// TIA Portal V18 program export: 2 tag tables, 0 data types, 2 data blocks, 5 code blocks (in call order from the OBs), 1 instance data blocks

VAR_GLOBAL   // PLC tag table "AI_Tags"
   AI_FT3210_Bon3 AT %ID128 : Real;   // Cảm biến lưu lượng nước dosing vào Bồn 3
   AI_FT3210_Bon3_HMI AT %MD756 : Real;   // Giá trị mô phỏng/HMI song song cho Cảm biến lưu lượng nước dosing vào Bồn 3
   AI_FT3210_Bon3_Use_HMI AT %M420.7 : Bool;   // Chọn chế độ mô phỏng HMI cho Cảm biến lưu lượng nước dosing vào Bồn 3
   AI_FT3210_Bon3_Sim_Req AT %M323.0 : Bool;   // Yêu cầu mô phỏng cảm biến cho Cảm biến lưu lượng nước dosing vào Bồn 3
   AI_FT3210_Bon3_Sim_Active AT %M323.1 : Bool;   // Mô phỏng cảm biến đang hoạt động cho Cảm biến lưu lượng nước dosing vào Bồn 3
   AI_FT3210_Bon3_Eff AT %MD760 : Real;   // Giá trị thực tế/mô phỏng hiệu dụng cho Cảm biến lưu lượng nước dosing vào Bồn 3
   AI_LT3213_Bon3 AT %ID132 : Real;   // Cảm biến mức liên tục Bồn 3
   AI_LT3213_Bon3_HMI AT %MD764 : Real;   // Giá trị mô phỏng/HMI song song cho Cảm biến mức liên tục Bồn 3
   AI_LT3213_Bon3_Use_HMI AT %M421.0 : Bool;   // Chọn chế độ mô phỏng HMI cho Cảm biến mức liên tục Bồn 3
   AI_LT3213_Bon3_Sim_Req AT %M323.2 : Bool;   // Yêu cầu mô phỏng cảm biến cho Cảm biến mức liên tục Bồn 3
   AI_LT3213_Bon3_Sim_Active AT %M323.3 : Bool;   // Mô phỏng cảm biến đang hoạt động cho Cảm biến mức liên tục Bồn 3
   AI_LT3213_Bon3_Eff AT %MD768 : Real;   // Giá trị thực tế/mô phỏng hiệu dụng cho Cảm biến mức liên tục Bồn 3
   AI_TT3214_Bon3 AT %ID136 : Real;   // Cảm biến nhiệt độ Bồn 3
   AI_TT3214_Bon3_HMI AT %MD772 : Real;   // Giá trị mô phỏng/HMI song song cho Cảm biến nhiệt độ Bồn 3
   AI_TT3214_Bon3_Use_HMI AT %M421.1 : Bool;   // Chọn chế độ mô phỏng HMI cho Cảm biến nhiệt độ Bồn 3
   AI_TT3214_Bon3_Sim_Req AT %M323.4 : Bool;   // Yêu cầu mô phỏng cảm biến cho Cảm biến nhiệt độ Bồn 3
   AI_TT3214_Bon3_Sim_Active AT %M323.5 : Bool;   // Mô phỏng cảm biến đang hoạt động cho Cảm biến nhiệt độ Bồn 3
   AI_TT3214_Bon3_Eff AT %MD776 : Real;   // Giá trị thực tế/mô phỏng hiệu dụng cho Cảm biến nhiệt độ Bồn 3
   AI_FT3215_Bon4 AT %ID140 : Real;   // Cảm biến lưu lượng nước dosing vào Bồn 4
   AI_FT3215_Bon4_HMI AT %MD780 : Real;   // Giá trị mô phỏng/HMI song song cho Cảm biến lưu lượng nước dosing vào Bồn 4
   AI_FT3215_Bon4_Use_HMI AT %M421.2 : Bool;   // Chọn chế độ mô phỏng HMI cho Cảm biến lưu lượng nước dosing vào Bồn 4
   AI_FT3215_Bon4_Sim_Req AT %M323.6 : Bool;   // Yêu cầu mô phỏng cảm biến cho Cảm biến lưu lượng nước dosing vào Bồn 4
   AI_FT3215_Bon4_Sim_Active AT %M323.7 : Bool;   // Mô phỏng cảm biến đang hoạt động cho Cảm biến lưu lượng nước dosing vào Bồn 4
   AI_FT3215_Bon4_Eff AT %MD784 : Real;   // Giá trị thực tế/mô phỏng hiệu dụng cho Cảm biến lưu lượng nước dosing vào Bồn 4
   AI_FQ3215_Bon4 AT %ID144 : Real;   // Bộ đếm lưu lượng tích lũy Bồn 4
   AI_FQ3215_Bon4_HMI AT %MD788 : Real;   // Giá trị mô phỏng/HMI song song cho Bộ đếm lưu lượng tích lũy Bồn 4
   AI_FQ3215_Bon4_Use_HMI AT %M421.3 : Bool;   // Chọn chế độ mô phỏng HMI cho Bộ đếm lưu lượng tích lũy Bồn 4
   AI_FQ3215_Bon4_Sim_Req AT %M324.0 : Bool;   // Yêu cầu mô phỏng cảm biến cho Bộ đếm lưu lượng tích lũy Bồn 4
   AI_FQ3215_Bon4_Sim_Active AT %M324.1 : Bool;   // Mô phỏng cảm biến đang hoạt động cho Bộ đếm lưu lượng tích lũy Bồn 4
   AI_FQ3215_Bon4_Eff AT %MD792 : Real;   // Giá trị thực tế/mô phỏng hiệu dụng cho Bộ đếm lưu lượng tích lũy Bồn 4
   AI_LS3217_Bon4_Cao AT %I0.5 : Bool;   // Cảm biến mức cao Bồn 4
   AI_LS3217_Bon4_Cao_HMI AT %M110.5 : Bool;   // Tín hiệu mô phỏng/HMI song song cho Cảm biến mức cao Bồn 4
   AI_LS3217_Bon4_Cao_HMI_Gated AT %M324.2 : Bool;   // Tín hiệu HMI đã qua xử lý chế độ cho Cảm biến mức cao Bồn 4
   AI_LS3217_Bon4_Cao_Eff AT %M324.3 : Bool;   // Tín hiệu thực tế/mô phỏng hiệu dụng cho Cảm biến mức cao Bồn 4
   AI_LT3218_Bon4 AT %ID148 : Real;   // Cảm biến mức liên tục Bồn 4
   AI_LT3218_Bon4_HMI AT %MD796 : Real;   // Giá trị mô phỏng/HMI song song cho Cảm biến mức liên tục Bồn 4
   AI_LT3218_Bon4_Use_HMI AT %M421.4 : Bool;   // Chọn chế độ mô phỏng HMI cho Cảm biến mức liên tục Bồn 4
   AI_LT3218_Bon4_Sim_Req AT %M324.4 : Bool;   // Yêu cầu mô phỏng cảm biến cho Cảm biến mức liên tục Bồn 4
   AI_LT3218_Bon4_Sim_Active AT %M324.5 : Bool;   // Mô phỏng cảm biến đang hoạt động cho Cảm biến mức liên tục Bồn 4
   AI_LT3218_Bon4_Eff AT %MD800 : Real;   // Giá trị thực tế/mô phỏng hiệu dụng cho Cảm biến mức liên tục Bồn 4
   AI_TT3219_Bon4 AT %ID152 : Real;   // Cảm biến nhiệt độ Bồn 4
   AI_TT3219_Bon4_HMI AT %MD804 : Real;   // Giá trị mô phỏng/HMI song song cho Cảm biến nhiệt độ Bồn 4
   AI_TT3219_Bon4_Use_HMI AT %M421.5 : Bool;   // Chọn chế độ mô phỏng HMI cho Cảm biến nhiệt độ Bồn 4
   AI_TT3219_Bon4_Sim_Req AT %M324.6 : Bool;   // Yêu cầu mô phỏng cảm biến cho Cảm biến nhiệt độ Bồn 4
   AI_TT3219_Bon4_Sim_Active AT %M324.7 : Bool;   // Mô phỏng cảm biến đang hoạt động cho Cảm biến nhiệt độ Bồn 4
   AI_TT3219_Bon4_Eff AT %MD808 : Real;   // Giá trị thực tế/mô phỏng hiệu dụng cho Cảm biến nhiệt độ Bồn 4
   AI_V3240_Nuoc_Bon3 AT %Q1.4 : Bool;   // Van on/off cấp nước Bồn 3
   AI_V3240_Nuoc_Bon3_M AT %M221.4 : Bool;   // Tag gương phản hồi HMI cho Van on/off cấp nước Bồn 3
   AI_CV3211_Nuoc_Bon3 AT %QD116 : Real;   // Van tuyến tính cấp nước Bồn 3
   AI_CV3211_Nuoc_Bon3_M AT %MD936 : Real;   // Tag gương phản hồi HMI cho Van tuyến tính cấp nước Bồn 3
   AI_AGTR3262_Khuay_Bon3 AT %Q1.5 : Bool;   // Động cơ khuấy Bồn 3
   AI_AGTR3262_Khuay_Bon3_M AT %M221.5 : Bool;   // Tag gương phản hồi HMI cho Động cơ khuấy Bồn 3
   AI_AGTR3262_Toc_Do_AO AT %QD120 : Real;   // Tín hiệu tốc độ khuấy Bồn 3
   AI_AGTR3262_Toc_Do_AO_M AT %MD940 : Real;   // Tag gương phản hồi HMI cho Tín hiệu tốc độ khuấy Bồn 3
   AI_V3242_Xa_Bon3 AT %Q1.6 : Bool;   // Van xả đáy Bồn 3 số 1
   AI_V3242_Xa_Bon3_M AT %M221.6 : Bool;   // Tag gương phản hồi HMI cho Van xả đáy Bồn 3 số 1
   AI_V3243_Xa_Bon3 AT %Q1.7 : Bool;   // Van xả đáy Bồn 3 số 2
   AI_V3243_Xa_Bon3_M AT %M221.7 : Bool;   // Tag gương phản hồi HMI cho Van xả đáy Bồn 3 số 2
   AI_V3244_Xa_Bon3 AT %Q2.0 : Bool;   // Van xả đáy Bồn 3 số 3
   AI_V3244_Xa_Bon3_M AT %M222.0 : Bool;   // Tag gương phản hồi HMI cho Van xả đáy Bồn 3 số 3
   AI_V3245_Nuoc_Bon4 AT %Q2.1 : Bool;   // Van on/off cấp nước Bồn 4
   AI_V3245_Nuoc_Bon4_M AT %M222.1 : Bool;   // Tag gương phản hồi HMI cho Van on/off cấp nước Bồn 4
   AI_CV3216_Hoi_Bon4 AT %QD124 : Real;   // Van tuyến tính gia nhiệt mô phỏng Bồn 4
   AI_CV3216_Hoi_Bon4_M AT %MD944 : Real;   // Tag gương phản hồi HMI cho Van tuyến tính gia nhiệt mô phỏng Bồn 4
   AI_AGTR3263_Khuay_Bon4 AT %Q2.2 : Bool;   // Động cơ khuấy Bồn 4
   AI_AGTR3263_Khuay_Bon4_M AT %M222.2 : Bool;   // Tag gương phản hồi HMI cho Động cơ khuấy Bồn 4
   AI_AGTR3263_Dao_Chieu AT %Q2.3 : Bool;   // Lệnh đảo chiều động cơ khuấy Bồn 4
   AI_AGTR3263_Dao_Chieu_M AT %M222.3 : Bool;   // Tag gương phản hồi HMI cho Lệnh đảo chiều động cơ khuấy Bồn 4
   AI_AGTR3263_Toc_Do_AO AT %QD128 : Real;   // Tốc độ đặt động cơ khuấy Bồn 4
   AI_AGTR3263_Toc_Do_AO_M AT %MD948 : Real;   // Tag gương phản hồi HMI cho Tốc độ đặt động cơ khuấy Bồn 4
   AI_V3247_Xa_Bon4 AT %Q2.4 : Bool;   // Van xả đáy Bồn 4 số 1
   AI_V3247_Xa_Bon4_M AT %M222.4 : Bool;   // Tag gương phản hồi HMI cho Van xả đáy Bồn 4 số 1
   AI_V3248_Xa_Bon4 AT %Q2.5 : Bool;   // Van xả đáy Bồn 4 số 2
   AI_V3248_Xa_Bon4_M AT %M222.5 : Bool;   // Tag gương phản hồi HMI cho Van xả đáy Bồn 4 số 2
   AI_V3249_Xa_Bon4 AT %Q2.6 : Bool;   // Van xả đáy Bồn 4 số 3
   AI_V3249_Xa_Bon4_M AT %M222.6 : Bool;   // Tag gương phản hồi HMI cho Van xả đáy Bồn 4 số 3
   AI_Pump3265_Chuyen_Nhanh2 AT %Q2.7 : Bool;   // Bơm chuyển dung dịch Nhánh 2 xuống bồn chứa
   AI_Pump3265_Chuyen_Nhanh2_M AT %M222.7 : Bool;   // Tag gương phản hồi HMI cho Bơm chuyển dung dịch Nhánh 2 xuống bồn chứa
   AI_HMI_Operator_Login AT %M422.5 : Bool;   // Đăng nhập quyền Operator
   AI_HMI_Engineer_Login AT %M422.6 : Bool;   // Đăng nhập quyền Engineer
   AI_HMI_Admin_Login AT %M422.7 : Bool;   // Đăng nhập quyền Admin
   AI_HMI_Che_Do_Manual AT %M423.0 : Bool;   // Cho phép điều khiển tay từng thiết bị
   AI_HMI_Ack_Alarm AT %M423.1 : Bool;   // Xác nhận cảnh báo
   AI_HMI_Reset_Alarm AT %M423.2 : Bool;   // Reset alarm bằng HMI
   AI_Gia_Lap_Mat_Ket_Noi_HMI AT %M423.3 : Bool;   // Nút giả lập mất kết nối PLC
   AI_HMI_User_Level AT %MW520 : Int;   // Mức quyền hiện tại: 1 Operator, 2 Engineer, 3 Admin
   AI_HMI_Cho_Phep_Sua_Thong_So AT %M327.2 : Bool;   // Cờ cho phép sửa công thức và PID
   AI_HMI_Alarm_Status AT %MW522 : Int;   // Mã cảnh báo tổng hợp cho WinCC TextList
   AI_HMI_AnToan_Status AT %MW524 : Int;   // Mã chẩn đoán an toàn ưu tiên
   AI_PLC2_Auto_Enable AT %M328.1 : Bool;   // Cho phép chạy Auto Nhánh 2 Bồn 3-4
   AI_PLC2_EStop_Latch AT %M328.2 : Bool;   // Chốt dừng khẩn HMI/SCADA Nhánh 2 Bồn 3-4
   AI_PLC2_Loi_Tong AT %M328.3 : Bool;   // Lỗi tổng khóa Auto Nhánh 2 Bồn 3-4
   AI_PLC2_Loi_Dry_Run AT %M328.4 : Bool;   // Lỗi chạy khô bơm Nhánh 2 Bồn 3-4
   AI_PLC2_Loi_Dosing AT %M328.5 : Bool;   // Lỗi quá thời gian dosing Nhánh 2 Bồn 3-4
   AI_PLC2_Loi_Truyen_Thong AT %M328.6 : Bool;   // Lỗi truyền thông mô phỏng Nhánh 2 Bồn 3-4
   AI_PLC2_State AT %MW528 : Int;   // Mã bước chu trình Nhánh 2 Bồn 3-4
   AI_PLC2_Step_Bon3_Dosing AT %M330.4 : Bool;   // Bồn 3 đang dosing nước
   AI_PLC2_Step_Bon3_Tip AT %M330.5 : Bool;   // Bồn 3 đang mô phỏng tip cốt tương đậu đậm đặc
   AI_PLC2_Step_Bon3_Khuay AT %M330.6 : Bool;   // Bồn 3 đang khuấy ban đầu
   AI_PLC2_Step_Bon3_Xa AT %M330.7 : Bool;   // Bồn 3 đang xả sang Bồn 4
   AI_PLC2_Step_Bon4_Dosing AT %M331.0 : Bool;   // Bồn 4 đang dosing bổ sung
   AI_PLC2_Step_Bon4_Tip AT %M331.1 : Bool;   // Bồn 4 đang tip phụ gia
   AI_PLC2_Step_Bon4_Khuay_Thuan AT %M331.2 : Bool;   // Bồn 4 khuấy chiều thuận
   AI_PLC2_Step_Bon4_Khuay_Nghich AT %M331.3 : Bool;   // Bồn 4 khuấy chiều ngược
   AI_PLC2_Step_Bon4_PID_Mo_Phong AT %M331.4 : Bool;   // Bồn 4 chạy PID mô phỏng
   AI_PLC2_Step_Bon4_Thanh_Trung AT %M331.5 : Bool;   // Bồn 4 giữ thời gian thanh trùng
   AI_PLC2_Xa_Bon3_Xong AT %M331.6 : Bool;   // Bồn 3 đã xả hết
   AI_PLC2_Xa_Bon4_Xong AT %M331.7 : Bool;   // Bồn 4 đã xả hết
   AI_PLC2_Me_Nhanh2_Hoan_Thanh AT %M332.5 : Bool;   // Cờ hoàn thành Nhánh 2 gửi sang PLC1
   AI_PLC2_Me_Nhanh2_Hoan_Thanh_M AT %M224.6 : Bool;   // Tag gương phản hồi HMI cho cờ hoàn thành Nhánh 2 gửi sang PLC1
   AI_Pump3265_Chuyen_Nhanh2_Cmd_Nhan AT %M333.0 : Bool;   // Nhận lệnh chạy bơm chuyển Nhánh 2 từ PLC1
   AI_Pump3265_Chuyen_Nhanh2_Cmd_Nhan_HMI AT %M111.1 : Bool;   // Tín hiệu mô phỏng/HMI song song cho lệnh chạy bơm chuyển Nhánh 2 từ PLC1
   AI_Nut_Khoi_Dong_Nhan AT %M333.2 : Bool;   // nút khởi động nhận từ PLC1
   AI_Nut_Khoi_Dong_Nhan_HMI AT %M111.2 : Bool;   // Tín hiệu mô phỏng/HMI song song cho nút khởi động nhận từ PLC1
   AI_Nut_Khoi_Dong_Nhan_HMI_Gated AT %M333.3 : Bool;   // Tín hiệu HMI đã qua xử lý chế độ cho nút khởi động nhận từ PLC1
   AI_Nut_Khoi_Dong_Nhan_Eff AT %M333.4 : Bool;   // Tín hiệu thực tế/mô phỏng hiệu dụng cho nút khởi động nhận từ PLC1
   AI_Nut_Dung_Nhan AT %M333.5 : Bool;   // nút dừng nhận từ PLC1
   AI_Nut_Dung_Nhan_HMI AT %M111.3 : Bool;   // Tín hiệu mô phỏng/HMI song song cho nút dừng nhận từ PLC1
   AI_Nut_Dung_Nhan_HMI_Gated AT %M333.6 : Bool;   // Tín hiệu HMI đã qua xử lý chế độ cho nút dừng nhận từ PLC1
   AI_Nut_Dung_Nhan_Eff AT %M333.7 : Bool;   // Tín hiệu thực tế/mô phỏng hiệu dụng cho nút dừng nhận từ PLC1
   AI_Nut_Reset_Nhan AT %M334.0 : Bool;   // nút reset nhận từ PLC1
   AI_Nut_Reset_Nhan_HMI AT %M111.4 : Bool;   // Tín hiệu mô phỏng/HMI song song cho nút reset nhận từ PLC1
   AI_Nut_Reset_Nhan_HMI_Gated AT %M334.1 : Bool;   // Tín hiệu HMI đã qua xử lý chế độ cho nút reset nhận từ PLC1
   AI_Nut_Reset_Nhan_Eff AT %M334.2 : Bool;   // Tín hiệu thực tế/mô phỏng hiệu dụng cho nút reset nhận từ PLC1
   AI_Nut_EStop_Nhan AT %M334.3 : Bool;   // nút dừng khẩn nhận từ PLC1
   AI_Nut_EStop_Nhan_HMI AT %M111.5 : Bool;   // Tín hiệu mô phỏng/HMI song song cho nút dừng khẩn nhận từ PLC1
   AI_Nut_EStop_Nhan_HMI_Gated AT %M334.4 : Bool;   // Tín hiệu HMI đã qua xử lý chế độ cho nút dừng khẩn nhận từ PLC1
   AI_Nut_EStop_Nhan_Eff AT %M334.5 : Bool;   // Tín hiệu thực tế/mô phỏng hiệu dụng cho nút dừng khẩn nhận từ PLC1
   AI_Clock_1Hz AT %M100.5 : Bool;   // Clock 1Hz system memory bit
   AI_FirstScan AT %M101.0 : Bool;   // First Scan system memory bit
   AI_PLC2_Last_CmdSeq AT %MW80 : Int;   // Last processed command sequence
   AI_PLC2_CmdSeq_New AT %M82.0 : Bool;   // New command sequence received
   AI_MB_TCP_Server_Error AT %M82.1 : Bool;   // Modbus TCP Server Error
   AI_MB_TCP_Server_Status AT %MW84 : Word;   // Modbus TCP Server Status
   AI_MB_TCP_Server_NDR AT %M82.2 : Bool;   // Modbus TCP Server New Data Received
   AI_MB_TCP_Server_DR AT %M82.3 : Bool;   // Modbus TCP Server Data Read
   AI_PLC1_Tip_Bon1_Xong_HMI AT %M423.4 : Bool;   // Nút mô phỏng tip Bồn 1 đã hoàn tất
   AI_PLC1_Khuay_Bon1_Xong_HMI AT %M423.5 : Bool;   // Nút mô phỏng hết thời gian khuấy Bồn 1
   AI_PLC1_Tip_Bon2_Xong_HMI AT %M423.6 : Bool;   // Nút mô phỏng tip Bồn 2 đã hoàn tất
   AI_PLC1_Khuay_Thuan_Bon2_Xong_HMI AT %M423.7 : Bool;   // Nút mô phỏng hết thời gian khuấy thuận Bồn 2
   AI_PLC1_Khuay_Nghich_Bon2_Xong_HMI AT %M424.0 : Bool;   // Nút mô phỏng hết thời gian khuấy ngược Bồn 2
   AI_PLC1_Thanh_Trung_Bon2_Xong_HMI AT %M424.1 : Bool;   // Nút mô phỏng hết thời gian thanh trùng Bồn 2
   AI_PLC2_Tip_Bon3_Xong_HMI AT %M424.2 : Bool;   // Nút mô phỏng tip Bồn 3 đã hoàn tất
   AI_PLC2_Khuay_Bon3_Xong_HMI AT %M424.3 : Bool;   // Nút mô phỏng hết thời gian khuấy Bồn 3
   AI_PLC2_Tip_Bon4_Xong_HMI AT %M424.4 : Bool;   // Nút mô phỏng tip Bồn 4 đã hoàn tất
   AI_PLC2_Khuay_Thuan_Bon4_Xong_HMI AT %M424.5 : Bool;   // Nút mô phỏng hết thời gian khuấy thuận Bồn 4
   AI_PLC2_Khuay_Nghich_Bon4_Xong_HMI AT %M424.6 : Bool;   // Nút mô phỏng hết thời gian khuấy ngược Bồn 4
   AI_PLC2_Thanh_Trung_Bon4_Xong_HMI AT %M424.7 : Bool;   // Nút mô phỏng hết thời gian thanh trùng Bồn 4
   AI_BonChua_Nhan_Dich_Xong_HMI AT %M425.0 : Bool;   // Nút mô phỏng nhận dịch vào Bồn chứa 01 xong
   AI_BonChua_Chuyen_Bon2_Xong_HMI AT %M425.1 : Bool;   // Nút mô phỏng chuyển sang Bồn chứa 02 xong
   AI_HMI_SP_PLC1_Nuoc_Bon1 AT %MD880 : Real;   // Lượng nước dosing Bồn 1
   AI_HMI_SP_PLC1_Nuoc_Bon2 AT %MD884 : Real;   // Lượng nước dosing bổ sung Bồn 2
   AI_HMI_SP_PLC1_Toc_Do_Bon1 AT %MD888 : Real;   // Tốc độ khuấy Bồn 1
   AI_HMI_SP_PLC1_Toc_Do_Bon2_Main AT %MD892 : Real;   // Tốc độ khuấy chính Bồn 2
   AI_HMI_SP_PLC1_Nhiet_Do_Bon2 AT %MD896 : Real;   // Setpoint nhiệt/PID Bồn 2
   AI_HMI_SP_PLC2_Nuoc_Bon3 AT %MD900 : Real;   // Lượng nước dosing Bồn 3
   AI_HMI_SP_PLC2_Nuoc_Bon4 AT %MD904 : Real;   // Lượng nước dosing bổ sung Bồn 4
   AI_HMI_SP_PLC2_Toc_Do_Bon3 AT %MD908 : Real;   // Tốc độ khuấy Bồn 3
   AI_HMI_SP_PLC2_Toc_Do_Bon4_Main AT %MD912 : Real;   // Tốc độ khuấy chính Bồn 4
   AI_HMI_SP_PLC2_Nhiet_Do_Bon4 AT %MD916 : Real;   // Setpoint nhiệt/PID mô phỏng Bồn 4
   AI_HMI_SP_BonChua1_Nhiet_Giai_Nhiet AT %MD920 : Real;   // Nhiệt độ giải nhiệt đích Bồn chứa 01
   AI_HMI_SP_Loc_Ap_Suat_Max AT %MD924 : Real;   // Ngưỡng áp suất cao trước màng lọc
   AI_HMI_SP_Time_Khuay_Bon1 AT %MD928 : Time;   // Thời gian khuấy Bồn 1
   AI_HMI_SP_Time_Khuay_Bon3 AT %MD932 : Time;   // Thời gian khuấy Bồn 3
   AI_HMI_SP_Time_Fwd AT %MD936 : Time;   // Thời gian khuấy chiều thuận
   AI_HMI_SP_Time_Rev AT %MD940 : Time;   // Thời gian khuấy chiều ngược
   AI_HMI_SP_Time_Sterilize AT %MD944 : Time;   // Thời gian giữ nhiệt thanh trùng
   AI_PLC1_Khuay_Bon1_Xong AT %M335.3 : Bool;   // Trạng thái tự động xong khuấy Bồn 1
   AI_PLC1_Khuay_Thuan_Bon2_Xong AT %M335.4 : Bool;   // Trạng thái tự động xong khuấy thuận Bồn 2
   AI_PLC1_Khuay_Nghich_Bon2_Xong AT %M335.5 : Bool;   // Trạng thái tự động xong khuấy ngược Bồn 2
   AI_PLC1_Thanh_Trung_Bon2_Xong AT %M335.6 : Bool;   // Trạng thái tự động xong thanh trùng Bồn 2
   AI_PLC2_Khuay_Bon3_Xong AT %M335.7 : Bool;   // Trạng thái tự động xong khuấy Bồn 3
   AI_PLC2_Khuay_Thuan_Bon4_Xong AT %M336.0 : Bool;   // Trạng thái tự động xong khuấy thuận Bồn 4
   AI_PLC2_Khuay_Nghich_Bon4_Xong AT %M336.1 : Bool;   // Trạng thái tự động xong khuấy ngược Bồn 4
   AI_PLC2_Thanh_Trung_Bon4_Xong AT %M336.2 : Bool;   // Trạng thái tự động xong thanh trùng Bồn 4
   AI_PID_Bon2_Enable AT %M336.3 : Bool;   // Cho phép PID Bồn 2
   AI_PID_Bon2_ManualEnable AT %M336.4 : Bool;   // Chế độ manual PID Bồn 2
   AI_PID_Bon2_Error AT %M336.5 : Bool;   // Lỗi khối PID Bồn 2
   AI_PID_Bon4_Enable AT %M336.6 : Bool;   // Cho phép PID mô phỏng Bồn 4
   AI_PID_Bon4_ManualEnable AT %M336.7 : Bool;   // Chế độ manual PID Bồn 4
   AI_PID_Bon4_Error AT %M337.0 : Bool;   // Lỗi khối PID Bồn 4
   AI_PID_Bon2_ErrorBits AT %MD948 : DWord;   // Mã lỗi DWORD PID Bồn 2
   AI_PID_Bon4_ErrorBits AT %MD952 : DWord;   // Mã lỗi DWORD PID Bồn 4
   AI_PID_Bon2_SP AT %MD956 : Real;   // Setpoint đưa vào PID Bồn 2
   AI_PID_Bon2_Err AT %MD960 : Real;   // Sai lệch PID Bồn 2 = SP - PV
   AI_PID_Bon2_CV AT %MD964 : Real;   // Giá trị điều khiển PID Bồn 2
   AI_PID_Bon2_ManualValue AT %MD968 : Real;   // Giá trị manual PID Bồn 2
   AI_PID_Bon4_SP AT %MD972 : Real;   // Setpoint đưa vào PID mô phỏng Bồn 4
   AI_PID_Bon4_Err AT %MD976 : Real;   // Sai lệch PID mô phỏng Bồn 4 = SP - PV
   AI_PID_Bon4_CV AT %MD980 : Real;   // Giá trị điều khiển PID mô phỏng Bồn 4
   AI_PID_Bon4_ManualValue AT %MD984 : Real;   // Giá trị manual PID Bồn 4
   AI_TT3219_Bon4_Sim AT %MD988 : Real;   // Nhiệt độ mô phỏng nội bộ cho PID Bồn 4
   AI_PID_Bon4_Tang_Nhiet_Buoc AT %MD992 : Real;   // Mức tăng nhiệt mô phỏng mỗi chu kỳ OB31
   AI_TT3219_Bon4_Target AT %MD996 : Real;   // Nhiệt độ đích mô phỏng bồn 4
   AI_TT3219_Bon4_Sim_Pure AT %MD1000 : Real;   // Nhiệt độ mô phỏng chưa có nhiễu bồn 4
   AI_PID_Bon4_Temp_Val_1 AT %MD1004 : Real;   // Biến tạm mô phỏng nhiệt độ 1
   AI_PID_Bon4_Temp_Val_2 AT %MD1008 : Real;   // Biến tạm mô phỏng nhiệt độ 2
   AI_PID_Bon4_Sim_Counter AT %MD1012 : Real;   // Đồng hồ chu kỳ mô phỏng
   AI_PID_Bon4_Sim_Angle AT %MD1016 : Real;   // Góc lượng giác nhiễu
   AI_PID_Bon4_Sim_Sin AT %MD1020 : Real;   // Giá trị hình sin nhiễu
   AI_PID_Bon4_Sim_Noise AT %MD1024 : Real;   // Giá trị nhiễu nhiệt độ
   AI_PID_Bon4_State AT %MW536 : Int;   // Trạng thái khối PID Bồn 4
   AI_PLC2_Stop_Active AT %M337.2 : Bool;   // Tín hiệu dừng active PLC2
   AI_AGTR3263_Khuay_Active AT %M337.5 : Bool;   // Trạng thái khuấy Bồn 4 active
   AI_AGTR3263_Should_Run AT %M337.6 : Bool;   // Yêu cầu chạy động cơ Bồn 4
   AI_HMI_Use_Sim_Input_PLC2 AT %M338.0 : Bool;   // Cho phép sử dụng đầu vào mô phỏng PLC2
   AI_Pump3265_Chuyen_Nhanh2_Cmd_Nhan_Eff AT %M338.3 : Bool;   // Lệnh chạy bơm chuyển Nhánh 2 nhận được hiệu dụng
   AI_Pump3265_Chuyen_Nhanh2_Cmd_Nhan_HMI_Gated AT %M338.5 : Bool;   // Lệnh chạy bơm chuyển Nhánh 2 HMI gated
   AI_PLC2_SP_Valid AT %M338.7 : Bool;   // Setpoint PLC2 hợp lệ
   AI_PLC2_Loi_Setpoint AT %M339.2 : Bool;   // Lỗi Setpoint PLC2
   AI_Init_Defaults_Done_PLC2 AT %M339.5 : Bool;   // Khởi tạo Setpoint mặc định PLC2 hoàn tất
   AI_Init_Trigger_PLC2 AT %M340.0 : Bool;   // Cờ kích hoạt nạp recipe mặc định PLC2
   AI_HMI_Load_Default_Recipe AT %M340.2 : Bool;   // Yêu cầu nạp lại Recipe mặc định từ HMI
   AI_PLC2_Load_Default_Cmd_Nhan AT %M340.4 : Bool;   // Nhận lệnh nạp recipe mặc định từ PLC1
   AI_PLC2_Load_Default_Cmd_Nhan_HMI AT %M111.6 : Bool;   // Tín hiệu mô phỏng/HMI cho nhận lệnh nạp recipe
   AI_PLC2_Load_Default_Cmd_Nhan_HMI_Gated AT %M340.5 : Bool;   // Tín hiệu nhận lệnh nạp recipe HMI gated
   AI_PLC2_Load_Default_Cmd_Nhan_Eff AT %M340.6 : Bool;   // Tín hiệu nhận lệnh nạp recipe hiệu dụng
   AI_PLC2_Load_Default_Done AT %M340.7 : Bool;   // Báo nạp recipe mặc định xong gửi sang PLC1
   AI_PLC2_Load_Default_Done_M AT %M225.1 : Bool;   // Tag gương phản hồi HMI cho báo nạp recipe xong PLC2
   AI_HMI_Sim_Mode AT %M341.3 : Bool;   // Cho phép toàn bộ tín hiệu mô phỏng HMI tác động vào input hiệu dụng
   AI_HMI_Run_Enable AT %M341.4 : Bool;   // Cho phép vận hành từ HMI ở chế độ thật
   AI_System_Mode_Real AT %M341.5 : Bool;   // Hệ thống đang hoạt động ở chế độ thực tế
   AI_System_Mode_Sim AT %M341.6 : Bool;   // Hệ thống đang hoạt động ở chế độ mô phỏng
   AI_HMI_Sim_Active_Warning AT %M341.7 : Bool;   // Cảnh báo chế độ mô phỏng HMI đang hoạt động
   AI_PID_Bon4_Kp_HMI AT %MD1036 : Real;   // HMI parameter for Kp PID Bồn 4
   AI_PID_Bon4_Ti_HMI AT %MD1040 : Real;   // HMI parameter for Ti PID Bồn 4
END_VAR

VAR_GLOBAL   // PLC tag table "Default tag table"
   System_Byte AT %MB101 : Byte;
   FirstScan AT %M101.0 : Bool;
   DiagStatusUpdate AT %M101.1 : Bool;
   AlwaysTRUE AT %M101.2 : Bool;
   AlwaysFALSE AT %M101.3 : Bool;
   Clock_Byte AT %MB100 : Byte;
   Clock_10Hz AT %M100.0 : Bool;
   Clock_5Hz AT %M100.1 : Bool;
   "Clock_2.5Hz" AT %M100.2 : Bool;
   Clock_2Hz AT %M100.3 : Bool;
   "Clock_1.25Hz" AT %M100.4 : Bool;
   Clock_1Hz AT %M100.5 : Bool;
   "Clock_0.625Hz" AT %M100.6 : Bool;
   "Clock_0.5Hz" AT %M100.7 : Bool;
END_VAR

DATA_BLOCK "AI_Timers_PLC2"   // DB1
TITLE = AI_Timers_PLC2
{ S7_Optimized_Access := 'TRUE' }
VERSION : 0.1
// Global DB containing all timers and PID instances
// stored: AutoNumber true, DBAccessibleFromOPCUA true, IsOnlyStoredInLoadMemory false, IsRetainMemResEnabled false, IsWriteProtectedInAS false, MemoryReserve 100
   VAR
      AI_Timer_Dosing_Bon3 : IEC_TIMER;
      AI_Timer_Dosing_Bon4 : IEC_TIMER;
      AI_Timer_Khuay_Bon3 : IEC_TIMER;
      AI_Timer_Khuay_Thuan_Bon4 : IEC_TIMER;
      AI_Timer_Khuay_Nghich_Bon4 : IEC_TIMER;
      AI_Timer_Thanh_Trung_Bon4 : IEC_TIMER;
   END_VAR
BEGIN
END_DATA_BLOCK

DATA_BLOCK "DB_Modbus_Holding_Register_DB"   // DB20
TITLE = DB_Modbus_Holding_Register_DB
{ S7_Optimized_Access := 'FALSE' }
VERSION : 0.1
// DB communication via Modbus TCP
// stored: AutoNumber false, DBAccessibleFromOPCUA true, IsOnlyStoredInLoadMemory false, IsWriteProtectedInAS false
   VAR
      CmdSeq : Int;
      Cmd_Start : Bool;
      Cmd_Stop : Bool;
      Cmd_Reset : Bool;
      Cmd_EStop : Bool;
      Cmd_Pump_Branch2_To_SubTanks : Bool;
      Cmd_Load_Recipe : Bool;
      Heartbeat_Client : Int;
      AckSeq : Int;
      Done_Branch2 : Bool;
      Done_Recipe : Bool;
      Alarm : Bool;
      State : Int;
      PID_Bon4_SP : Real;
      PID_Bon4_PV : Real;
      PID_Bon4_CV : Real;
      Heartbeat_Server : Int;
   END_VAR
BEGIN
END_DATA_BLOCK

ORGANIZATION_BLOCK "Main"   // OB1, LAD, ProgramCycle
TITLE = "Main Program Sweep (Cycle)"
{ S7_Optimized_Access := 'TRUE' }
VERSION : 0.1
// stored: AutoNumber true, IsIECCheckEnabled false, SetENOAutomatically false
   VAR_INPUT
      Initial_Call : Bool;   // Initial call of this OB
      Remanence : Bool;   // =True, if remanent data are available
   END_VAR
BEGIN

REGION Network 1: Modbus TCP Server - Call MB_SERVER
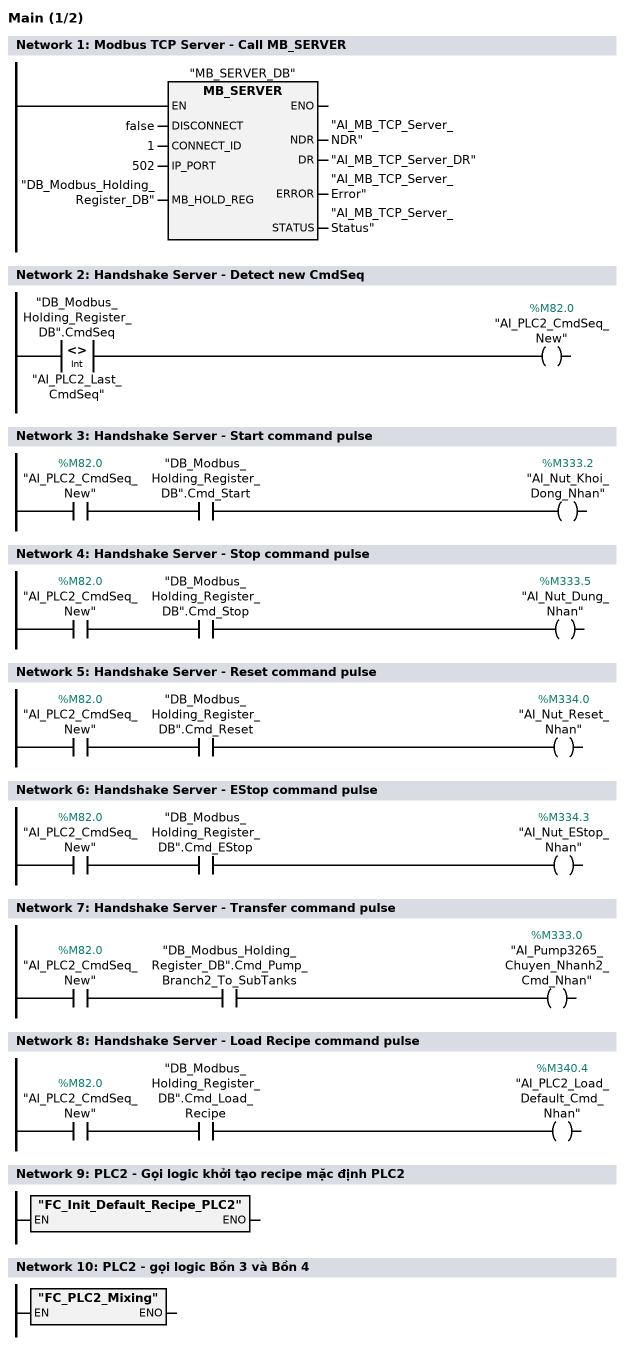
   RUNG wire#powerrail
      { S7_Templates := "[card1200 := 1, card1500 := 0]" } "MB_SERVER_DB".MB_SERVER(DISCONNECT := false, CONNECT_ID := 1, IP_PORT := 502, MB_HOLD_REG := "DB_Modbus_Holding_Register_DB", NDR => "AI_MB_TCP_Server_NDR", DR => "AI_MB_TCP_Server_DR", ERROR => "AI_MB_TCP_Server_Error", STATUS => "AI_MB_TCP_Server_Status")
   END_RUNG
   // the same network as SCL:
   "MB_SERVER_DB"(DISCONNECT := false,   // MB_SERVER
                  CONNECT_ID := 1,
                  IP_PORT := 502,
                  MB_HOLD_REG := "DB_Modbus_Holding_Register_DB",
                  NDR => "AI_MB_TCP_Server_NDR",
                  DR => "AI_MB_TCP_Server_DR",
                  ERROR => "AI_MB_TCP_Server_Error",
                  STATUS => "AI_MB_TCP_Server_Status");
END_REGION

REGION Network 2: Handshake Server - Detect new CmdSeq
   RUNG wire#powerrail
      { S7_Templates := "SrcType := Int" } NE_Contact(in1 := "DB_Modbus_Holding_Register_DB".CmdSeq, in2 := "AI_PLC2_Last_CmdSeq")
      Coil( "AI_PLC2_CmdSeq_New" )
   END_RUNG
   // the same network as SCL:
   "AI_PLC2_CmdSeq_New" := "DB_Modbus_Holding_Register_DB".CmdSeq <> "AI_PLC2_Last_CmdSeq";
END_REGION

REGION Network 3: Handshake Server - Start command pulse
   RUNG wire#powerrail
      Contact( "AI_PLC2_CmdSeq_New" )
      Contact( "DB_Modbus_Holding_Register_DB".Cmd_Start )
      Coil( "AI_Nut_Khoi_Dong_Nhan" )
   END_RUNG
   // the same network as SCL:
   "AI_Nut_Khoi_Dong_Nhan" := "AI_PLC2_CmdSeq_New" AND "DB_Modbus_Holding_Register_DB".Cmd_Start;
END_REGION

REGION Network 4: Handshake Server - Stop command pulse
   RUNG wire#powerrail
      Contact( "AI_PLC2_CmdSeq_New" )
      Contact( "DB_Modbus_Holding_Register_DB".Cmd_Stop )
      Coil( "AI_Nut_Dung_Nhan" )
   END_RUNG
   // the same network as SCL:
   "AI_Nut_Dung_Nhan" := "AI_PLC2_CmdSeq_New" AND "DB_Modbus_Holding_Register_DB".Cmd_Stop;
END_REGION

REGION Network 5: Handshake Server - Reset command pulse
   RUNG wire#powerrail
      Contact( "AI_PLC2_CmdSeq_New" )
      Contact( "DB_Modbus_Holding_Register_DB".Cmd_Reset )
      Coil( "AI_Nut_Reset_Nhan" )
   END_RUNG
   // the same network as SCL:
   "AI_Nut_Reset_Nhan" := "AI_PLC2_CmdSeq_New" AND "DB_Modbus_Holding_Register_DB".Cmd_Reset;
END_REGION

REGION Network 6: Handshake Server - EStop command pulse
   RUNG wire#powerrail
      Contact( "AI_PLC2_CmdSeq_New" )
      Contact( "DB_Modbus_Holding_Register_DB".Cmd_EStop )
      Coil( "AI_Nut_EStop_Nhan" )
   END_RUNG
   // the same network as SCL:
   "AI_Nut_EStop_Nhan" := "AI_PLC2_CmdSeq_New" AND "DB_Modbus_Holding_Register_DB".Cmd_EStop;
END_REGION

REGION Network 7: Handshake Server - Transfer command pulse
   RUNG wire#powerrail
      Contact( "AI_PLC2_CmdSeq_New" )
      Contact( "DB_Modbus_Holding_Register_DB".Cmd_Pump_Branch2_To_SubTanks )
      Coil( "AI_Pump3265_Chuyen_Nhanh2_Cmd_Nhan" )
   END_RUNG
   // the same network as SCL:
   "AI_Pump3265_Chuyen_Nhanh2_Cmd_Nhan" := "AI_PLC2_CmdSeq_New" AND "DB_Modbus_Holding_Register_DB".Cmd_Pump_Branch2_To_SubTanks;
END_REGION

REGION Network 8: Handshake Server - Load Recipe command pulse
   RUNG wire#powerrail
      Contact( "AI_PLC2_CmdSeq_New" )
      Contact( "DB_Modbus_Holding_Register_DB".Cmd_Load_Recipe )
      Coil( "AI_PLC2_Load_Default_Cmd_Nhan" )
   END_RUNG
   // the same network as SCL:
   "AI_PLC2_Load_Default_Cmd_Nhan" := "AI_PLC2_CmdSeq_New" AND "DB_Modbus_Holding_Register_DB".Cmd_Load_Recipe;
END_REGION

REGION Network 9: PLC2 - Gọi logic khởi tạo recipe mặc định PLC2
   RUNG wire#powerrail
      "FC_Init_Default_Recipe_PLC2"()
   END_RUNG
   // the same network as SCL:
   "FC_Init_Default_Recipe_PLC2"();
END_REGION

REGION Network 10: PLC2 - gọi logic Bồn 3 và Bồn 4
   RUNG wire#powerrail
      "FC_PLC2_Mixing"()
   END_RUNG
   // the same network as SCL:
   "FC_PLC2_Mixing"();
END_REGION

REGION Network 11: PLC2 - cập nhật mirror HMI
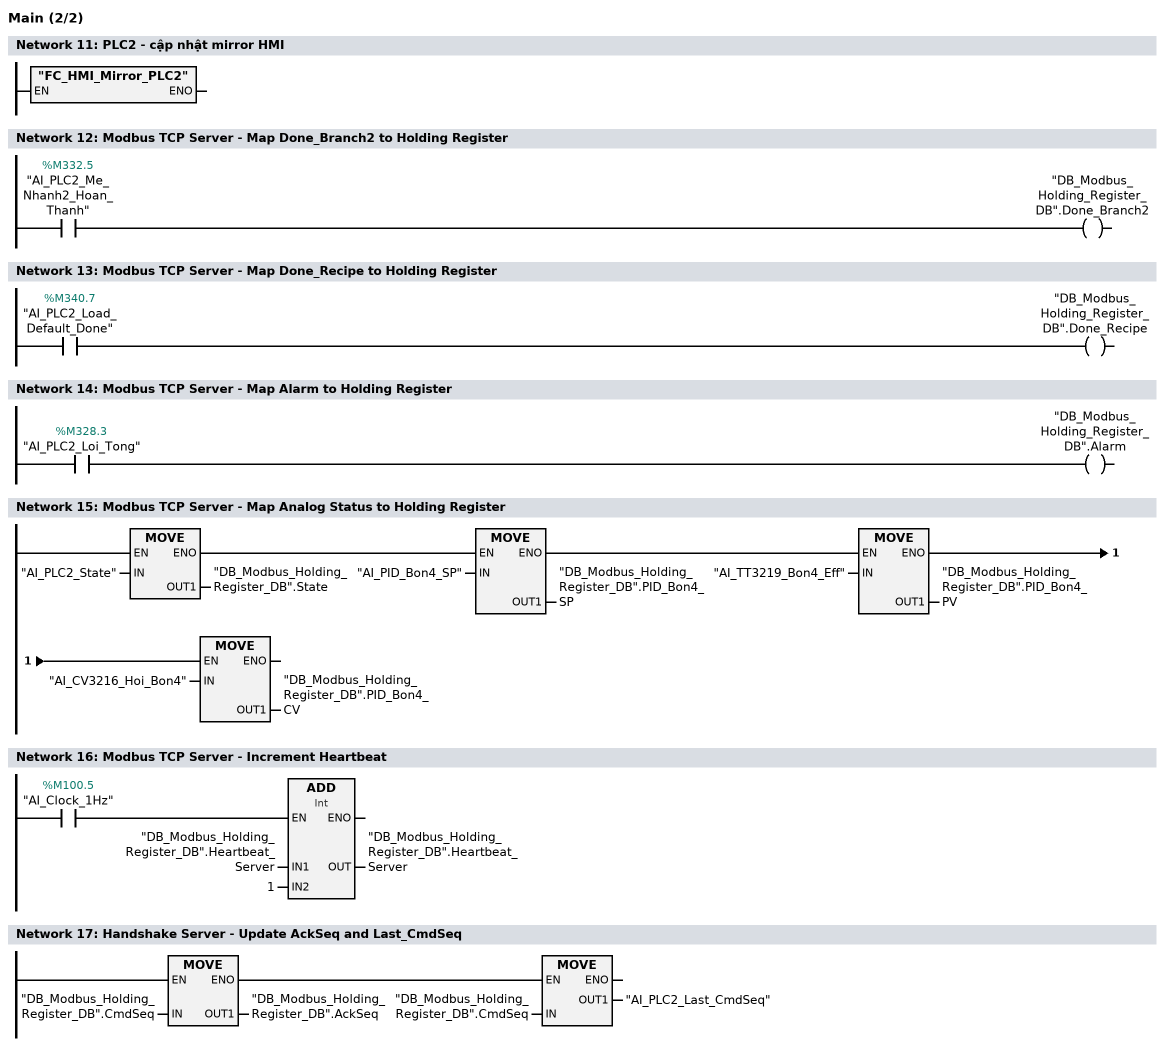
   RUNG wire#powerrail
      "FC_HMI_Mirror_PLC2"()
   END_RUNG
   // the same network as SCL:
   "FC_HMI_Mirror_PLC2"();
END_REGION

REGION Network 12: Modbus TCP Server - Map Done_Branch2 to Holding Register
   RUNG wire#powerrail
      Contact( "AI_PLC2_Me_Nhanh2_Hoan_Thanh" )
      Coil( "DB_Modbus_Holding_Register_DB".Done_Branch2 )
   END_RUNG
   // the same network as SCL:
   "DB_Modbus_Holding_Register_DB".Done_Branch2 := "AI_PLC2_Me_Nhanh2_Hoan_Thanh";
END_REGION

REGION Network 13: Modbus TCP Server - Map Done_Recipe to Holding Register
   RUNG wire#powerrail
      Contact( "AI_PLC2_Load_Default_Done" )
      Coil( "DB_Modbus_Holding_Register_DB".Done_Recipe )
   END_RUNG
   // the same network as SCL:
   "DB_Modbus_Holding_Register_DB".Done_Recipe := "AI_PLC2_Load_Default_Done";
END_REGION

REGION Network 14: Modbus TCP Server - Map Alarm to Holding Register
   RUNG wire#powerrail
      Contact( "AI_PLC2_Loi_Tong" )
      Coil( "DB_Modbus_Holding_Register_DB".Alarm )
   END_RUNG
   // the same network as SCL:
   "DB_Modbus_Holding_Register_DB".Alarm := "AI_PLC2_Loi_Tong";
END_REGION

REGION Network 15: Modbus TCP Server - Map Analog Status to Holding Register
   RUNG wire#powerrail
      { S7_GenerateENO := "TRUE" } Move(in := "AI_PLC2_State", out1 => "DB_Modbus_Holding_Register_DB".State)
      { S7_GenerateENO := "TRUE" } Move(in := "AI_PID_Bon4_SP", out1 => "DB_Modbus_Holding_Register_DB".PID_Bon4_SP)
      { S7_GenerateENO := "TRUE" } Move(in := "AI_TT3219_Bon4_Eff", out1 => "DB_Modbus_Holding_Register_DB".PID_Bon4_PV)
      { S7_GenerateENO := "TRUE" } Move(in := "AI_CV3216_Hoi_Bon4", out1 => "DB_Modbus_Holding_Register_DB".PID_Bon4_CV)
   END_RUNG
   // the same network as SCL:
   // ENO of a box is taken as its EN; it also drops when the box reports an error
   "DB_Modbus_Holding_Register_DB".State := "AI_PLC2_State";
   "DB_Modbus_Holding_Register_DB".PID_Bon4_SP := "AI_PID_Bon4_SP";
   "DB_Modbus_Holding_Register_DB".PID_Bon4_PV := "AI_TT3219_Bon4_Eff";
   "DB_Modbus_Holding_Register_DB".PID_Bon4_CV := "AI_CV3216_Hoi_Bon4";
END_REGION

REGION Network 16: Modbus TCP Server - Increment Heartbeat
   RUNG wire#powerrail
      Contact( "AI_Clock_1Hz" )
      { S7_Templates := "SrcType := Int"; S7_GenerateENO := "TRUE" } Add(in1 := "DB_Modbus_Holding_Register_DB".Heartbeat_Server, in2 := 1, out => "DB_Modbus_Holding_Register_DB".Heartbeat_Server)
   END_RUNG
   // the same network as SCL:
   IF "AI_Clock_1Hz" THEN
       "DB_Modbus_Holding_Register_DB".Heartbeat_Server := "DB_Modbus_Holding_Register_DB".Heartbeat_Server + 1;
   END_IF;
END_REGION

REGION Network 17: Handshake Server - Update AckSeq and Last_CmdSeq
   RUNG wire#powerrail
      { S7_GenerateENO := "TRUE" } Move(in := "DB_Modbus_Holding_Register_DB".CmdSeq, out1 => "DB_Modbus_Holding_Register_DB".AckSeq)
      { S7_GenerateENO := "TRUE" } Move(in := "DB_Modbus_Holding_Register_DB".CmdSeq, out1 => "AI_PLC2_Last_CmdSeq")
   END_RUNG
   // the same network as SCL:
   // ENO of a box is taken as its EN; it also drops when the box reports an error
   "DB_Modbus_Holding_Register_DB".AckSeq := "DB_Modbus_Holding_Register_DB".CmdSeq;
   "AI_PLC2_Last_CmdSeq" := "DB_Modbus_Holding_Register_DB".CmdSeq;
END_REGION
END_ORGANIZATION_BLOCK

FUNCTION "FC_Init_Default_Recipe_PLC2" : Void   // FC51, LAD
{ S7_Optimized_Access := 'TRUE' }
VERSION : 0.1
// stored: AutoNumber true, IsIECCheckEnabled false, SetENOAutomatically false, UDAEnableTagReadback false
BEGIN

REGION Network 1: Kích hoạt nạp recipe mặc định lần đầu scan PLC2
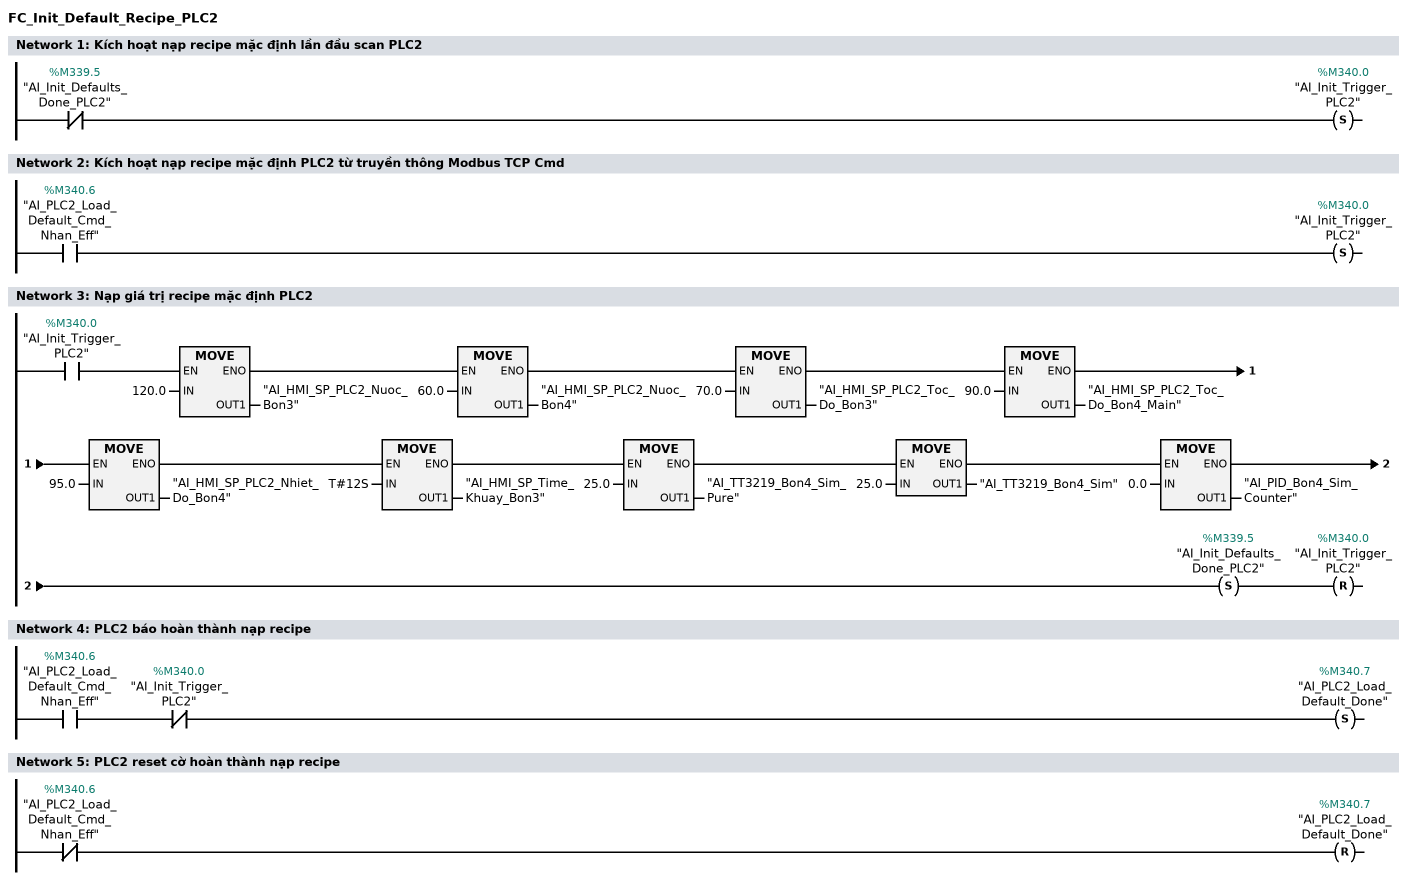
   RUNG wire#powerrail
      I_Contact( "AI_Init_Defaults_Done_PLC2" )
      S_Coil( "AI_Init_Trigger_PLC2" )
   END_RUNG
   // the same network as SCL:
   IF NOT "AI_Init_Defaults_Done_PLC2" THEN "AI_Init_Trigger_PLC2" := TRUE; END_IF;
END_REGION

REGION Network 2: Kích hoạt nạp recipe mặc định PLC2 từ truyền thông Modbus TCP Cmd
   RUNG wire#powerrail
      Contact( "AI_PLC2_Load_Default_Cmd_Nhan_Eff" )
      S_Coil( "AI_Init_Trigger_PLC2" )
   END_RUNG
   // the same network as SCL:
   IF "AI_PLC2_Load_Default_Cmd_Nhan_Eff" THEN "AI_Init_Trigger_PLC2" := TRUE; END_IF;
END_REGION

REGION Network 3: Nạp giá trị recipe mặc định PLC2
   RUNG wire#powerrail
      Contact( "AI_Init_Trigger_PLC2" )
      { S7_GenerateENO := "TRUE" } Move(in := 120.0, out1 => "AI_HMI_SP_PLC2_Nuoc_Bon3")
      { S7_GenerateENO := "TRUE" } Move(in := 60.0, out1 => "AI_HMI_SP_PLC2_Nuoc_Bon4")
      { S7_GenerateENO := "TRUE" } Move(in := 70.0, out1 => "AI_HMI_SP_PLC2_Toc_Do_Bon3")
      { S7_GenerateENO := "TRUE" } Move(in := 90.0, out1 => "AI_HMI_SP_PLC2_Toc_Do_Bon4_Main")
      { S7_GenerateENO := "TRUE" } Move(in := 95.0, out1 => "AI_HMI_SP_PLC2_Nhiet_Do_Bon4")
      { S7_GenerateENO := "TRUE" } Move(in := T#12S, out1 => "AI_HMI_SP_Time_Khuay_Bon3")
      { S7_GenerateENO := "TRUE" } Move(in := 25.0, out1 => "AI_TT3219_Bon4_Sim_Pure")
      { S7_GenerateENO := "TRUE" } Move(in := 25.0, out1 => "AI_TT3219_Bon4_Sim")
      { S7_GenerateENO := "TRUE" } Move(in := 0.0, out1 => "AI_PID_Bon4_Sim_Counter")
      S_Coil( "AI_Init_Defaults_Done_PLC2" )
      R_Coil( "AI_Init_Trigger_PLC2" )
   END_RUNG
   // the same network as SCL:
   // ENO of a box is taken as its EN; it also drops when the box reports an error
   IF "AI_Init_Trigger_PLC2" THEN
       "AI_HMI_SP_PLC2_Nuoc_Bon3" := 120.0;
       "AI_HMI_SP_PLC2_Nuoc_Bon4" := 60.0;
       "AI_HMI_SP_PLC2_Toc_Do_Bon3" := 70.0;
       "AI_HMI_SP_PLC2_Toc_Do_Bon4_Main" := 90.0;
       "AI_HMI_SP_PLC2_Nhiet_Do_Bon4" := 95.0;
       "AI_HMI_SP_Time_Khuay_Bon3" := T#12S;
       "AI_TT3219_Bon4_Sim_Pure" := 25.0;
       "AI_TT3219_Bon4_Sim" := 25.0;
       "AI_PID_Bon4_Sim_Counter" := 0.0;
       "AI_Init_Defaults_Done_PLC2" := TRUE;
       "AI_Init_Trigger_PLC2" := FALSE;
   END_IF;
END_REGION

REGION Network 4: PLC2 báo hoàn thành nạp recipe
   RUNG wire#powerrail
      Contact( "AI_PLC2_Load_Default_Cmd_Nhan_Eff" )
      I_Contact( "AI_Init_Trigger_PLC2" )
      S_Coil( "AI_PLC2_Load_Default_Done" )
   END_RUNG
   // the same network as SCL:
   IF "AI_PLC2_Load_Default_Cmd_Nhan_Eff" AND NOT "AI_Init_Trigger_PLC2" THEN
       "AI_PLC2_Load_Default_Done" := TRUE;
   END_IF;
END_REGION

REGION Network 5: PLC2 reset cờ hoàn thành nạp recipe
   RUNG wire#powerrail
      I_Contact( "AI_PLC2_Load_Default_Cmd_Nhan_Eff" )
      R_Coil( "AI_PLC2_Load_Default_Done" )
   END_RUNG
   // the same network as SCL:
   IF NOT "AI_PLC2_Load_Default_Cmd_Nhan_Eff" THEN "AI_PLC2_Load_Default_Done" := FALSE; END_IF;
END_REGION
END_FUNCTION

FUNCTION "FC_PLC2_Mixing" : Void   // FC20, LAD
{ S7_Optimized_Access := 'TRUE' }
VERSION : 0.1
// stored: AutoNumber true, IsIECCheckEnabled false, SetENOAutomatically false, UDAEnableTagReadback false
BEGIN

REGION Network 1: Khóa nút nhấn Start HMI qua Run Enable PLC2
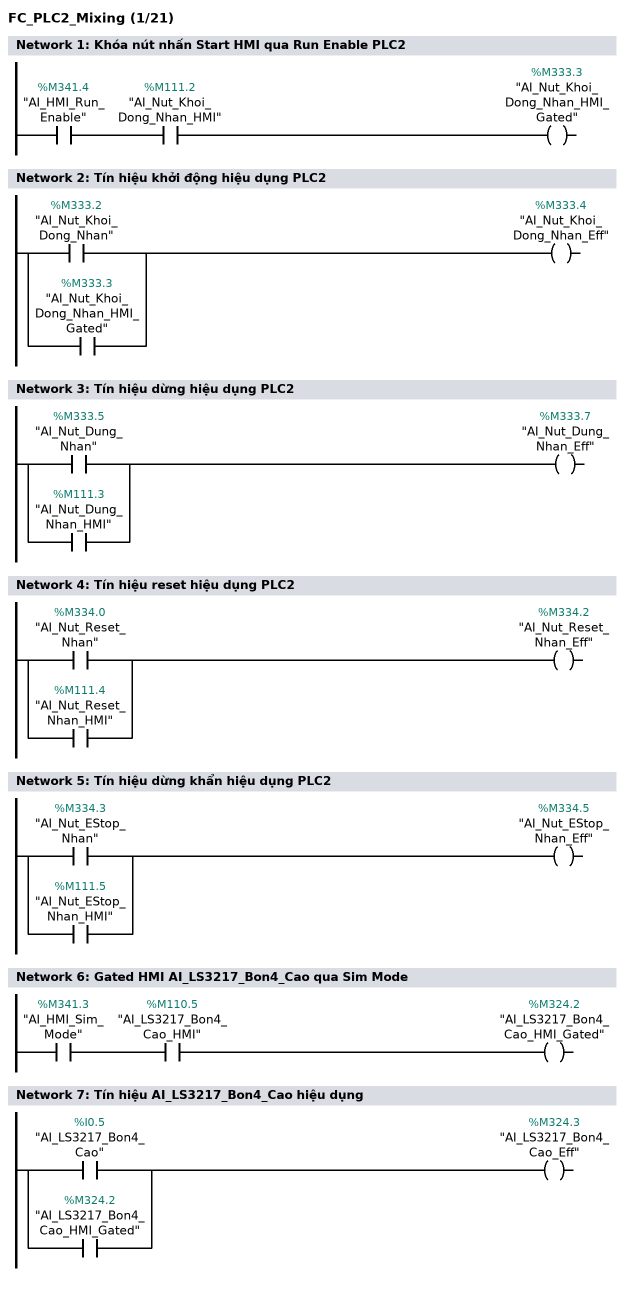
   RUNG wire#powerrail
      Contact( "AI_HMI_Run_Enable" )
      Contact( "AI_Nut_Khoi_Dong_Nhan_HMI" )
      Coil( "AI_Nut_Khoi_Dong_Nhan_HMI_Gated" )
   END_RUNG
   // the same network as SCL:
   "AI_Nut_Khoi_Dong_Nhan_HMI_Gated" := "AI_HMI_Run_Enable" AND "AI_Nut_Khoi_Dong_Nhan_HMI";
END_REGION

REGION Network 2: Tín hiệu khởi động hiệu dụng PLC2
   RUNG wire#powerrail
      Contact( "AI_Nut_Khoi_Dong_Nhan" )
      wire#w1
      Coil( "AI_Nut_Khoi_Dong_Nhan_Eff" )
   END_RUNG
   RUNG wire#powerrail
      Contact( "AI_Nut_Khoi_Dong_Nhan_HMI_Gated" )
   END_RUNG wire#w1
   // the same network as SCL:
   "AI_Nut_Khoi_Dong_Nhan_Eff" := "AI_Nut_Khoi_Dong_Nhan" OR "AI_Nut_Khoi_Dong_Nhan_HMI_Gated";
END_REGION

REGION Network 3: Tín hiệu dừng hiệu dụng PLC2
   RUNG wire#powerrail
      Contact( "AI_Nut_Dung_Nhan" )
      wire#w1
      Coil( "AI_Nut_Dung_Nhan_Eff" )
   END_RUNG
   RUNG wire#powerrail
      Contact( "AI_Nut_Dung_Nhan_HMI" )
   END_RUNG wire#w1
   // the same network as SCL:
   "AI_Nut_Dung_Nhan_Eff" := "AI_Nut_Dung_Nhan" OR "AI_Nut_Dung_Nhan_HMI";
END_REGION

REGION Network 4: Tín hiệu reset hiệu dụng PLC2
   RUNG wire#powerrail
      Contact( "AI_Nut_Reset_Nhan" )
      wire#w1
      Coil( "AI_Nut_Reset_Nhan_Eff" )
   END_RUNG
   RUNG wire#powerrail
      Contact( "AI_Nut_Reset_Nhan_HMI" )
   END_RUNG wire#w1
   // the same network as SCL:
   "AI_Nut_Reset_Nhan_Eff" := "AI_Nut_Reset_Nhan" OR "AI_Nut_Reset_Nhan_HMI";
END_REGION

REGION Network 5: Tín hiệu dừng khẩn hiệu dụng PLC2
   RUNG wire#powerrail
      Contact( "AI_Nut_EStop_Nhan" )
      wire#w1
      Coil( "AI_Nut_EStop_Nhan_Eff" )
   END_RUNG
   RUNG wire#powerrail
      Contact( "AI_Nut_EStop_Nhan_HMI" )
   END_RUNG wire#w1
   // the same network as SCL:
   "AI_Nut_EStop_Nhan_Eff" := "AI_Nut_EStop_Nhan" OR "AI_Nut_EStop_Nhan_HMI";
END_REGION

REGION Network 6: Gated HMI AI_LS3217_Bon4_Cao qua Sim Mode
   RUNG wire#powerrail
      Contact( "AI_HMI_Sim_Mode" )
      Contact( "AI_LS3217_Bon4_Cao_HMI" )
      Coil( "AI_LS3217_Bon4_Cao_HMI_Gated" )
   END_RUNG
   // the same network as SCL:
   "AI_LS3217_Bon4_Cao_HMI_Gated" := "AI_HMI_Sim_Mode" AND "AI_LS3217_Bon4_Cao_HMI";
END_REGION

REGION Network 7: Tín hiệu AI_LS3217_Bon4_Cao hiệu dụng
   RUNG wire#powerrail
      Contact( "AI_LS3217_Bon4_Cao" )
      wire#w1
      Coil( "AI_LS3217_Bon4_Cao_Eff" )
   END_RUNG
   RUNG wire#powerrail
      Contact( "AI_LS3217_Bon4_Cao_HMI_Gated" )
   END_RUNG wire#w1
   // the same network as SCL:
   "AI_LS3217_Bon4_Cao_Eff" := "AI_LS3217_Bon4_Cao" OR "AI_LS3217_Bon4_Cao_HMI_Gated";
END_REGION

REGION Network 8: Gated HMI AI_Pump3265_Chuyen_Nhanh2_Cmd_Nhan qua Sim Mode
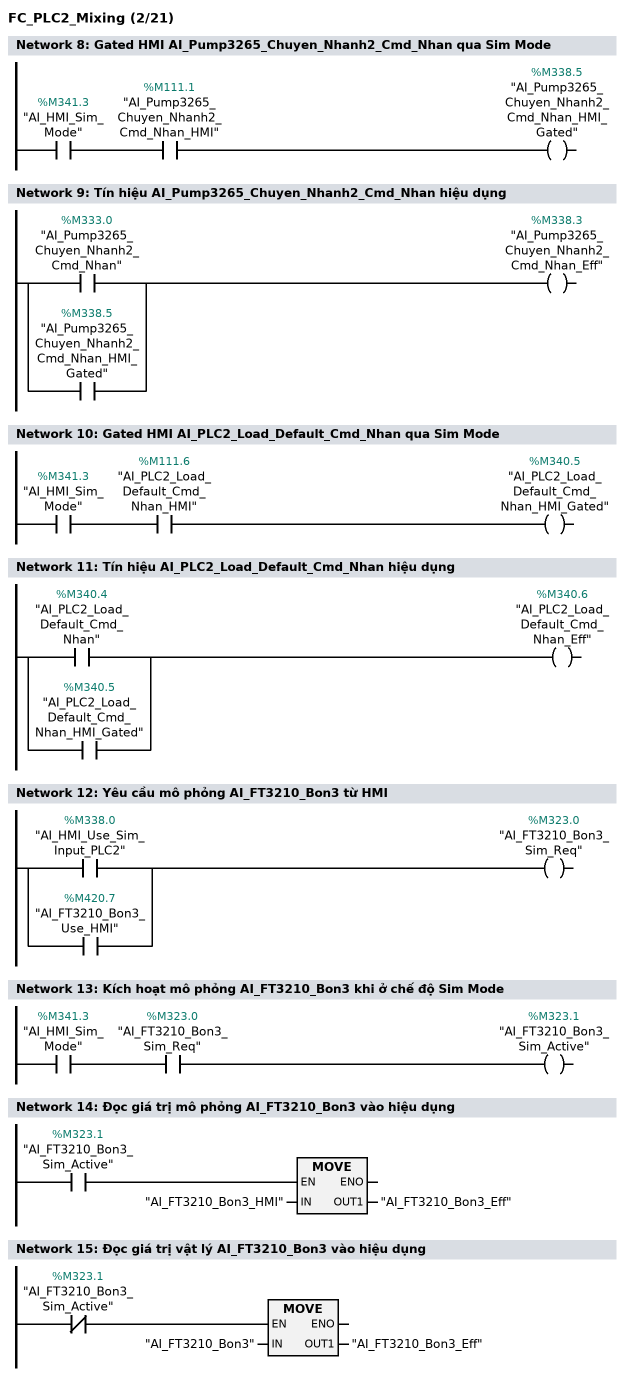
   RUNG wire#powerrail
      Contact( "AI_HMI_Sim_Mode" )
      Contact( "AI_Pump3265_Chuyen_Nhanh2_Cmd_Nhan_HMI" )
      Coil( "AI_Pump3265_Chuyen_Nhanh2_Cmd_Nhan_HMI_Gated" )
   END_RUNG
   // the same network as SCL:
   "AI_Pump3265_Chuyen_Nhanh2_Cmd_Nhan_HMI_Gated" := "AI_HMI_Sim_Mode" AND "AI_Pump3265_Chuyen_Nhanh2_Cmd_Nhan_HMI";
END_REGION

REGION Network 9: Tín hiệu AI_Pump3265_Chuyen_Nhanh2_Cmd_Nhan hiệu dụng
   RUNG wire#powerrail
      Contact( "AI_Pump3265_Chuyen_Nhanh2_Cmd_Nhan" )
      wire#w1
      Coil( "AI_Pump3265_Chuyen_Nhanh2_Cmd_Nhan_Eff" )
   END_RUNG
   RUNG wire#powerrail
      Contact( "AI_Pump3265_Chuyen_Nhanh2_Cmd_Nhan_HMI_Gated" )
   END_RUNG wire#w1
   // the same network as SCL:
   "AI_Pump3265_Chuyen_Nhanh2_Cmd_Nhan_Eff" := "AI_Pump3265_Chuyen_Nhanh2_Cmd_Nhan" OR "AI_Pump3265_Chuyen_Nhanh2_Cmd_Nhan_HMI_Gated";
END_REGION

REGION Network 10: Gated HMI AI_PLC2_Load_Default_Cmd_Nhan qua Sim Mode
   RUNG wire#powerrail
      Contact( "AI_HMI_Sim_Mode" )
      Contact( "AI_PLC2_Load_Default_Cmd_Nhan_HMI" )
      Coil( "AI_PLC2_Load_Default_Cmd_Nhan_HMI_Gated" )
   END_RUNG
   // the same network as SCL:
   "AI_PLC2_Load_Default_Cmd_Nhan_HMI_Gated" := "AI_HMI_Sim_Mode" AND "AI_PLC2_Load_Default_Cmd_Nhan_HMI";
END_REGION

REGION Network 11: Tín hiệu AI_PLC2_Load_Default_Cmd_Nhan hiệu dụng
   RUNG wire#powerrail
      Contact( "AI_PLC2_Load_Default_Cmd_Nhan" )
      wire#w1
      Coil( "AI_PLC2_Load_Default_Cmd_Nhan_Eff" )
   END_RUNG
   RUNG wire#powerrail
      Contact( "AI_PLC2_Load_Default_Cmd_Nhan_HMI_Gated" )
   END_RUNG wire#w1
   // the same network as SCL:
   "AI_PLC2_Load_Default_Cmd_Nhan_Eff" := "AI_PLC2_Load_Default_Cmd_Nhan" OR "AI_PLC2_Load_Default_Cmd_Nhan_HMI_Gated";
END_REGION

REGION Network 12: Yêu cầu mô phỏng AI_FT3210_Bon3 từ HMI
   RUNG wire#powerrail
      Contact( "AI_HMI_Use_Sim_Input_PLC2" )
      wire#w1
      Coil( "AI_FT3210_Bon3_Sim_Req" )
   END_RUNG
   RUNG wire#powerrail
      Contact( "AI_FT3210_Bon3_Use_HMI" )
   END_RUNG wire#w1
   // the same network as SCL:
   "AI_FT3210_Bon3_Sim_Req" := "AI_HMI_Use_Sim_Input_PLC2" OR "AI_FT3210_Bon3_Use_HMI";
END_REGION

REGION Network 13: Kích hoạt mô phỏng AI_FT3210_Bon3 khi ở chế độ Sim Mode
   RUNG wire#powerrail
      Contact( "AI_HMI_Sim_Mode" )
      Contact( "AI_FT3210_Bon3_Sim_Req" )
      Coil( "AI_FT3210_Bon3_Sim_Active" )
   END_RUNG
   // the same network as SCL:
   "AI_FT3210_Bon3_Sim_Active" := "AI_HMI_Sim_Mode" AND "AI_FT3210_Bon3_Sim_Req";
END_REGION

REGION Network 14: Đọc giá trị mô phỏng AI_FT3210_Bon3 vào hiệu dụng
   RUNG wire#powerrail
      Contact( "AI_FT3210_Bon3_Sim_Active" )
      { S7_GenerateENO := "TRUE" } Move(in := "AI_FT3210_Bon3_HMI", out1 => "AI_FT3210_Bon3_Eff")
   END_RUNG
   // the same network as SCL:
   IF "AI_FT3210_Bon3_Sim_Active" THEN "AI_FT3210_Bon3_Eff" := "AI_FT3210_Bon3_HMI"; END_IF;
END_REGION

REGION Network 15: Đọc giá trị vật lý AI_FT3210_Bon3 vào hiệu dụng
   RUNG wire#powerrail
      I_Contact( "AI_FT3210_Bon3_Sim_Active" )
      { S7_GenerateENO := "TRUE" } Move(in := "AI_FT3210_Bon3", out1 => "AI_FT3210_Bon3_Eff")
   END_RUNG
   // the same network as SCL:
   IF NOT "AI_FT3210_Bon3_Sim_Active" THEN "AI_FT3210_Bon3_Eff" := "AI_FT3210_Bon3"; END_IF;
END_REGION

REGION Network 16: Yêu cầu mô phỏng AI_LT3213_Bon3 từ HMI
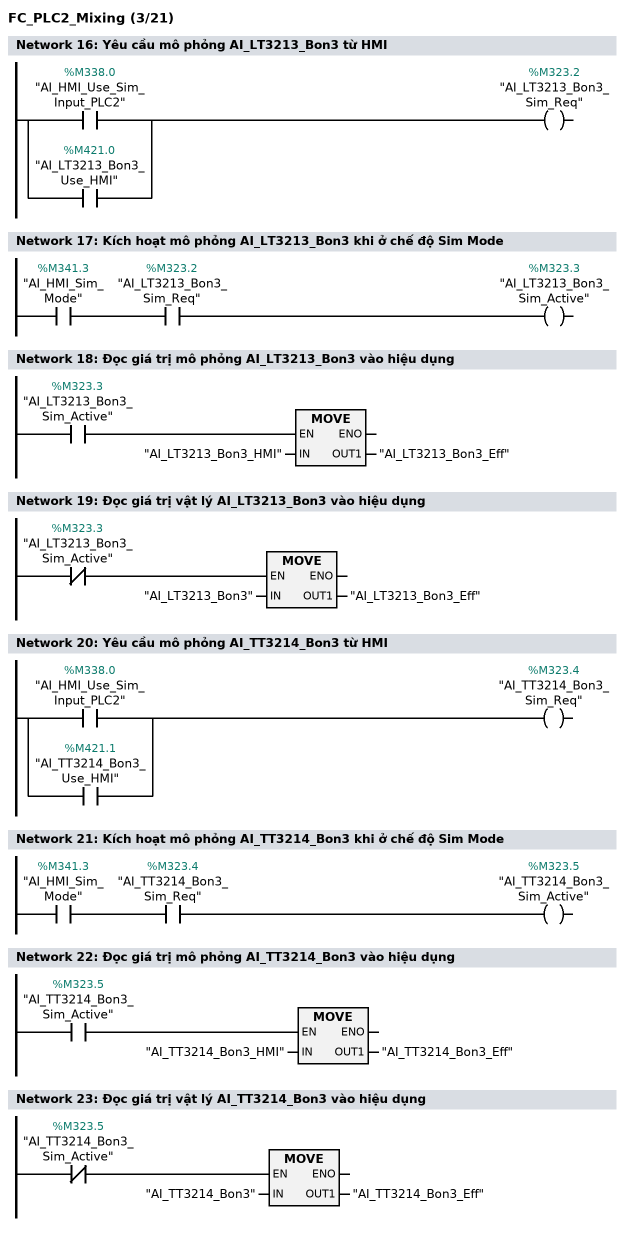
   RUNG wire#powerrail
      Contact( "AI_HMI_Use_Sim_Input_PLC2" )
      wire#w1
      Coil( "AI_LT3213_Bon3_Sim_Req" )
   END_RUNG
   RUNG wire#powerrail
      Contact( "AI_LT3213_Bon3_Use_HMI" )
   END_RUNG wire#w1
   // the same network as SCL:
   "AI_LT3213_Bon3_Sim_Req" := "AI_HMI_Use_Sim_Input_PLC2" OR "AI_LT3213_Bon3_Use_HMI";
END_REGION

REGION Network 17: Kích hoạt mô phỏng AI_LT3213_Bon3 khi ở chế độ Sim Mode
   RUNG wire#powerrail
      Contact( "AI_HMI_Sim_Mode" )
      Contact( "AI_LT3213_Bon3_Sim_Req" )
      Coil( "AI_LT3213_Bon3_Sim_Active" )
   END_RUNG
   // the same network as SCL:
   "AI_LT3213_Bon3_Sim_Active" := "AI_HMI_Sim_Mode" AND "AI_LT3213_Bon3_Sim_Req";
END_REGION

REGION Network 18: Đọc giá trị mô phỏng AI_LT3213_Bon3 vào hiệu dụng
   RUNG wire#powerrail
      Contact( "AI_LT3213_Bon3_Sim_Active" )
      { S7_GenerateENO := "TRUE" } Move(in := "AI_LT3213_Bon3_HMI", out1 => "AI_LT3213_Bon3_Eff")
   END_RUNG
   // the same network as SCL:
   IF "AI_LT3213_Bon3_Sim_Active" THEN "AI_LT3213_Bon3_Eff" := "AI_LT3213_Bon3_HMI"; END_IF;
END_REGION

REGION Network 19: Đọc giá trị vật lý AI_LT3213_Bon3 vào hiệu dụng
   RUNG wire#powerrail
      I_Contact( "AI_LT3213_Bon3_Sim_Active" )
      { S7_GenerateENO := "TRUE" } Move(in := "AI_LT3213_Bon3", out1 => "AI_LT3213_Bon3_Eff")
   END_RUNG
   // the same network as SCL:
   IF NOT "AI_LT3213_Bon3_Sim_Active" THEN "AI_LT3213_Bon3_Eff" := "AI_LT3213_Bon3"; END_IF;
END_REGION

REGION Network 20: Yêu cầu mô phỏng AI_TT3214_Bon3 từ HMI
   RUNG wire#powerrail
      Contact( "AI_HMI_Use_Sim_Input_PLC2" )
      wire#w1
      Coil( "AI_TT3214_Bon3_Sim_Req" )
   END_RUNG
   RUNG wire#powerrail
      Contact( "AI_TT3214_Bon3_Use_HMI" )
   END_RUNG wire#w1
   // the same network as SCL:
   "AI_TT3214_Bon3_Sim_Req" := "AI_HMI_Use_Sim_Input_PLC2" OR "AI_TT3214_Bon3_Use_HMI";
END_REGION

REGION Network 21: Kích hoạt mô phỏng AI_TT3214_Bon3 khi ở chế độ Sim Mode
   RUNG wire#powerrail
      Contact( "AI_HMI_Sim_Mode" )
      Contact( "AI_TT3214_Bon3_Sim_Req" )
      Coil( "AI_TT3214_Bon3_Sim_Active" )
   END_RUNG
   // the same network as SCL:
   "AI_TT3214_Bon3_Sim_Active" := "AI_HMI_Sim_Mode" AND "AI_TT3214_Bon3_Sim_Req";
END_REGION

REGION Network 22: Đọc giá trị mô phỏng AI_TT3214_Bon3 vào hiệu dụng
   RUNG wire#powerrail
      Contact( "AI_TT3214_Bon3_Sim_Active" )
      { S7_GenerateENO := "TRUE" } Move(in := "AI_TT3214_Bon3_HMI", out1 => "AI_TT3214_Bon3_Eff")
   END_RUNG
   // the same network as SCL:
   IF "AI_TT3214_Bon3_Sim_Active" THEN "AI_TT3214_Bon3_Eff" := "AI_TT3214_Bon3_HMI"; END_IF;
END_REGION

REGION Network 23: Đọc giá trị vật lý AI_TT3214_Bon3 vào hiệu dụng
   RUNG wire#powerrail
      I_Contact( "AI_TT3214_Bon3_Sim_Active" )
      { S7_GenerateENO := "TRUE" } Move(in := "AI_TT3214_Bon3", out1 => "AI_TT3214_Bon3_Eff")
   END_RUNG
   // the same network as SCL:
   IF NOT "AI_TT3214_Bon3_Sim_Active" THEN "AI_TT3214_Bon3_Eff" := "AI_TT3214_Bon3"; END_IF;
END_REGION

REGION Network 24: Yêu cầu mô phỏng AI_FT3215_Bon4 từ HMI
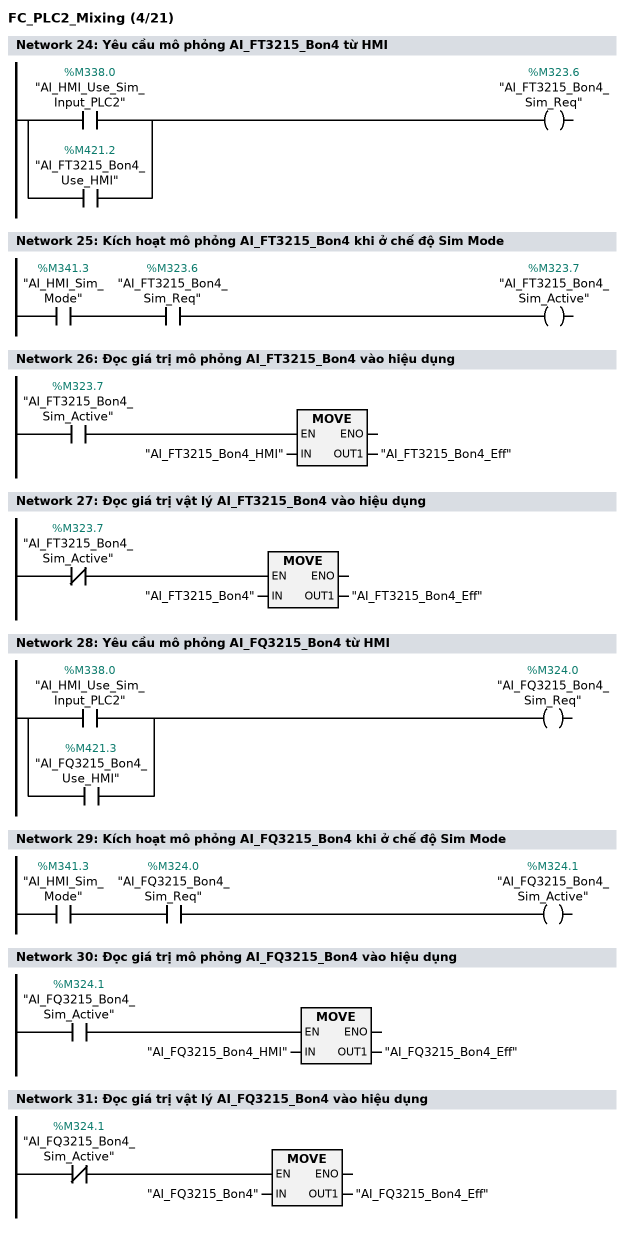
   RUNG wire#powerrail
      Contact( "AI_HMI_Use_Sim_Input_PLC2" )
      wire#w1
      Coil( "AI_FT3215_Bon4_Sim_Req" )
   END_RUNG
   RUNG wire#powerrail
      Contact( "AI_FT3215_Bon4_Use_HMI" )
   END_RUNG wire#w1
   // the same network as SCL:
   "AI_FT3215_Bon4_Sim_Req" := "AI_HMI_Use_Sim_Input_PLC2" OR "AI_FT3215_Bon4_Use_HMI";
END_REGION

REGION Network 25: Kích hoạt mô phỏng AI_FT3215_Bon4 khi ở chế độ Sim Mode
   RUNG wire#powerrail
      Contact( "AI_HMI_Sim_Mode" )
      Contact( "AI_FT3215_Bon4_Sim_Req" )
      Coil( "AI_FT3215_Bon4_Sim_Active" )
   END_RUNG
   // the same network as SCL:
   "AI_FT3215_Bon4_Sim_Active" := "AI_HMI_Sim_Mode" AND "AI_FT3215_Bon4_Sim_Req";
END_REGION

REGION Network 26: Đọc giá trị mô phỏng AI_FT3215_Bon4 vào hiệu dụng
   RUNG wire#powerrail
      Contact( "AI_FT3215_Bon4_Sim_Active" )
      { S7_GenerateENO := "TRUE" } Move(in := "AI_FT3215_Bon4_HMI", out1 => "AI_FT3215_Bon4_Eff")
   END_RUNG
   // the same network as SCL:
   IF "AI_FT3215_Bon4_Sim_Active" THEN "AI_FT3215_Bon4_Eff" := "AI_FT3215_Bon4_HMI"; END_IF;
END_REGION

REGION Network 27: Đọc giá trị vật lý AI_FT3215_Bon4 vào hiệu dụng
   RUNG wire#powerrail
      I_Contact( "AI_FT3215_Bon4_Sim_Active" )
      { S7_GenerateENO := "TRUE" } Move(in := "AI_FT3215_Bon4", out1 => "AI_FT3215_Bon4_Eff")
   END_RUNG
   // the same network as SCL:
   IF NOT "AI_FT3215_Bon4_Sim_Active" THEN "AI_FT3215_Bon4_Eff" := "AI_FT3215_Bon4"; END_IF;
END_REGION

REGION Network 28: Yêu cầu mô phỏng AI_FQ3215_Bon4 từ HMI
   RUNG wire#powerrail
      Contact( "AI_HMI_Use_Sim_Input_PLC2" )
      wire#w1
      Coil( "AI_FQ3215_Bon4_Sim_Req" )
   END_RUNG
   RUNG wire#powerrail
      Contact( "AI_FQ3215_Bon4_Use_HMI" )
   END_RUNG wire#w1
   // the same network as SCL:
   "AI_FQ3215_Bon4_Sim_Req" := "AI_HMI_Use_Sim_Input_PLC2" OR "AI_FQ3215_Bon4_Use_HMI";
END_REGION

REGION Network 29: Kích hoạt mô phỏng AI_FQ3215_Bon4 khi ở chế độ Sim Mode
   RUNG wire#powerrail
      Contact( "AI_HMI_Sim_Mode" )
      Contact( "AI_FQ3215_Bon4_Sim_Req" )
      Coil( "AI_FQ3215_Bon4_Sim_Active" )
   END_RUNG
   // the same network as SCL:
   "AI_FQ3215_Bon4_Sim_Active" := "AI_HMI_Sim_Mode" AND "AI_FQ3215_Bon4_Sim_Req";
END_REGION

REGION Network 30: Đọc giá trị mô phỏng AI_FQ3215_Bon4 vào hiệu dụng
   RUNG wire#powerrail
      Contact( "AI_FQ3215_Bon4_Sim_Active" )
      { S7_GenerateENO := "TRUE" } Move(in := "AI_FQ3215_Bon4_HMI", out1 => "AI_FQ3215_Bon4_Eff")
   END_RUNG
   // the same network as SCL:
   IF "AI_FQ3215_Bon4_Sim_Active" THEN "AI_FQ3215_Bon4_Eff" := "AI_FQ3215_Bon4_HMI"; END_IF;
END_REGION

REGION Network 31: Đọc giá trị vật lý AI_FQ3215_Bon4 vào hiệu dụng
   RUNG wire#powerrail
      I_Contact( "AI_FQ3215_Bon4_Sim_Active" )
      { S7_GenerateENO := "TRUE" } Move(in := "AI_FQ3215_Bon4", out1 => "AI_FQ3215_Bon4_Eff")
   END_RUNG
   // the same network as SCL:
   IF NOT "AI_FQ3215_Bon4_Sim_Active" THEN "AI_FQ3215_Bon4_Eff" := "AI_FQ3215_Bon4"; END_IF;
END_REGION

REGION Network 32: Yêu cầu mô phỏng AI_LT3218_Bon4 từ HMI
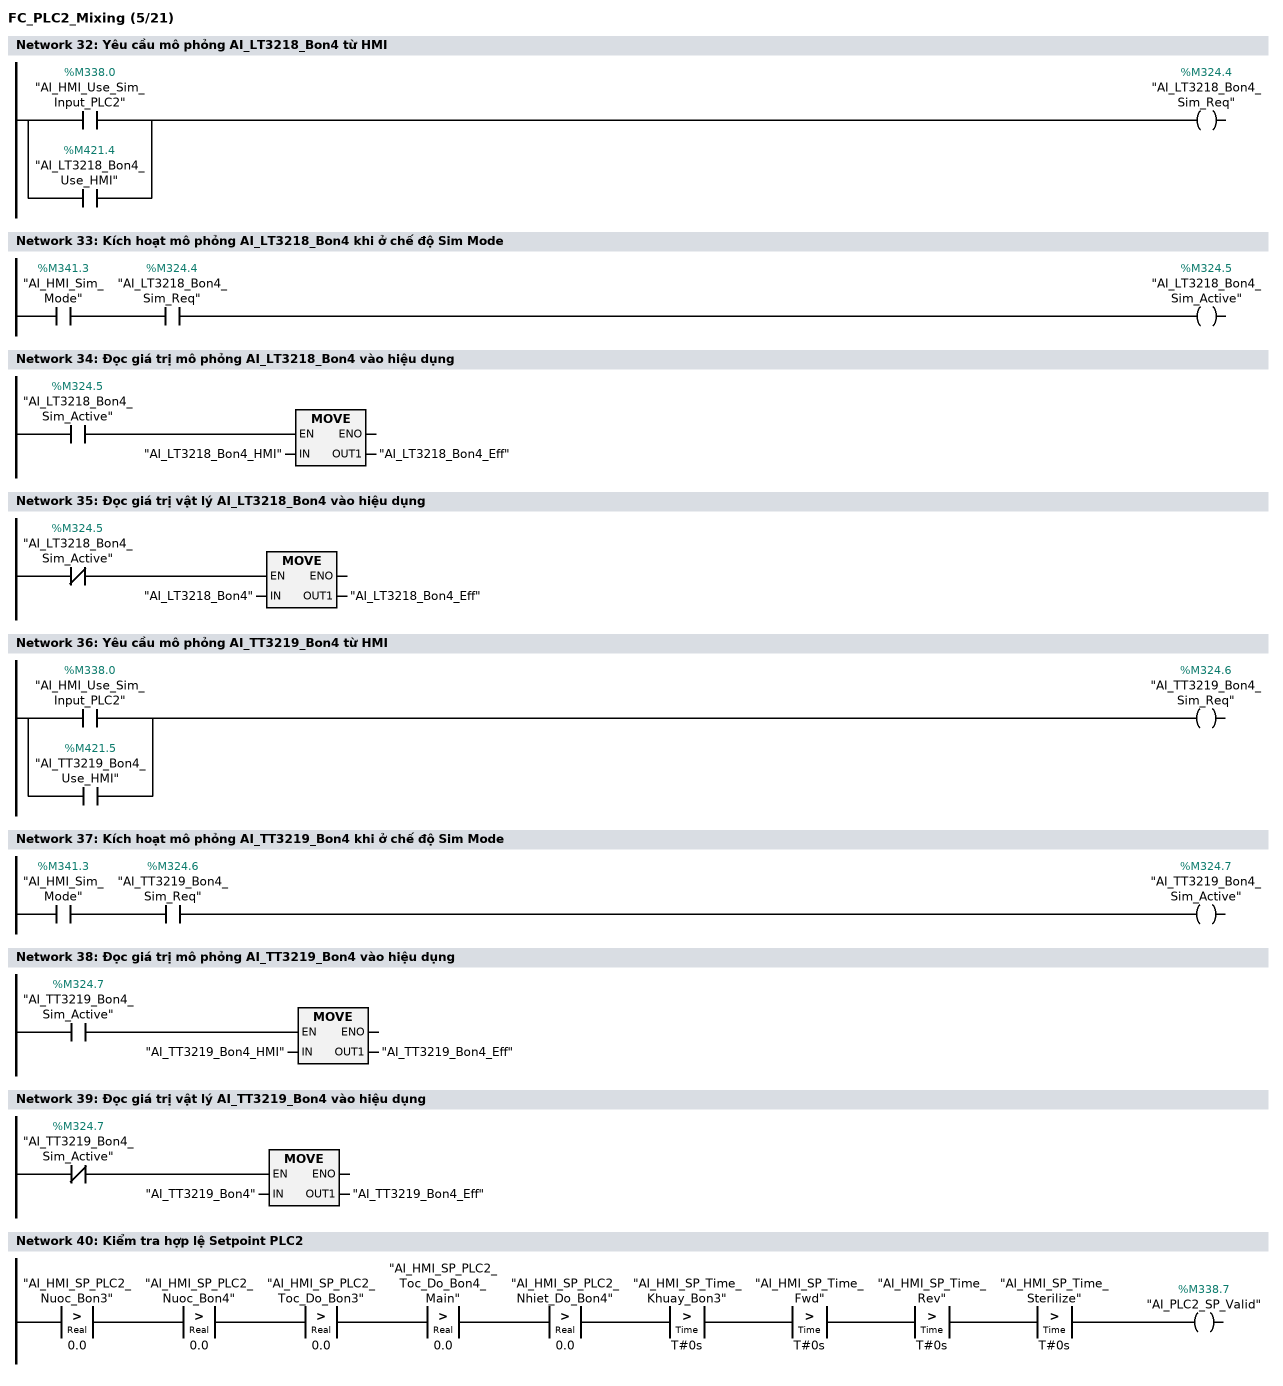
   RUNG wire#powerrail
      Contact( "AI_HMI_Use_Sim_Input_PLC2" )
      wire#w1
      Coil( "AI_LT3218_Bon4_Sim_Req" )
   END_RUNG
   RUNG wire#powerrail
      Contact( "AI_LT3218_Bon4_Use_HMI" )
   END_RUNG wire#w1
   // the same network as SCL:
   "AI_LT3218_Bon4_Sim_Req" := "AI_HMI_Use_Sim_Input_PLC2" OR "AI_LT3218_Bon4_Use_HMI";
END_REGION

REGION Network 33: Kích hoạt mô phỏng AI_LT3218_Bon4 khi ở chế độ Sim Mode
   RUNG wire#powerrail
      Contact( "AI_HMI_Sim_Mode" )
      Contact( "AI_LT3218_Bon4_Sim_Req" )
      Coil( "AI_LT3218_Bon4_Sim_Active" )
   END_RUNG
   // the same network as SCL:
   "AI_LT3218_Bon4_Sim_Active" := "AI_HMI_Sim_Mode" AND "AI_LT3218_Bon4_Sim_Req";
END_REGION

REGION Network 34: Đọc giá trị mô phỏng AI_LT3218_Bon4 vào hiệu dụng
   RUNG wire#powerrail
      Contact( "AI_LT3218_Bon4_Sim_Active" )
      { S7_GenerateENO := "TRUE" } Move(in := "AI_LT3218_Bon4_HMI", out1 => "AI_LT3218_Bon4_Eff")
   END_RUNG
   // the same network as SCL:
   IF "AI_LT3218_Bon4_Sim_Active" THEN "AI_LT3218_Bon4_Eff" := "AI_LT3218_Bon4_HMI"; END_IF;
END_REGION

REGION Network 35: Đọc giá trị vật lý AI_LT3218_Bon4 vào hiệu dụng
   RUNG wire#powerrail
      I_Contact( "AI_LT3218_Bon4_Sim_Active" )
      { S7_GenerateENO := "TRUE" } Move(in := "AI_LT3218_Bon4", out1 => "AI_LT3218_Bon4_Eff")
   END_RUNG
   // the same network as SCL:
   IF NOT "AI_LT3218_Bon4_Sim_Active" THEN "AI_LT3218_Bon4_Eff" := "AI_LT3218_Bon4"; END_IF;
END_REGION

REGION Network 36: Yêu cầu mô phỏng AI_TT3219_Bon4 từ HMI
   RUNG wire#powerrail
      Contact( "AI_HMI_Use_Sim_Input_PLC2" )
      wire#w1
      Coil( "AI_TT3219_Bon4_Sim_Req" )
   END_RUNG
   RUNG wire#powerrail
      Contact( "AI_TT3219_Bon4_Use_HMI" )
   END_RUNG wire#w1
   // the same network as SCL:
   "AI_TT3219_Bon4_Sim_Req" := "AI_HMI_Use_Sim_Input_PLC2" OR "AI_TT3219_Bon4_Use_HMI";
END_REGION

REGION Network 37: Kích hoạt mô phỏng AI_TT3219_Bon4 khi ở chế độ Sim Mode
   RUNG wire#powerrail
      Contact( "AI_HMI_Sim_Mode" )
      Contact( "AI_TT3219_Bon4_Sim_Req" )
      Coil( "AI_TT3219_Bon4_Sim_Active" )
   END_RUNG
   // the same network as SCL:
   "AI_TT3219_Bon4_Sim_Active" := "AI_HMI_Sim_Mode" AND "AI_TT3219_Bon4_Sim_Req";
END_REGION

REGION Network 38: Đọc giá trị mô phỏng AI_TT3219_Bon4 vào hiệu dụng
   RUNG wire#powerrail
      Contact( "AI_TT3219_Bon4_Sim_Active" )
      { S7_GenerateENO := "TRUE" } Move(in := "AI_TT3219_Bon4_HMI", out1 => "AI_TT3219_Bon4_Eff")
   END_RUNG
   // the same network as SCL:
   IF "AI_TT3219_Bon4_Sim_Active" THEN "AI_TT3219_Bon4_Eff" := "AI_TT3219_Bon4_HMI"; END_IF;
END_REGION

REGION Network 39: Đọc giá trị vật lý AI_TT3219_Bon4 vào hiệu dụng
   RUNG wire#powerrail
      I_Contact( "AI_TT3219_Bon4_Sim_Active" )
      { S7_GenerateENO := "TRUE" } Move(in := "AI_TT3219_Bon4", out1 => "AI_TT3219_Bon4_Eff")
   END_RUNG
   // the same network as SCL:
   IF NOT "AI_TT3219_Bon4_Sim_Active" THEN "AI_TT3219_Bon4_Eff" := "AI_TT3219_Bon4"; END_IF;
END_REGION

REGION Network 40: Kiểm tra hợp lệ Setpoint PLC2
   RUNG wire#powerrail
      { S7_Templates := "SrcType := Real" } GT_Contact(in1 := "AI_HMI_SP_PLC2_Nuoc_Bon3", in2 := 0.0)
      { S7_Templates := "SrcType := Real" } GT_Contact(in1 := "AI_HMI_SP_PLC2_Nuoc_Bon4", in2 := 0.0)
      { S7_Templates := "SrcType := Real" } GT_Contact(in1 := "AI_HMI_SP_PLC2_Toc_Do_Bon3", in2 := 0.0)
      { S7_Templates := "SrcType := Real" } GT_Contact(in1 := "AI_HMI_SP_PLC2_Toc_Do_Bon4_Main", in2 := 0.0)
      { S7_Templates := "SrcType := Real" } GT_Contact(in1 := "AI_HMI_SP_PLC2_Nhiet_Do_Bon4", in2 := 0.0)
      { S7_Templates := "SrcType := Time" } GT_Contact(in1 := "AI_HMI_SP_Time_Khuay_Bon3", in2 := T#0s)
      { S7_Templates := "SrcType := Time" } GT_Contact(in1 := "AI_HMI_SP_Time_Fwd", in2 := T#0s)
      { S7_Templates := "SrcType := Time" } GT_Contact(in1 := "AI_HMI_SP_Time_Rev", in2 := T#0s)
      { S7_Templates := "SrcType := Time" } GT_Contact(in1 := "AI_HMI_SP_Time_Sterilize", in2 := T#0s)
      Coil( "AI_PLC2_SP_Valid" )
   END_RUNG
   // the same network as SCL:
   "AI_PLC2_SP_Valid" := ("AI_HMI_SP_PLC2_Nuoc_Bon3" > 0.0) AND ("AI_HMI_SP_PLC2_Nuoc_Bon4" > 0.0) AND ("AI_HMI_SP_PLC2_Toc_Do_Bon3" > 0.0) AND ("AI_HMI_SP_PLC2_Toc_Do_Bon4_Main" > 0.0) AND ("AI_HMI_SP_PLC2_Nhiet_Do_Bon4" > 0.0) AND ("AI_HMI_SP_Time_Khuay_Bon3" > T#0s) AND ("AI_HMI_SP_Time_Fwd" > T#0s) AND ("AI_HMI_SP_Time_Rev" > T#0s) AND ("AI_HMI_SP_Time_Sterilize" > T#0s);
END_REGION

REGION Network 41: Start PLC2 thành công từ HMI dùng chung
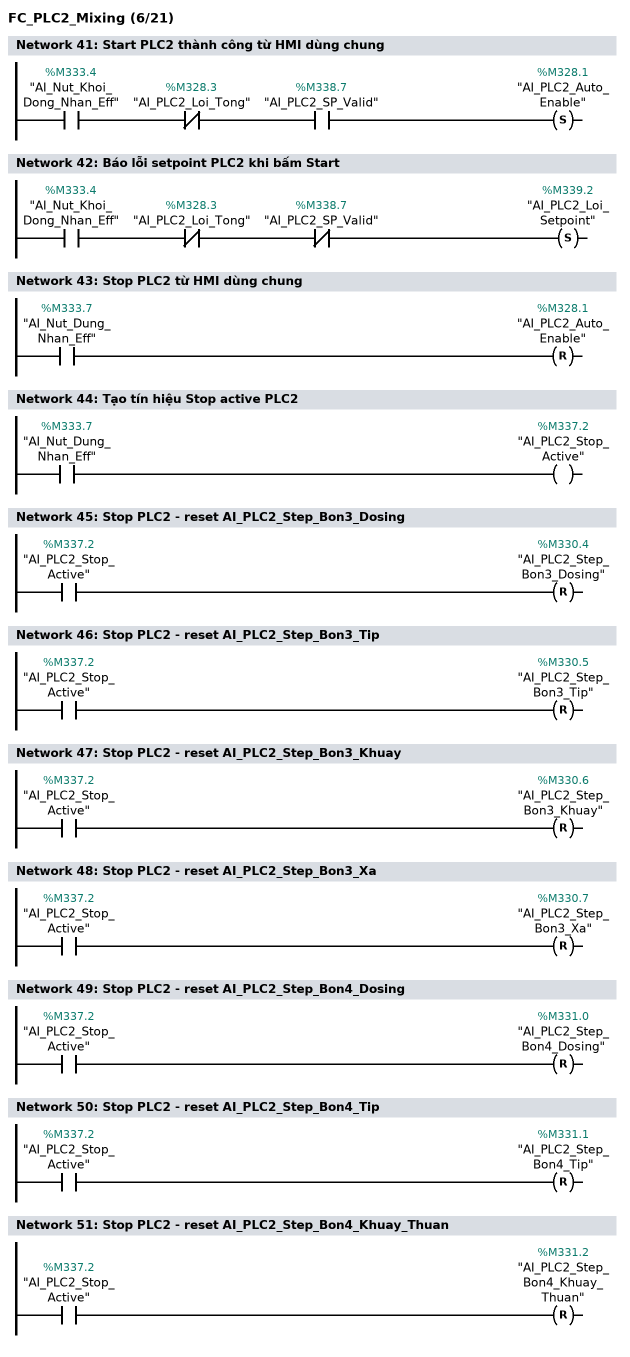
   RUNG wire#powerrail
      Contact( "AI_Nut_Khoi_Dong_Nhan_Eff" )
      I_Contact( "AI_PLC2_Loi_Tong" )
      Contact( "AI_PLC2_SP_Valid" )
      S_Coil( "AI_PLC2_Auto_Enable" )
   END_RUNG
   // the same network as SCL:
   IF "AI_Nut_Khoi_Dong_Nhan_Eff" AND NOT "AI_PLC2_Loi_Tong" AND "AI_PLC2_SP_Valid" THEN
       "AI_PLC2_Auto_Enable" := TRUE;
   END_IF;
END_REGION

REGION Network 42: Báo lỗi setpoint PLC2 khi bấm Start
   RUNG wire#powerrail
      Contact( "AI_Nut_Khoi_Dong_Nhan_Eff" )
      I_Contact( "AI_PLC2_Loi_Tong" )
      I_Contact( "AI_PLC2_SP_Valid" )
      S_Coil( "AI_PLC2_Loi_Setpoint" )
   END_RUNG
   // the same network as SCL:
   IF "AI_Nut_Khoi_Dong_Nhan_Eff" AND NOT "AI_PLC2_Loi_Tong" AND NOT "AI_PLC2_SP_Valid" THEN
       "AI_PLC2_Loi_Setpoint" := TRUE;
   END_IF;
END_REGION

REGION Network 43: Stop PLC2 từ HMI dùng chung
   RUNG wire#powerrail
      Contact( "AI_Nut_Dung_Nhan_Eff" )
      R_Coil( "AI_PLC2_Auto_Enable" )
   END_RUNG
   // the same network as SCL:
   IF "AI_Nut_Dung_Nhan_Eff" THEN "AI_PLC2_Auto_Enable" := FALSE; END_IF;
END_REGION

REGION Network 44: Tạo tín hiệu Stop active PLC2
   RUNG wire#powerrail
      Contact( "AI_Nut_Dung_Nhan_Eff" )
      Coil( "AI_PLC2_Stop_Active" )
   END_RUNG
   // the same network as SCL:
   "AI_PLC2_Stop_Active" := "AI_Nut_Dung_Nhan_Eff";
END_REGION

REGION Network 45: Stop PLC2 - reset AI_PLC2_Step_Bon3_Dosing
   RUNG wire#powerrail
      Contact( "AI_PLC2_Stop_Active" )
      R_Coil( "AI_PLC2_Step_Bon3_Dosing" )
   END_RUNG
   // the same network as SCL:
   IF "AI_PLC2_Stop_Active" THEN "AI_PLC2_Step_Bon3_Dosing" := FALSE; END_IF;
END_REGION

REGION Network 46: Stop PLC2 - reset AI_PLC2_Step_Bon3_Tip
   RUNG wire#powerrail
      Contact( "AI_PLC2_Stop_Active" )
      R_Coil( "AI_PLC2_Step_Bon3_Tip" )
   END_RUNG
   // the same network as SCL:
   IF "AI_PLC2_Stop_Active" THEN "AI_PLC2_Step_Bon3_Tip" := FALSE; END_IF;
END_REGION

REGION Network 47: Stop PLC2 - reset AI_PLC2_Step_Bon3_Khuay
   RUNG wire#powerrail
      Contact( "AI_PLC2_Stop_Active" )
      R_Coil( "AI_PLC2_Step_Bon3_Khuay" )
   END_RUNG
   // the same network as SCL:
   IF "AI_PLC2_Stop_Active" THEN "AI_PLC2_Step_Bon3_Khuay" := FALSE; END_IF;
END_REGION

REGION Network 48: Stop PLC2 - reset AI_PLC2_Step_Bon3_Xa
   RUNG wire#powerrail
      Contact( "AI_PLC2_Stop_Active" )
      R_Coil( "AI_PLC2_Step_Bon3_Xa" )
   END_RUNG
   // the same network as SCL:
   IF "AI_PLC2_Stop_Active" THEN "AI_PLC2_Step_Bon3_Xa" := FALSE; END_IF;
END_REGION

REGION Network 49: Stop PLC2 - reset AI_PLC2_Step_Bon4_Dosing
   RUNG wire#powerrail
      Contact( "AI_PLC2_Stop_Active" )
      R_Coil( "AI_PLC2_Step_Bon4_Dosing" )
   END_RUNG
   // the same network as SCL:
   IF "AI_PLC2_Stop_Active" THEN "AI_PLC2_Step_Bon4_Dosing" := FALSE; END_IF;
END_REGION

REGION Network 50: Stop PLC2 - reset AI_PLC2_Step_Bon4_Tip
   RUNG wire#powerrail
      Contact( "AI_PLC2_Stop_Active" )
      R_Coil( "AI_PLC2_Step_Bon4_Tip" )
   END_RUNG
   // the same network as SCL:
   IF "AI_PLC2_Stop_Active" THEN "AI_PLC2_Step_Bon4_Tip" := FALSE; END_IF;
END_REGION

REGION Network 51: Stop PLC2 - reset AI_PLC2_Step_Bon4_Khuay_Thuan
   RUNG wire#powerrail
      Contact( "AI_PLC2_Stop_Active" )
      R_Coil( "AI_PLC2_Step_Bon4_Khuay_Thuan" )
   END_RUNG
   // the same network as SCL:
   IF "AI_PLC2_Stop_Active" THEN "AI_PLC2_Step_Bon4_Khuay_Thuan" := FALSE; END_IF;
END_REGION

REGION Network 52: Stop PLC2 - reset AI_PLC2_Step_Bon4_Khuay_Nghich
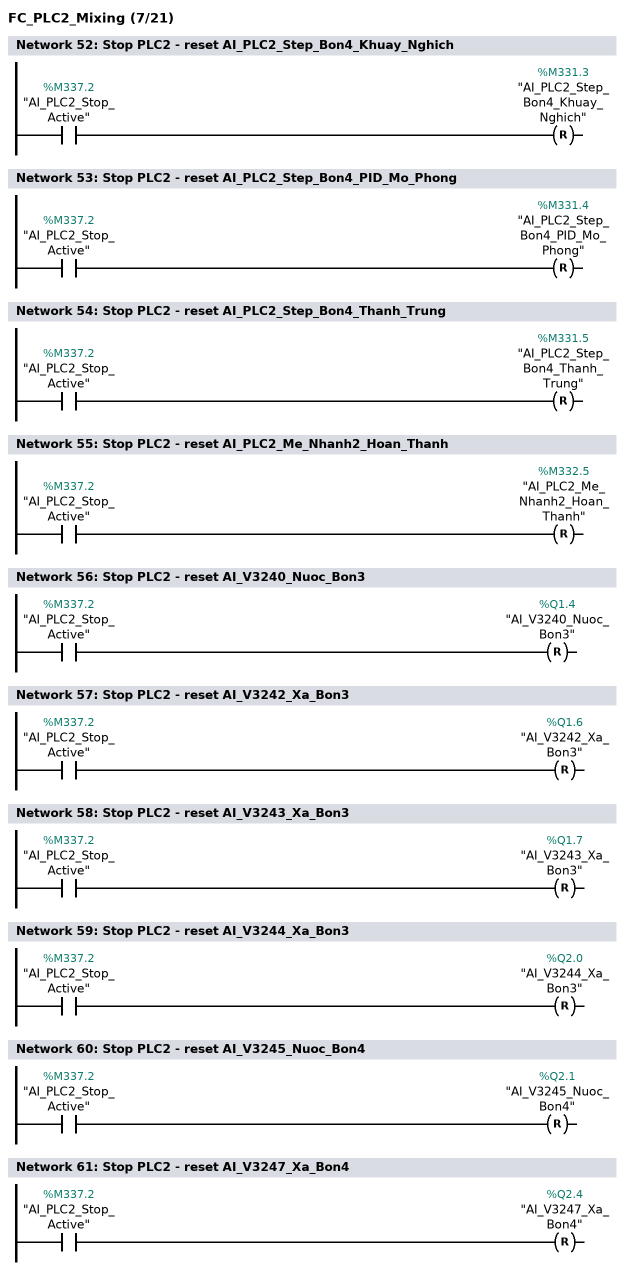
   RUNG wire#powerrail
      Contact( "AI_PLC2_Stop_Active" )
      R_Coil( "AI_PLC2_Step_Bon4_Khuay_Nghich" )
   END_RUNG
   // the same network as SCL:
   IF "AI_PLC2_Stop_Active" THEN "AI_PLC2_Step_Bon4_Khuay_Nghich" := FALSE; END_IF;
END_REGION

REGION Network 53: Stop PLC2 - reset AI_PLC2_Step_Bon4_PID_Mo_Phong
   RUNG wire#powerrail
      Contact( "AI_PLC2_Stop_Active" )
      R_Coil( "AI_PLC2_Step_Bon4_PID_Mo_Phong" )
   END_RUNG
   // the same network as SCL:
   IF "AI_PLC2_Stop_Active" THEN "AI_PLC2_Step_Bon4_PID_Mo_Phong" := FALSE; END_IF;
END_REGION

REGION Network 54: Stop PLC2 - reset AI_PLC2_Step_Bon4_Thanh_Trung
   RUNG wire#powerrail
      Contact( "AI_PLC2_Stop_Active" )
      R_Coil( "AI_PLC2_Step_Bon4_Thanh_Trung" )
   END_RUNG
   // the same network as SCL:
   IF "AI_PLC2_Stop_Active" THEN "AI_PLC2_Step_Bon4_Thanh_Trung" := FALSE; END_IF;
END_REGION

REGION Network 55: Stop PLC2 - reset AI_PLC2_Me_Nhanh2_Hoan_Thanh
   RUNG wire#powerrail
      Contact( "AI_PLC2_Stop_Active" )
      R_Coil( "AI_PLC2_Me_Nhanh2_Hoan_Thanh" )
   END_RUNG
   // the same network as SCL:
   IF "AI_PLC2_Stop_Active" THEN "AI_PLC2_Me_Nhanh2_Hoan_Thanh" := FALSE; END_IF;
END_REGION

REGION Network 56: Stop PLC2 - reset AI_V3240_Nuoc_Bon3
   RUNG wire#powerrail
      Contact( "AI_PLC2_Stop_Active" )
      R_Coil( "AI_V3240_Nuoc_Bon3" )
   END_RUNG
   // the same network as SCL:
   IF "AI_PLC2_Stop_Active" THEN "AI_V3240_Nuoc_Bon3" := FALSE; END_IF;
END_REGION

REGION Network 57: Stop PLC2 - reset AI_V3242_Xa_Bon3
   RUNG wire#powerrail
      Contact( "AI_PLC2_Stop_Active" )
      R_Coil( "AI_V3242_Xa_Bon3" )
   END_RUNG
   // the same network as SCL:
   IF "AI_PLC2_Stop_Active" THEN "AI_V3242_Xa_Bon3" := FALSE; END_IF;
END_REGION

REGION Network 58: Stop PLC2 - reset AI_V3243_Xa_Bon3
   RUNG wire#powerrail
      Contact( "AI_PLC2_Stop_Active" )
      R_Coil( "AI_V3243_Xa_Bon3" )
   END_RUNG
   // the same network as SCL:
   IF "AI_PLC2_Stop_Active" THEN "AI_V3243_Xa_Bon3" := FALSE; END_IF;
END_REGION

REGION Network 59: Stop PLC2 - reset AI_V3244_Xa_Bon3
   RUNG wire#powerrail
      Contact( "AI_PLC2_Stop_Active" )
      R_Coil( "AI_V3244_Xa_Bon3" )
   END_RUNG
   // the same network as SCL:
   IF "AI_PLC2_Stop_Active" THEN "AI_V3244_Xa_Bon3" := FALSE; END_IF;
END_REGION

REGION Network 60: Stop PLC2 - reset AI_V3245_Nuoc_Bon4
   RUNG wire#powerrail
      Contact( "AI_PLC2_Stop_Active" )
      R_Coil( "AI_V3245_Nuoc_Bon4" )
   END_RUNG
   // the same network as SCL:
   IF "AI_PLC2_Stop_Active" THEN "AI_V3245_Nuoc_Bon4" := FALSE; END_IF;
END_REGION

REGION Network 61: Stop PLC2 - reset AI_V3247_Xa_Bon4
   RUNG wire#powerrail
      Contact( "AI_PLC2_Stop_Active" )
      R_Coil( "AI_V3247_Xa_Bon4" )
   END_RUNG
   // the same network as SCL:
   IF "AI_PLC2_Stop_Active" THEN "AI_V3247_Xa_Bon4" := FALSE; END_IF;
END_REGION

REGION Network 62: Stop PLC2 - reset AI_V3248_Xa_Bon4
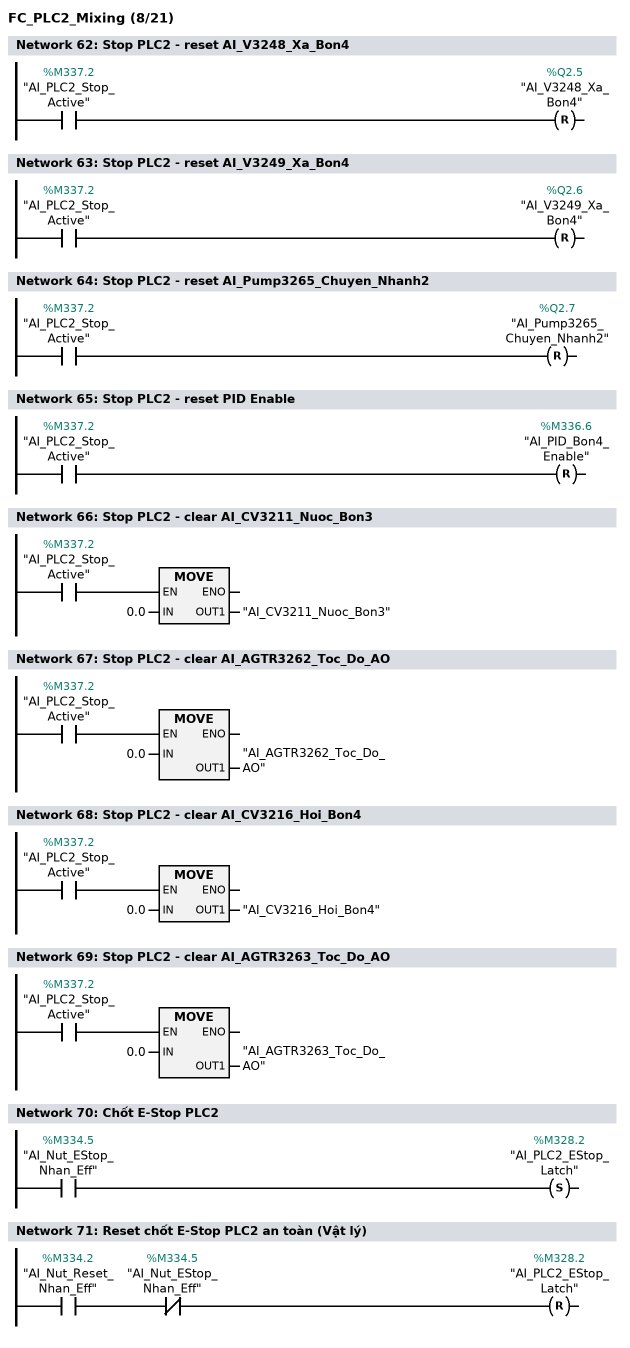
   RUNG wire#powerrail
      Contact( "AI_PLC2_Stop_Active" )
      R_Coil( "AI_V3248_Xa_Bon4" )
   END_RUNG
   // the same network as SCL:
   IF "AI_PLC2_Stop_Active" THEN "AI_V3248_Xa_Bon4" := FALSE; END_IF;
END_REGION

REGION Network 63: Stop PLC2 - reset AI_V3249_Xa_Bon4
   RUNG wire#powerrail
      Contact( "AI_PLC2_Stop_Active" )
      R_Coil( "AI_V3249_Xa_Bon4" )
   END_RUNG
   // the same network as SCL:
   IF "AI_PLC2_Stop_Active" THEN "AI_V3249_Xa_Bon4" := FALSE; END_IF;
END_REGION

REGION Network 64: Stop PLC2 - reset AI_Pump3265_Chuyen_Nhanh2
   RUNG wire#powerrail
      Contact( "AI_PLC2_Stop_Active" )
      R_Coil( "AI_Pump3265_Chuyen_Nhanh2" )
   END_RUNG
   // the same network as SCL:
   IF "AI_PLC2_Stop_Active" THEN "AI_Pump3265_Chuyen_Nhanh2" := FALSE; END_IF;
END_REGION

REGION Network 65: Stop PLC2 - reset PID Enable
   RUNG wire#powerrail
      Contact( "AI_PLC2_Stop_Active" )
      R_Coil( "AI_PID_Bon4_Enable" )
   END_RUNG
   // the same network as SCL:
   IF "AI_PLC2_Stop_Active" THEN "AI_PID_Bon4_Enable" := FALSE; END_IF;
END_REGION

REGION Network 66: Stop PLC2 - clear AI_CV3211_Nuoc_Bon3
   RUNG wire#powerrail
      Contact( "AI_PLC2_Stop_Active" )
      { S7_GenerateENO := "TRUE" } Move(in := 0.0, out1 => "AI_CV3211_Nuoc_Bon3")
   END_RUNG
   // the same network as SCL:
   IF "AI_PLC2_Stop_Active" THEN "AI_CV3211_Nuoc_Bon3" := 0.0; END_IF;
END_REGION

REGION Network 67: Stop PLC2 - clear AI_AGTR3262_Toc_Do_AO
   RUNG wire#powerrail
      Contact( "AI_PLC2_Stop_Active" )
      { S7_GenerateENO := "TRUE" } Move(in := 0.0, out1 => "AI_AGTR3262_Toc_Do_AO")
   END_RUNG
   // the same network as SCL:
   IF "AI_PLC2_Stop_Active" THEN "AI_AGTR3262_Toc_Do_AO" := 0.0; END_IF;
END_REGION

REGION Network 68: Stop PLC2 - clear AI_CV3216_Hoi_Bon4
   RUNG wire#powerrail
      Contact( "AI_PLC2_Stop_Active" )
      { S7_GenerateENO := "TRUE" } Move(in := 0.0, out1 => "AI_CV3216_Hoi_Bon4")
   END_RUNG
   // the same network as SCL:
   IF "AI_PLC2_Stop_Active" THEN "AI_CV3216_Hoi_Bon4" := 0.0; END_IF;
END_REGION

REGION Network 69: Stop PLC2 - clear AI_AGTR3263_Toc_Do_AO
   RUNG wire#powerrail
      Contact( "AI_PLC2_Stop_Active" )
      { S7_GenerateENO := "TRUE" } Move(in := 0.0, out1 => "AI_AGTR3263_Toc_Do_AO")
   END_RUNG
   // the same network as SCL:
   IF "AI_PLC2_Stop_Active" THEN "AI_AGTR3263_Toc_Do_AO" := 0.0; END_IF;
END_REGION

REGION Network 70: Chốt E-Stop PLC2
   RUNG wire#powerrail
      Contact( "AI_Nut_EStop_Nhan_Eff" )
      S_Coil( "AI_PLC2_EStop_Latch" )
   END_RUNG
   // the same network as SCL:
   IF "AI_Nut_EStop_Nhan_Eff" THEN "AI_PLC2_EStop_Latch" := TRUE; END_IF;
END_REGION

REGION Network 71: Reset chốt E-Stop PLC2 an toàn (Vật lý)
   RUNG wire#powerrail
      Contact( "AI_Nut_Reset_Nhan_Eff" )
      I_Contact( "AI_Nut_EStop_Nhan_Eff" )
      R_Coil( "AI_PLC2_EStop_Latch" )
   END_RUNG
   // the same network as SCL:
   IF "AI_Nut_Reset_Nhan_Eff" AND NOT "AI_Nut_EStop_Nhan_Eff" THEN "AI_PLC2_EStop_Latch" := FALSE; END_IF;
END_REGION

REGION Network 72: Reset chốt E-Stop PLC2 an toàn (HMI)
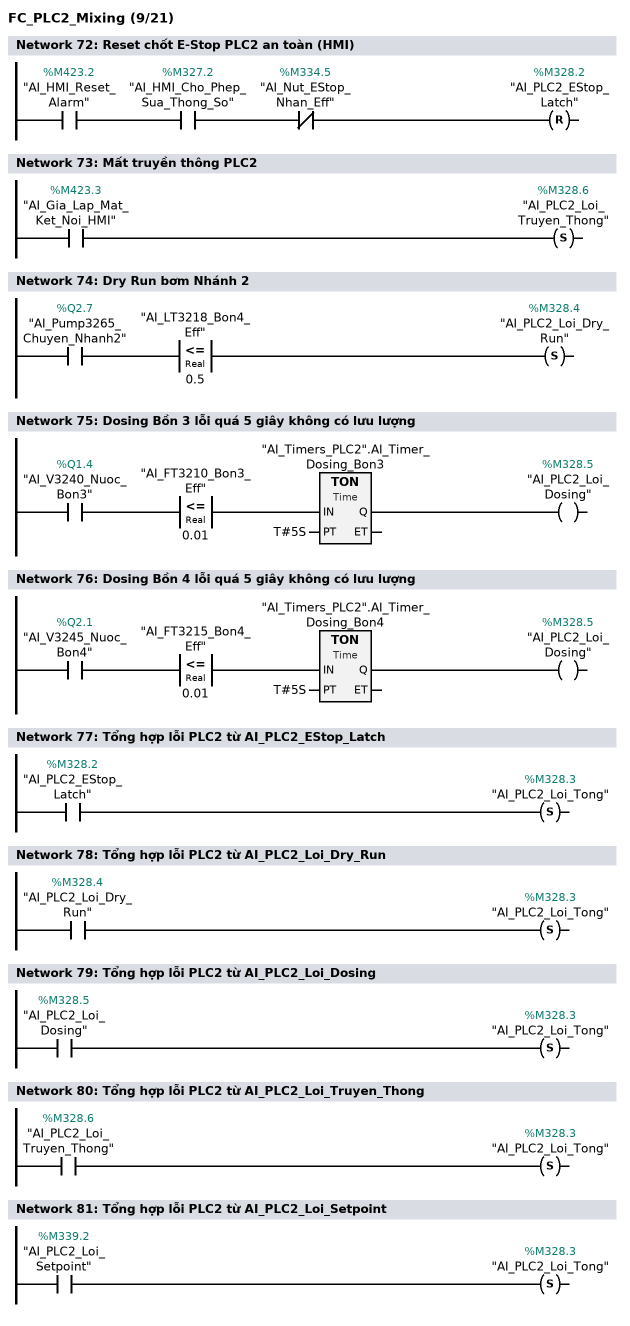
   RUNG wire#powerrail
      Contact( "AI_HMI_Reset_Alarm" )
      Contact( "AI_HMI_Cho_Phep_Sua_Thong_So" )
      I_Contact( "AI_Nut_EStop_Nhan_Eff" )
      R_Coil( "AI_PLC2_EStop_Latch" )
   END_RUNG
   // the same network as SCL:
   IF "AI_HMI_Reset_Alarm" AND "AI_HMI_Cho_Phep_Sua_Thong_So" AND NOT "AI_Nut_EStop_Nhan_Eff" THEN
       "AI_PLC2_EStop_Latch" := FALSE;
   END_IF;
END_REGION

REGION Network 73: Mất truyền thông PLC2
   RUNG wire#powerrail
      Contact( "AI_Gia_Lap_Mat_Ket_Noi_HMI" )
      S_Coil( "AI_PLC2_Loi_Truyen_Thong" )
   END_RUNG
   // the same network as SCL:
   IF "AI_Gia_Lap_Mat_Ket_Noi_HMI" THEN "AI_PLC2_Loi_Truyen_Thong" := TRUE; END_IF;
END_REGION

REGION Network 74: Dry Run bơm Nhánh 2
   RUNG wire#powerrail
      Contact( "AI_Pump3265_Chuyen_Nhanh2" )
      { S7_Templates := "SrcType := Real" } LE_Contact(in1 := "AI_LT3218_Bon4_Eff", in2 := 0.5)
      S_Coil( "AI_PLC2_Loi_Dry_Run" )
   END_RUNG
   // the same network as SCL:
   IF "AI_Pump3265_Chuyen_Nhanh2" AND ("AI_LT3218_Bon4_Eff" <= 0.5) THEN
       "AI_PLC2_Loi_Dry_Run" := TRUE;
   END_IF;
END_REGION

REGION Network 75: Dosing Bồn 3 lỗi quá 5 giây không có lưu lượng
   RUNG wire#powerrail
      Contact( "AI_V3240_Nuoc_Bon3" )
      { S7_Templates := "SrcType := Real" } LE_Contact(in1 := "AI_FT3210_Bon3_Eff", in2 := 0.01)
      { S7_Templates := "time_type := Time" } "AI_Timers_PLC2".AI_Timer_Dosing_Bon3.TON(pt := T#5S, et =>)
      Coil( "AI_PLC2_Loi_Dosing" )
   END_RUNG
   // the same network as SCL:
   "AI_Timers_PLC2".AI_Timer_Dosing_Bon3.TON(IN := "AI_V3240_Nuoc_Bon3" AND ("AI_FT3210_Bon3_Eff" <= 0.01),
                           PT := T#5S);
   "AI_PLC2_Loi_Dosing" := "AI_Timers_PLC2".AI_Timer_Dosing_Bon3.Q;
END_REGION

REGION Network 76: Dosing Bồn 4 lỗi quá 5 giây không có lưu lượng
   RUNG wire#powerrail
      Contact( "AI_V3245_Nuoc_Bon4" )
      { S7_Templates := "SrcType := Real" } LE_Contact(in1 := "AI_FT3215_Bon4_Eff", in2 := 0.01)
      { S7_Templates := "time_type := Time" } "AI_Timers_PLC2".AI_Timer_Dosing_Bon4.TON(pt := T#5S, et =>)
      Coil( "AI_PLC2_Loi_Dosing" )
   END_RUNG
   // the same network as SCL:
   "AI_Timers_PLC2".AI_Timer_Dosing_Bon4.TON(IN := "AI_V3245_Nuoc_Bon4" AND ("AI_FT3215_Bon4_Eff" <= 0.01),
                           PT := T#5S);
   "AI_PLC2_Loi_Dosing" := "AI_Timers_PLC2".AI_Timer_Dosing_Bon4.Q;
END_REGION

REGION Network 77: Tổng hợp lỗi PLC2 từ AI_PLC2_EStop_Latch
   RUNG wire#powerrail
      Contact( "AI_PLC2_EStop_Latch" )
      S_Coil( "AI_PLC2_Loi_Tong" )
   END_RUNG
   // the same network as SCL:
   IF "AI_PLC2_EStop_Latch" THEN "AI_PLC2_Loi_Tong" := TRUE; END_IF;
END_REGION

REGION Network 78: Tổng hợp lỗi PLC2 từ AI_PLC2_Loi_Dry_Run
   RUNG wire#powerrail
      Contact( "AI_PLC2_Loi_Dry_Run" )
      S_Coil( "AI_PLC2_Loi_Tong" )
   END_RUNG
   // the same network as SCL:
   IF "AI_PLC2_Loi_Dry_Run" THEN "AI_PLC2_Loi_Tong" := TRUE; END_IF;
END_REGION

REGION Network 79: Tổng hợp lỗi PLC2 từ AI_PLC2_Loi_Dosing
   RUNG wire#powerrail
      Contact( "AI_PLC2_Loi_Dosing" )
      S_Coil( "AI_PLC2_Loi_Tong" )
   END_RUNG
   // the same network as SCL:
   IF "AI_PLC2_Loi_Dosing" THEN "AI_PLC2_Loi_Tong" := TRUE; END_IF;
END_REGION

REGION Network 80: Tổng hợp lỗi PLC2 từ AI_PLC2_Loi_Truyen_Thong
   RUNG wire#powerrail
      Contact( "AI_PLC2_Loi_Truyen_Thong" )
      S_Coil( "AI_PLC2_Loi_Tong" )
   END_RUNG
   // the same network as SCL:
   IF "AI_PLC2_Loi_Truyen_Thong" THEN "AI_PLC2_Loi_Tong" := TRUE; END_IF;
END_REGION

REGION Network 81: Tổng hợp lỗi PLC2 từ AI_PLC2_Loi_Setpoint
   RUNG wire#powerrail
      Contact( "AI_PLC2_Loi_Setpoint" )
      S_Coil( "AI_PLC2_Loi_Tong" )
   END_RUNG
   // the same network as SCL:
   IF "AI_PLC2_Loi_Setpoint" THEN "AI_PLC2_Loi_Tong" := TRUE; END_IF;
END_REGION

REGION Network 82: Reset AI_PLC2_Loi_Tong từ nút vật lý
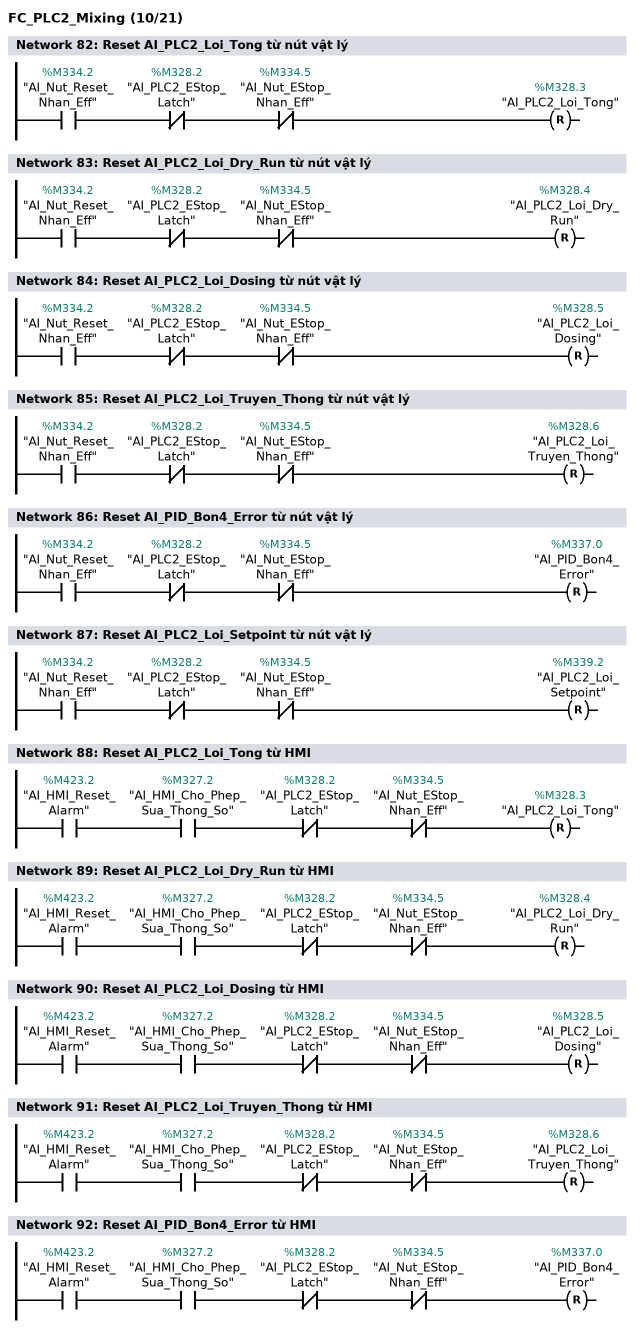
   RUNG wire#powerrail
      Contact( "AI_Nut_Reset_Nhan_Eff" )
      I_Contact( "AI_PLC2_EStop_Latch" )
      I_Contact( "AI_Nut_EStop_Nhan_Eff" )
      R_Coil( "AI_PLC2_Loi_Tong" )
   END_RUNG
   // the same network as SCL:
   IF "AI_Nut_Reset_Nhan_Eff" AND NOT "AI_PLC2_EStop_Latch" AND NOT "AI_Nut_EStop_Nhan_Eff" THEN
       "AI_PLC2_Loi_Tong" := FALSE;
   END_IF;
END_REGION

REGION Network 83: Reset AI_PLC2_Loi_Dry_Run từ nút vật lý
   RUNG wire#powerrail
      Contact( "AI_Nut_Reset_Nhan_Eff" )
      I_Contact( "AI_PLC2_EStop_Latch" )
      I_Contact( "AI_Nut_EStop_Nhan_Eff" )
      R_Coil( "AI_PLC2_Loi_Dry_Run" )
   END_RUNG
   // the same network as SCL:
   IF "AI_Nut_Reset_Nhan_Eff" AND NOT "AI_PLC2_EStop_Latch" AND NOT "AI_Nut_EStop_Nhan_Eff" THEN
       "AI_PLC2_Loi_Dry_Run" := FALSE;
   END_IF;
END_REGION

REGION Network 84: Reset AI_PLC2_Loi_Dosing từ nút vật lý
   RUNG wire#powerrail
      Contact( "AI_Nut_Reset_Nhan_Eff" )
      I_Contact( "AI_PLC2_EStop_Latch" )
      I_Contact( "AI_Nut_EStop_Nhan_Eff" )
      R_Coil( "AI_PLC2_Loi_Dosing" )
   END_RUNG
   // the same network as SCL:
   IF "AI_Nut_Reset_Nhan_Eff" AND NOT "AI_PLC2_EStop_Latch" AND NOT "AI_Nut_EStop_Nhan_Eff" THEN
       "AI_PLC2_Loi_Dosing" := FALSE;
   END_IF;
END_REGION

REGION Network 85: Reset AI_PLC2_Loi_Truyen_Thong từ nút vật lý
   RUNG wire#powerrail
      Contact( "AI_Nut_Reset_Nhan_Eff" )
      I_Contact( "AI_PLC2_EStop_Latch" )
      I_Contact( "AI_Nut_EStop_Nhan_Eff" )
      R_Coil( "AI_PLC2_Loi_Truyen_Thong" )
   END_RUNG
   // the same network as SCL:
   IF "AI_Nut_Reset_Nhan_Eff" AND NOT "AI_PLC2_EStop_Latch" AND NOT "AI_Nut_EStop_Nhan_Eff" THEN
       "AI_PLC2_Loi_Truyen_Thong" := FALSE;
   END_IF;
END_REGION

REGION Network 86: Reset AI_PID_Bon4_Error từ nút vật lý
   RUNG wire#powerrail
      Contact( "AI_Nut_Reset_Nhan_Eff" )
      I_Contact( "AI_PLC2_EStop_Latch" )
      I_Contact( "AI_Nut_EStop_Nhan_Eff" )
      R_Coil( "AI_PID_Bon4_Error" )
   END_RUNG
   // the same network as SCL:
   IF "AI_Nut_Reset_Nhan_Eff" AND NOT "AI_PLC2_EStop_Latch" AND NOT "AI_Nut_EStop_Nhan_Eff" THEN
       "AI_PID_Bon4_Error" := FALSE;
   END_IF;
END_REGION

REGION Network 87: Reset AI_PLC2_Loi_Setpoint từ nút vật lý
   RUNG wire#powerrail
      Contact( "AI_Nut_Reset_Nhan_Eff" )
      I_Contact( "AI_PLC2_EStop_Latch" )
      I_Contact( "AI_Nut_EStop_Nhan_Eff" )
      R_Coil( "AI_PLC2_Loi_Setpoint" )
   END_RUNG
   // the same network as SCL:
   IF "AI_Nut_Reset_Nhan_Eff" AND NOT "AI_PLC2_EStop_Latch" AND NOT "AI_Nut_EStop_Nhan_Eff" THEN
       "AI_PLC2_Loi_Setpoint" := FALSE;
   END_IF;
END_REGION

REGION Network 88: Reset AI_PLC2_Loi_Tong từ HMI
   RUNG wire#powerrail
      Contact( "AI_HMI_Reset_Alarm" )
      Contact( "AI_HMI_Cho_Phep_Sua_Thong_So" )
      I_Contact( "AI_PLC2_EStop_Latch" )
      I_Contact( "AI_Nut_EStop_Nhan_Eff" )
      R_Coil( "AI_PLC2_Loi_Tong" )
   END_RUNG
   // the same network as SCL:
   IF "AI_HMI_Reset_Alarm" AND "AI_HMI_Cho_Phep_Sua_Thong_So" AND NOT "AI_PLC2_EStop_Latch" AND NOT "AI_Nut_EStop_Nhan_Eff" THEN
       "AI_PLC2_Loi_Tong" := FALSE;
   END_IF;
END_REGION

REGION Network 89: Reset AI_PLC2_Loi_Dry_Run từ HMI
   RUNG wire#powerrail
      Contact( "AI_HMI_Reset_Alarm" )
      Contact( "AI_HMI_Cho_Phep_Sua_Thong_So" )
      I_Contact( "AI_PLC2_EStop_Latch" )
      I_Contact( "AI_Nut_EStop_Nhan_Eff" )
      R_Coil( "AI_PLC2_Loi_Dry_Run" )
   END_RUNG
   // the same network as SCL:
   IF "AI_HMI_Reset_Alarm" AND "AI_HMI_Cho_Phep_Sua_Thong_So" AND NOT "AI_PLC2_EStop_Latch" AND NOT "AI_Nut_EStop_Nhan_Eff" THEN
       "AI_PLC2_Loi_Dry_Run" := FALSE;
   END_IF;
END_REGION

REGION Network 90: Reset AI_PLC2_Loi_Dosing từ HMI
   RUNG wire#powerrail
      Contact( "AI_HMI_Reset_Alarm" )
      Contact( "AI_HMI_Cho_Phep_Sua_Thong_So" )
      I_Contact( "AI_PLC2_EStop_Latch" )
      I_Contact( "AI_Nut_EStop_Nhan_Eff" )
      R_Coil( "AI_PLC2_Loi_Dosing" )
   END_RUNG
   // the same network as SCL:
   IF "AI_HMI_Reset_Alarm" AND "AI_HMI_Cho_Phep_Sua_Thong_So" AND NOT "AI_PLC2_EStop_Latch" AND NOT "AI_Nut_EStop_Nhan_Eff" THEN
       "AI_PLC2_Loi_Dosing" := FALSE;
   END_IF;
END_REGION

REGION Network 91: Reset AI_PLC2_Loi_Truyen_Thong từ HMI
   RUNG wire#powerrail
      Contact( "AI_HMI_Reset_Alarm" )
      Contact( "AI_HMI_Cho_Phep_Sua_Thong_So" )
      I_Contact( "AI_PLC2_EStop_Latch" )
      I_Contact( "AI_Nut_EStop_Nhan_Eff" )
      R_Coil( "AI_PLC2_Loi_Truyen_Thong" )
   END_RUNG
   // the same network as SCL:
   IF "AI_HMI_Reset_Alarm" AND "AI_HMI_Cho_Phep_Sua_Thong_So" AND NOT "AI_PLC2_EStop_Latch" AND NOT "AI_Nut_EStop_Nhan_Eff" THEN
       "AI_PLC2_Loi_Truyen_Thong" := FALSE;
   END_IF;
END_REGION

REGION Network 92: Reset AI_PID_Bon4_Error từ HMI
   RUNG wire#powerrail
      Contact( "AI_HMI_Reset_Alarm" )
      Contact( "AI_HMI_Cho_Phep_Sua_Thong_So" )
      I_Contact( "AI_PLC2_EStop_Latch" )
      I_Contact( "AI_Nut_EStop_Nhan_Eff" )
      R_Coil( "AI_PID_Bon4_Error" )
   END_RUNG
   // the same network as SCL:
   IF "AI_HMI_Reset_Alarm" AND "AI_HMI_Cho_Phep_Sua_Thong_So" AND NOT "AI_PLC2_EStop_Latch" AND NOT "AI_Nut_EStop_Nhan_Eff" THEN
       "AI_PID_Bon4_Error" := FALSE;
   END_IF;
END_REGION

REGION Network 93: Reset AI_PLC2_Loi_Setpoint từ HMI
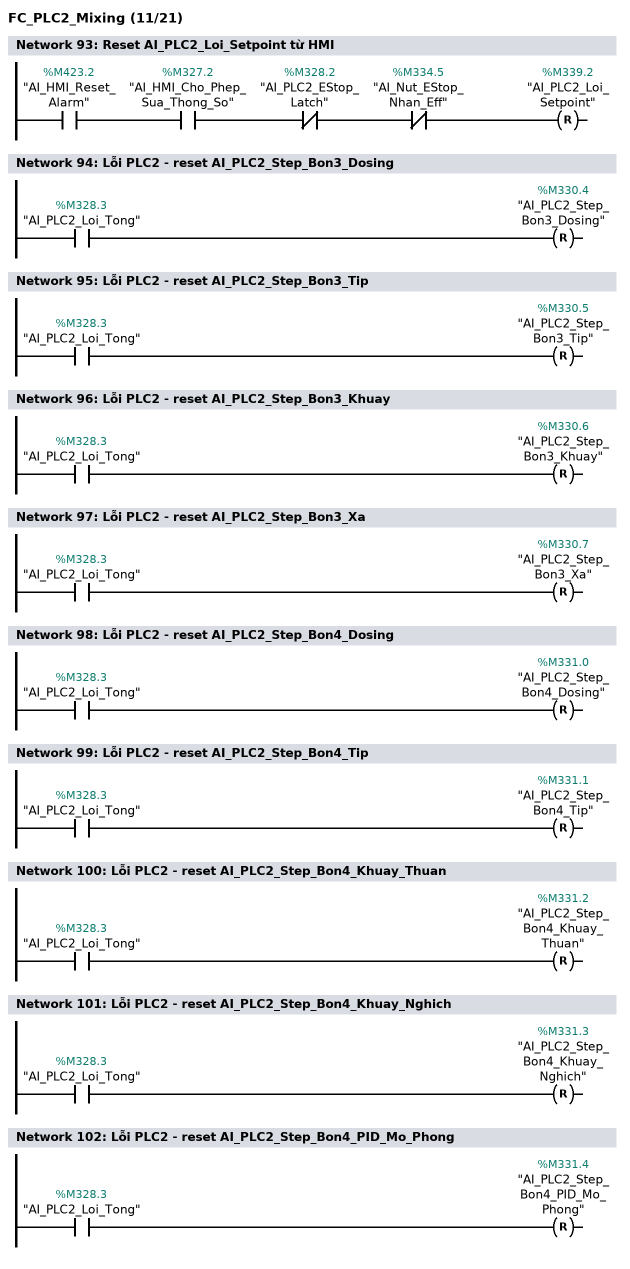
   RUNG wire#powerrail
      Contact( "AI_HMI_Reset_Alarm" )
      Contact( "AI_HMI_Cho_Phep_Sua_Thong_So" )
      I_Contact( "AI_PLC2_EStop_Latch" )
      I_Contact( "AI_Nut_EStop_Nhan_Eff" )
      R_Coil( "AI_PLC2_Loi_Setpoint" )
   END_RUNG
   // the same network as SCL:
   IF "AI_HMI_Reset_Alarm" AND "AI_HMI_Cho_Phep_Sua_Thong_So" AND NOT "AI_PLC2_EStop_Latch" AND NOT "AI_Nut_EStop_Nhan_Eff" THEN
       "AI_PLC2_Loi_Setpoint" := FALSE;
   END_IF;
END_REGION

REGION Network 94: Lỗi PLC2 - reset AI_PLC2_Step_Bon3_Dosing
   RUNG wire#powerrail
      Contact( "AI_PLC2_Loi_Tong" )
      R_Coil( "AI_PLC2_Step_Bon3_Dosing" )
   END_RUNG
   // the same network as SCL:
   IF "AI_PLC2_Loi_Tong" THEN "AI_PLC2_Step_Bon3_Dosing" := FALSE; END_IF;
END_REGION

REGION Network 95: Lỗi PLC2 - reset AI_PLC2_Step_Bon3_Tip
   RUNG wire#powerrail
      Contact( "AI_PLC2_Loi_Tong" )
      R_Coil( "AI_PLC2_Step_Bon3_Tip" )
   END_RUNG
   // the same network as SCL:
   IF "AI_PLC2_Loi_Tong" THEN "AI_PLC2_Step_Bon3_Tip" := FALSE; END_IF;
END_REGION

REGION Network 96: Lỗi PLC2 - reset AI_PLC2_Step_Bon3_Khuay
   RUNG wire#powerrail
      Contact( "AI_PLC2_Loi_Tong" )
      R_Coil( "AI_PLC2_Step_Bon3_Khuay" )
   END_RUNG
   // the same network as SCL:
   IF "AI_PLC2_Loi_Tong" THEN "AI_PLC2_Step_Bon3_Khuay" := FALSE; END_IF;
END_REGION

REGION Network 97: Lỗi PLC2 - reset AI_PLC2_Step_Bon3_Xa
   RUNG wire#powerrail
      Contact( "AI_PLC2_Loi_Tong" )
      R_Coil( "AI_PLC2_Step_Bon3_Xa" )
   END_RUNG
   // the same network as SCL:
   IF "AI_PLC2_Loi_Tong" THEN "AI_PLC2_Step_Bon3_Xa" := FALSE; END_IF;
END_REGION

REGION Network 98: Lỗi PLC2 - reset AI_PLC2_Step_Bon4_Dosing
   RUNG wire#powerrail
      Contact( "AI_PLC2_Loi_Tong" )
      R_Coil( "AI_PLC2_Step_Bon4_Dosing" )
   END_RUNG
   // the same network as SCL:
   IF "AI_PLC2_Loi_Tong" THEN "AI_PLC2_Step_Bon4_Dosing" := FALSE; END_IF;
END_REGION

REGION Network 99: Lỗi PLC2 - reset AI_PLC2_Step_Bon4_Tip
   RUNG wire#powerrail
      Contact( "AI_PLC2_Loi_Tong" )
      R_Coil( "AI_PLC2_Step_Bon4_Tip" )
   END_RUNG
   // the same network as SCL:
   IF "AI_PLC2_Loi_Tong" THEN "AI_PLC2_Step_Bon4_Tip" := FALSE; END_IF;
END_REGION

REGION Network 100: Lỗi PLC2 - reset AI_PLC2_Step_Bon4_Khuay_Thuan
   RUNG wire#powerrail
      Contact( "AI_PLC2_Loi_Tong" )
      R_Coil( "AI_PLC2_Step_Bon4_Khuay_Thuan" )
   END_RUNG
   // the same network as SCL:
   IF "AI_PLC2_Loi_Tong" THEN "AI_PLC2_Step_Bon4_Khuay_Thuan" := FALSE; END_IF;
END_REGION

REGION Network 101: Lỗi PLC2 - reset AI_PLC2_Step_Bon4_Khuay_Nghich
   RUNG wire#powerrail
      Contact( "AI_PLC2_Loi_Tong" )
      R_Coil( "AI_PLC2_Step_Bon4_Khuay_Nghich" )
   END_RUNG
   // the same network as SCL:
   IF "AI_PLC2_Loi_Tong" THEN "AI_PLC2_Step_Bon4_Khuay_Nghich" := FALSE; END_IF;
END_REGION

REGION Network 102: Lỗi PLC2 - reset AI_PLC2_Step_Bon4_PID_Mo_Phong
   RUNG wire#powerrail
      Contact( "AI_PLC2_Loi_Tong" )
      R_Coil( "AI_PLC2_Step_Bon4_PID_Mo_Phong" )
   END_RUNG
   // the same network as SCL:
   IF "AI_PLC2_Loi_Tong" THEN "AI_PLC2_Step_Bon4_PID_Mo_Phong" := FALSE; END_IF;
END_REGION

REGION Network 103: Lỗi PLC2 - reset AI_PLC2_Step_Bon4_Thanh_Trung
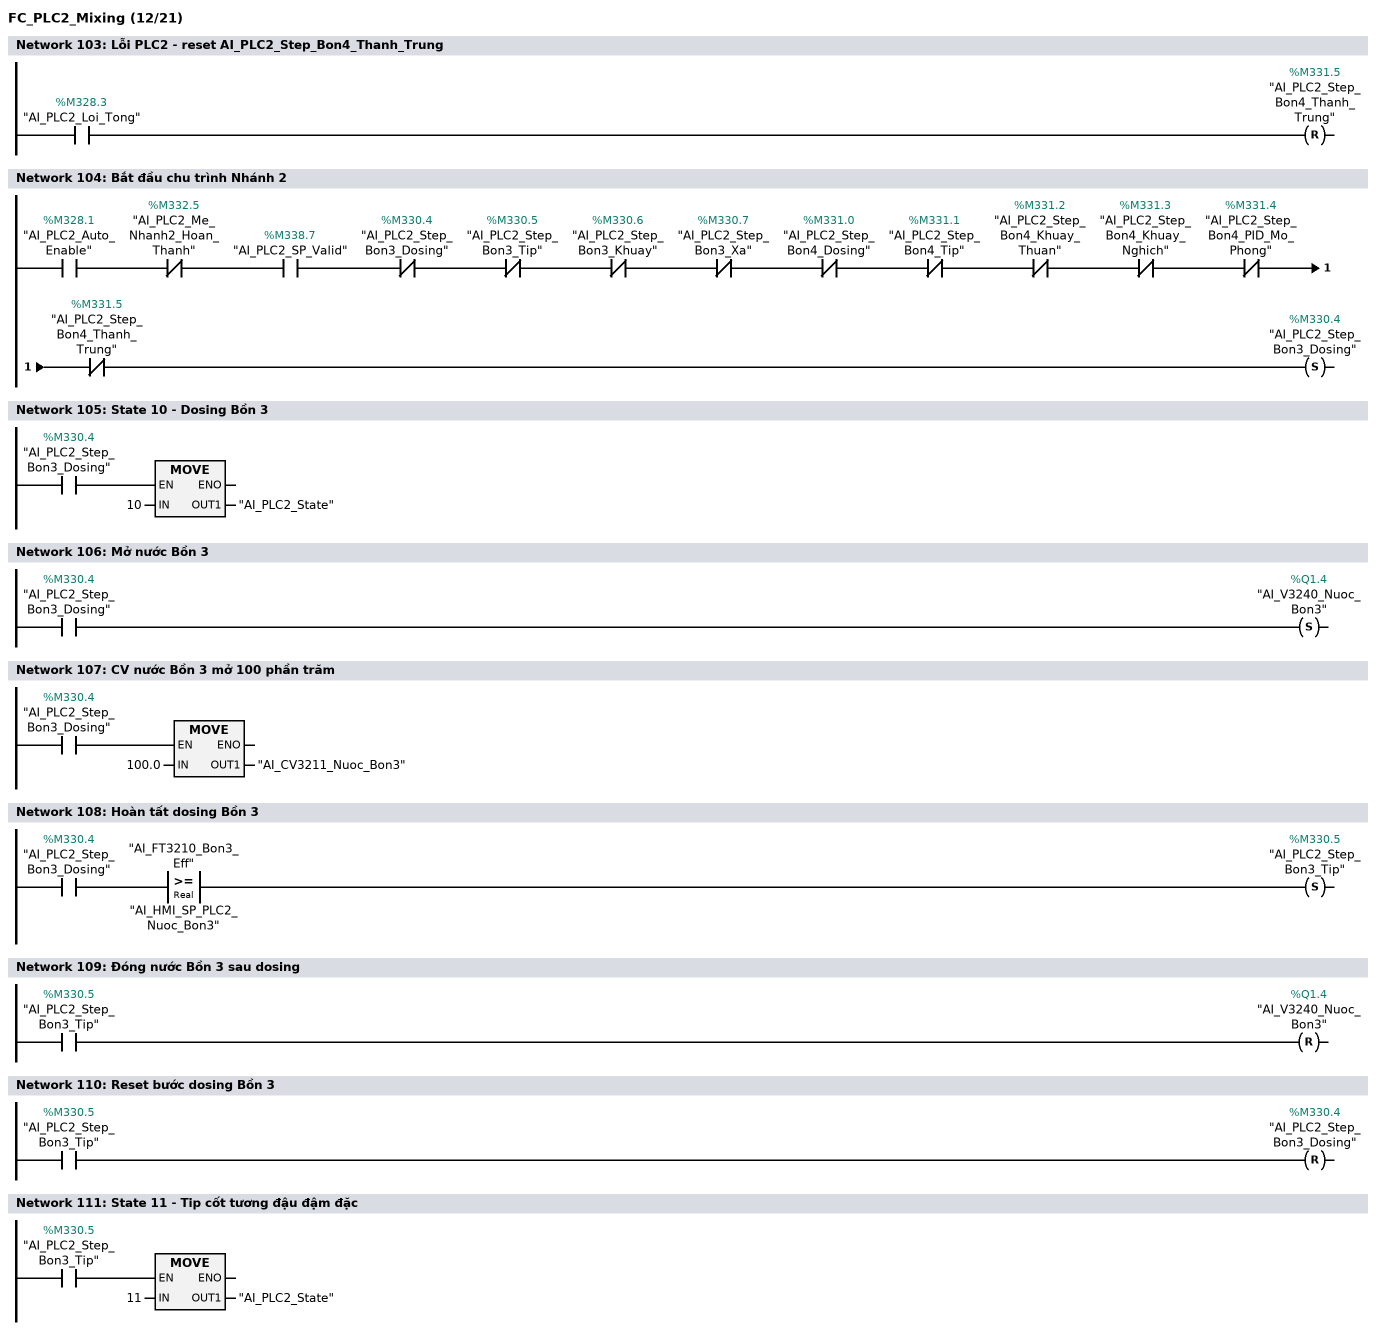
   RUNG wire#powerrail
      Contact( "AI_PLC2_Loi_Tong" )
      R_Coil( "AI_PLC2_Step_Bon4_Thanh_Trung" )
   END_RUNG
   // the same network as SCL:
   IF "AI_PLC2_Loi_Tong" THEN "AI_PLC2_Step_Bon4_Thanh_Trung" := FALSE; END_IF;
END_REGION

REGION Network 104: Bắt đầu chu trình Nhánh 2
   RUNG wire#powerrail
      Contact( "AI_PLC2_Auto_Enable" )
      I_Contact( "AI_PLC2_Me_Nhanh2_Hoan_Thanh" )
      Contact( "AI_PLC2_SP_Valid" )
      I_Contact( "AI_PLC2_Step_Bon3_Dosing" )
      I_Contact( "AI_PLC2_Step_Bon3_Tip" )
      I_Contact( "AI_PLC2_Step_Bon3_Khuay" )
      I_Contact( "AI_PLC2_Step_Bon3_Xa" )
      I_Contact( "AI_PLC2_Step_Bon4_Dosing" )
      I_Contact( "AI_PLC2_Step_Bon4_Tip" )
      I_Contact( "AI_PLC2_Step_Bon4_Khuay_Thuan" )
      I_Contact( "AI_PLC2_Step_Bon4_Khuay_Nghich" )
      I_Contact( "AI_PLC2_Step_Bon4_PID_Mo_Phong" )
      I_Contact( "AI_PLC2_Step_Bon4_Thanh_Trung" )
      S_Coil( "AI_PLC2_Step_Bon3_Dosing" )
   END_RUNG
   // the same network as SCL:
   IF "AI_PLC2_Auto_Enable" AND NOT "AI_PLC2_Me_Nhanh2_Hoan_Thanh" AND "AI_PLC2_SP_Valid" AND NOT "AI_PLC2_Step_Bon3_Dosing" AND NOT "AI_PLC2_Step_Bon3_Tip" AND NOT "AI_PLC2_Step_Bon3_Khuay" AND NOT "AI_PLC2_Step_Bon3_Xa" AND NOT "AI_PLC2_Step_Bon4_Dosing" AND NOT "AI_PLC2_Step_Bon4_Tip" AND NOT "AI_PLC2_Step_Bon4_Khuay_Thuan" AND NOT "AI_PLC2_Step_Bon4_Khuay_Nghich" AND NOT "AI_PLC2_Step_Bon4_PID_Mo_Phong" AND NOT "AI_PLC2_Step_Bon4_Thanh_Trung" THEN
       "AI_PLC2_Step_Bon3_Dosing" := TRUE;
   END_IF;
END_REGION

REGION Network 105: State 10 - Dosing Bồn 3
   RUNG wire#powerrail
      Contact( "AI_PLC2_Step_Bon3_Dosing" )
      { S7_GenerateENO := "TRUE" } Move(in := 10, out1 => "AI_PLC2_State")
   END_RUNG
   // the same network as SCL:
   IF "AI_PLC2_Step_Bon3_Dosing" THEN "AI_PLC2_State" := 10; END_IF;
END_REGION

REGION Network 106: Mở nước Bồn 3
   RUNG wire#powerrail
      Contact( "AI_PLC2_Step_Bon3_Dosing" )
      S_Coil( "AI_V3240_Nuoc_Bon3" )
   END_RUNG
   // the same network as SCL:
   IF "AI_PLC2_Step_Bon3_Dosing" THEN "AI_V3240_Nuoc_Bon3" := TRUE; END_IF;
END_REGION

REGION Network 107: CV nước Bồn 3 mở 100 phần trăm
   RUNG wire#powerrail
      Contact( "AI_PLC2_Step_Bon3_Dosing" )
      { S7_GenerateENO := "TRUE" } Move(in := 100.0, out1 => "AI_CV3211_Nuoc_Bon3")
   END_RUNG
   // the same network as SCL:
   IF "AI_PLC2_Step_Bon3_Dosing" THEN "AI_CV3211_Nuoc_Bon3" := 100.0; END_IF;
END_REGION

REGION Network 108: Hoàn tất dosing Bồn 3
   RUNG wire#powerrail
      Contact( "AI_PLC2_Step_Bon3_Dosing" )
      { S7_Templates := "SrcType := Real" } GE_Contact(in1 := "AI_FT3210_Bon3_Eff", in2 := "AI_HMI_SP_PLC2_Nuoc_Bon3")
      S_Coil( "AI_PLC2_Step_Bon3_Tip" )
   END_RUNG
   // the same network as SCL:
   IF "AI_PLC2_Step_Bon3_Dosing" AND ("AI_FT3210_Bon3_Eff" >= "AI_HMI_SP_PLC2_Nuoc_Bon3") THEN
       "AI_PLC2_Step_Bon3_Tip" := TRUE;
   END_IF;
END_REGION

REGION Network 109: Đóng nước Bồn 3 sau dosing
   RUNG wire#powerrail
      Contact( "AI_PLC2_Step_Bon3_Tip" )
      R_Coil( "AI_V3240_Nuoc_Bon3" )
   END_RUNG
   // the same network as SCL:
   IF "AI_PLC2_Step_Bon3_Tip" THEN "AI_V3240_Nuoc_Bon3" := FALSE; END_IF;
END_REGION

REGION Network 110: Reset bước dosing Bồn 3
   RUNG wire#powerrail
      Contact( "AI_PLC2_Step_Bon3_Tip" )
      R_Coil( "AI_PLC2_Step_Bon3_Dosing" )
   END_RUNG
   // the same network as SCL:
   IF "AI_PLC2_Step_Bon3_Tip" THEN "AI_PLC2_Step_Bon3_Dosing" := FALSE; END_IF;
END_REGION

REGION Network 111: State 11 - Tip cốt tương đậu đậm đặc
   RUNG wire#powerrail
      Contact( "AI_PLC2_Step_Bon3_Tip" )
      { S7_GenerateENO := "TRUE" } Move(in := 11, out1 => "AI_PLC2_State")
   END_RUNG
   // the same network as SCL:
   IF "AI_PLC2_Step_Bon3_Tip" THEN "AI_PLC2_State" := 11; END_IF;
END_REGION

REGION Network 112: Tip Bồn 3 xong chuyển sang khuấy
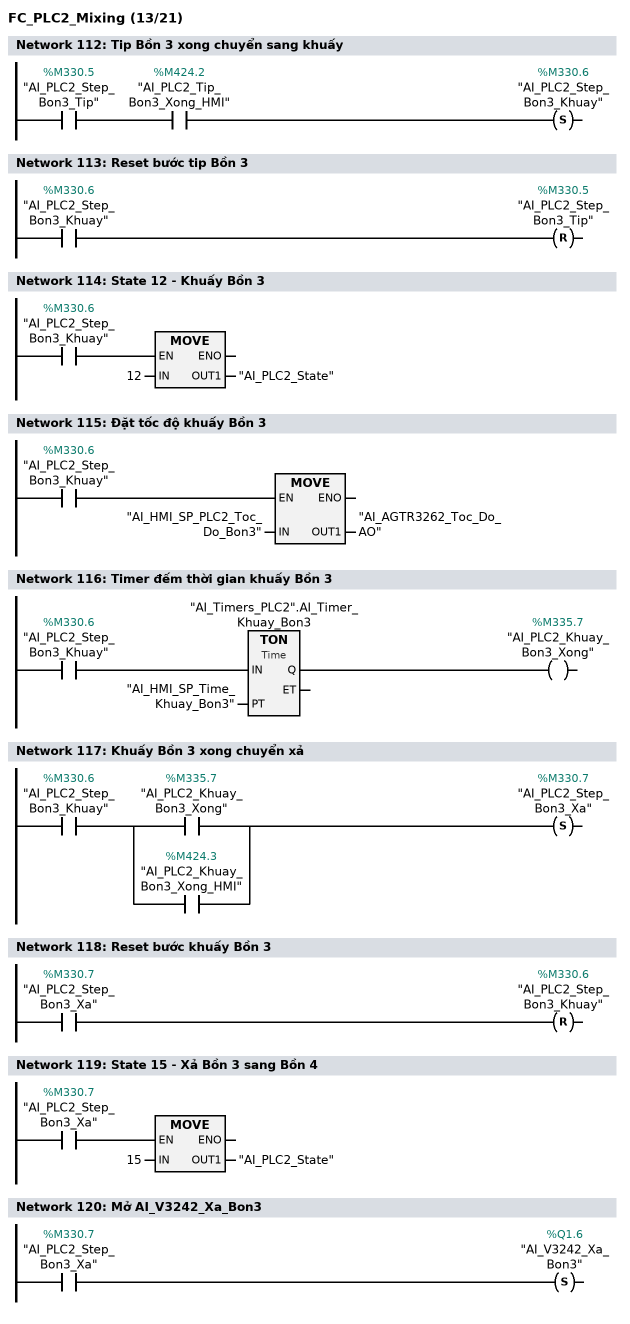
   RUNG wire#powerrail
      Contact( "AI_PLC2_Step_Bon3_Tip" )
      Contact( "AI_PLC2_Tip_Bon3_Xong_HMI" )
      S_Coil( "AI_PLC2_Step_Bon3_Khuay" )
   END_RUNG
   // the same network as SCL:
   IF "AI_PLC2_Step_Bon3_Tip" AND "AI_PLC2_Tip_Bon3_Xong_HMI" THEN "AI_PLC2_Step_Bon3_Khuay" := TRUE; END_IF;
END_REGION

REGION Network 113: Reset bước tip Bồn 3
   RUNG wire#powerrail
      Contact( "AI_PLC2_Step_Bon3_Khuay" )
      R_Coil( "AI_PLC2_Step_Bon3_Tip" )
   END_RUNG
   // the same network as SCL:
   IF "AI_PLC2_Step_Bon3_Khuay" THEN "AI_PLC2_Step_Bon3_Tip" := FALSE; END_IF;
END_REGION

REGION Network 114: State 12 - Khuấy Bồn 3
   RUNG wire#powerrail
      Contact( "AI_PLC2_Step_Bon3_Khuay" )
      { S7_GenerateENO := "TRUE" } Move(in := 12, out1 => "AI_PLC2_State")
   END_RUNG
   // the same network as SCL:
   IF "AI_PLC2_Step_Bon3_Khuay" THEN "AI_PLC2_State" := 12; END_IF;
END_REGION

REGION Network 115: Đặt tốc độ khuấy Bồn 3
   RUNG wire#powerrail
      Contact( "AI_PLC2_Step_Bon3_Khuay" )
      { S7_GenerateENO := "TRUE" } Move(in := "AI_HMI_SP_PLC2_Toc_Do_Bon3", out1 => "AI_AGTR3262_Toc_Do_AO")
   END_RUNG
   // the same network as SCL:
   IF "AI_PLC2_Step_Bon3_Khuay" THEN "AI_AGTR3262_Toc_Do_AO" := "AI_HMI_SP_PLC2_Toc_Do_Bon3"; END_IF;
END_REGION

REGION Network 116: Timer đếm thời gian khuấy Bồn 3
   RUNG wire#powerrail
      Contact( "AI_PLC2_Step_Bon3_Khuay" )
      { S7_Templates := "time_type := Time" } "AI_Timers_PLC2".AI_Timer_Khuay_Bon3.TON(pt := "AI_HMI_SP_Time_Khuay_Bon3", et =>)
      Coil( "AI_PLC2_Khuay_Bon3_Xong" )
   END_RUNG
   // the same network as SCL:
   "AI_Timers_PLC2".AI_Timer_Khuay_Bon3.TON(IN := "AI_PLC2_Step_Bon3_Khuay", PT := "AI_HMI_SP_Time_Khuay_Bon3");
   "AI_PLC2_Khuay_Bon3_Xong" := "AI_Timers_PLC2".AI_Timer_Khuay_Bon3.Q;
END_REGION

REGION Network 117: Khuấy Bồn 3 xong chuyển xả
   RUNG wire#powerrail
      Contact( "AI_PLC2_Step_Bon3_Khuay" )
      wire#w1
      Contact( "AI_PLC2_Khuay_Bon3_Xong" )
      wire#w2
      S_Coil( "AI_PLC2_Step_Bon3_Xa" )
   END_RUNG
   RUNG wire#w1
      Contact( "AI_PLC2_Khuay_Bon3_Xong_HMI" )
   END_RUNG wire#w2
   // the same network as SCL:
   IF "AI_PLC2_Step_Bon3_Khuay" AND ("AI_PLC2_Khuay_Bon3_Xong" OR "AI_PLC2_Khuay_Bon3_Xong_HMI") THEN
       "AI_PLC2_Step_Bon3_Xa" := TRUE;
   END_IF;
END_REGION

REGION Network 118: Reset bước khuấy Bồn 3
   RUNG wire#powerrail
      Contact( "AI_PLC2_Step_Bon3_Xa" )
      R_Coil( "AI_PLC2_Step_Bon3_Khuay" )
   END_RUNG
   // the same network as SCL:
   IF "AI_PLC2_Step_Bon3_Xa" THEN "AI_PLC2_Step_Bon3_Khuay" := FALSE; END_IF;
END_REGION

REGION Network 119: State 15 - Xả Bồn 3 sang Bồn 4
   RUNG wire#powerrail
      Contact( "AI_PLC2_Step_Bon3_Xa" )
      { S7_GenerateENO := "TRUE" } Move(in := 15, out1 => "AI_PLC2_State")
   END_RUNG
   // the same network as SCL:
   IF "AI_PLC2_Step_Bon3_Xa" THEN "AI_PLC2_State" := 15; END_IF;
END_REGION

REGION Network 120: Mở AI_V3242_Xa_Bon3
   RUNG wire#powerrail
      Contact( "AI_PLC2_Step_Bon3_Xa" )
      S_Coil( "AI_V3242_Xa_Bon3" )
   END_RUNG
   // the same network as SCL:
   IF "AI_PLC2_Step_Bon3_Xa" THEN "AI_V3242_Xa_Bon3" := TRUE; END_IF;
END_REGION

REGION Network 121: Mở AI_V3243_Xa_Bon3
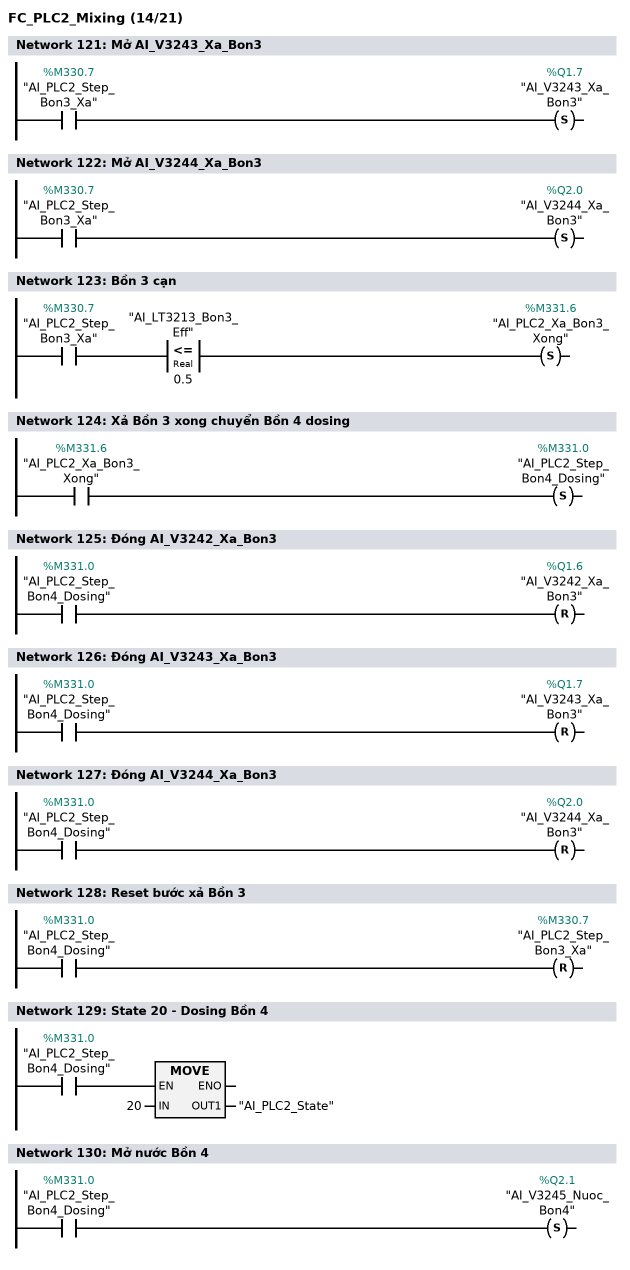
   RUNG wire#powerrail
      Contact( "AI_PLC2_Step_Bon3_Xa" )
      S_Coil( "AI_V3243_Xa_Bon3" )
   END_RUNG
   // the same network as SCL:
   IF "AI_PLC2_Step_Bon3_Xa" THEN "AI_V3243_Xa_Bon3" := TRUE; END_IF;
END_REGION

REGION Network 122: Mở AI_V3244_Xa_Bon3
   RUNG wire#powerrail
      Contact( "AI_PLC2_Step_Bon3_Xa" )
      S_Coil( "AI_V3244_Xa_Bon3" )
   END_RUNG
   // the same network as SCL:
   IF "AI_PLC2_Step_Bon3_Xa" THEN "AI_V3244_Xa_Bon3" := TRUE; END_IF;
END_REGION

REGION Network 123: Bồn 3 cạn
   RUNG wire#powerrail
      Contact( "AI_PLC2_Step_Bon3_Xa" )
      { S7_Templates := "SrcType := Real" } LE_Contact(in1 := "AI_LT3213_Bon3_Eff", in2 := 0.5)
      S_Coil( "AI_PLC2_Xa_Bon3_Xong" )
   END_RUNG
   // the same network as SCL:
   IF "AI_PLC2_Step_Bon3_Xa" AND ("AI_LT3213_Bon3_Eff" <= 0.5) THEN "AI_PLC2_Xa_Bon3_Xong" := TRUE; END_IF;
END_REGION

REGION Network 124: Xả Bồn 3 xong chuyển Bồn 4 dosing
   RUNG wire#powerrail
      Contact( "AI_PLC2_Xa_Bon3_Xong" )
      S_Coil( "AI_PLC2_Step_Bon4_Dosing" )
   END_RUNG
   // the same network as SCL:
   IF "AI_PLC2_Xa_Bon3_Xong" THEN "AI_PLC2_Step_Bon4_Dosing" := TRUE; END_IF;
END_REGION

REGION Network 125: Đóng AI_V3242_Xa_Bon3
   RUNG wire#powerrail
      Contact( "AI_PLC2_Step_Bon4_Dosing" )
      R_Coil( "AI_V3242_Xa_Bon3" )
   END_RUNG
   // the same network as SCL:
   IF "AI_PLC2_Step_Bon4_Dosing" THEN "AI_V3242_Xa_Bon3" := FALSE; END_IF;
END_REGION

REGION Network 126: Đóng AI_V3243_Xa_Bon3
   RUNG wire#powerrail
      Contact( "AI_PLC2_Step_Bon4_Dosing" )
      R_Coil( "AI_V3243_Xa_Bon3" )
   END_RUNG
   // the same network as SCL:
   IF "AI_PLC2_Step_Bon4_Dosing" THEN "AI_V3243_Xa_Bon3" := FALSE; END_IF;
END_REGION

REGION Network 127: Đóng AI_V3244_Xa_Bon3
   RUNG wire#powerrail
      Contact( "AI_PLC2_Step_Bon4_Dosing" )
      R_Coil( "AI_V3244_Xa_Bon3" )
   END_RUNG
   // the same network as SCL:
   IF "AI_PLC2_Step_Bon4_Dosing" THEN "AI_V3244_Xa_Bon3" := FALSE; END_IF;
END_REGION

REGION Network 128: Reset bước xả Bồn 3
   RUNG wire#powerrail
      Contact( "AI_PLC2_Step_Bon4_Dosing" )
      R_Coil( "AI_PLC2_Step_Bon3_Xa" )
   END_RUNG
   // the same network as SCL:
   IF "AI_PLC2_Step_Bon4_Dosing" THEN "AI_PLC2_Step_Bon3_Xa" := FALSE; END_IF;
END_REGION

REGION Network 129: State 20 - Dosing Bồn 4
   RUNG wire#powerrail
      Contact( "AI_PLC2_Step_Bon4_Dosing" )
      { S7_GenerateENO := "TRUE" } Move(in := 20, out1 => "AI_PLC2_State")
   END_RUNG
   // the same network as SCL:
   IF "AI_PLC2_Step_Bon4_Dosing" THEN "AI_PLC2_State" := 20; END_IF;
END_REGION

REGION Network 130: Mở nước Bồn 4
   RUNG wire#powerrail
      Contact( "AI_PLC2_Step_Bon4_Dosing" )
      S_Coil( "AI_V3245_Nuoc_Bon4" )
   END_RUNG
   // the same network as SCL:
   IF "AI_PLC2_Step_Bon4_Dosing" THEN "AI_V3245_Nuoc_Bon4" := TRUE; END_IF;
END_REGION

REGION Network 131: Hoàn tất dosing Bồn 4
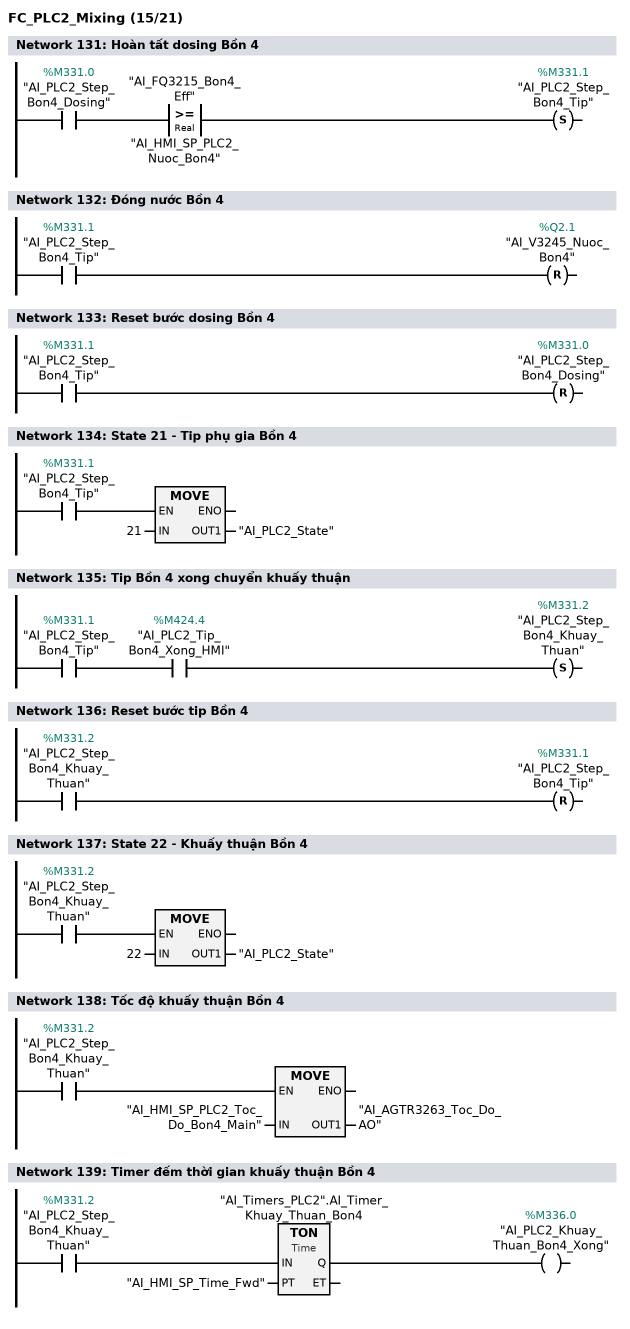
   RUNG wire#powerrail
      Contact( "AI_PLC2_Step_Bon4_Dosing" )
      { S7_Templates := "SrcType := Real" } GE_Contact(in1 := "AI_FQ3215_Bon4_Eff", in2 := "AI_HMI_SP_PLC2_Nuoc_Bon4")
      S_Coil( "AI_PLC2_Step_Bon4_Tip" )
   END_RUNG
   // the same network as SCL:
   IF "AI_PLC2_Step_Bon4_Dosing" AND ("AI_FQ3215_Bon4_Eff" >= "AI_HMI_SP_PLC2_Nuoc_Bon4") THEN
       "AI_PLC2_Step_Bon4_Tip" := TRUE;
   END_IF;
END_REGION

REGION Network 132: Đóng nước Bồn 4
   RUNG wire#powerrail
      Contact( "AI_PLC2_Step_Bon4_Tip" )
      R_Coil( "AI_V3245_Nuoc_Bon4" )
   END_RUNG
   // the same network as SCL:
   IF "AI_PLC2_Step_Bon4_Tip" THEN "AI_V3245_Nuoc_Bon4" := FALSE; END_IF;
END_REGION

REGION Network 133: Reset bước dosing Bồn 4
   RUNG wire#powerrail
      Contact( "AI_PLC2_Step_Bon4_Tip" )
      R_Coil( "AI_PLC2_Step_Bon4_Dosing" )
   END_RUNG
   // the same network as SCL:
   IF "AI_PLC2_Step_Bon4_Tip" THEN "AI_PLC2_Step_Bon4_Dosing" := FALSE; END_IF;
END_REGION

REGION Network 134: State 21 - Tip phụ gia Bồn 4
   RUNG wire#powerrail
      Contact( "AI_PLC2_Step_Bon4_Tip" )
      { S7_GenerateENO := "TRUE" } Move(in := 21, out1 => "AI_PLC2_State")
   END_RUNG
   // the same network as SCL:
   IF "AI_PLC2_Step_Bon4_Tip" THEN "AI_PLC2_State" := 21; END_IF;
END_REGION

REGION Network 135: Tip Bồn 4 xong chuyển khuấy thuận
   RUNG wire#powerrail
      Contact( "AI_PLC2_Step_Bon4_Tip" )
      Contact( "AI_PLC2_Tip_Bon4_Xong_HMI" )
      S_Coil( "AI_PLC2_Step_Bon4_Khuay_Thuan" )
   END_RUNG
   // the same network as SCL:
   IF "AI_PLC2_Step_Bon4_Tip" AND "AI_PLC2_Tip_Bon4_Xong_HMI" THEN
       "AI_PLC2_Step_Bon4_Khuay_Thuan" := TRUE;
   END_IF;
END_REGION

REGION Network 136: Reset bước tip Bồn 4
   RUNG wire#powerrail
      Contact( "AI_PLC2_Step_Bon4_Khuay_Thuan" )
      R_Coil( "AI_PLC2_Step_Bon4_Tip" )
   END_RUNG
   // the same network as SCL:
   IF "AI_PLC2_Step_Bon4_Khuay_Thuan" THEN "AI_PLC2_Step_Bon4_Tip" := FALSE; END_IF;
END_REGION

REGION Network 137: State 22 - Khuấy thuận Bồn 4
   RUNG wire#powerrail
      Contact( "AI_PLC2_Step_Bon4_Khuay_Thuan" )
      { S7_GenerateENO := "TRUE" } Move(in := 22, out1 => "AI_PLC2_State")
   END_RUNG
   // the same network as SCL:
   IF "AI_PLC2_Step_Bon4_Khuay_Thuan" THEN "AI_PLC2_State" := 22; END_IF;
END_REGION

REGION Network 138: Tốc độ khuấy thuận Bồn 4
   RUNG wire#powerrail
      Contact( "AI_PLC2_Step_Bon4_Khuay_Thuan" )
      { S7_GenerateENO := "TRUE" } Move(in := "AI_HMI_SP_PLC2_Toc_Do_Bon4_Main", out1 => "AI_AGTR3263_Toc_Do_AO")
   END_RUNG
   // the same network as SCL:
   IF "AI_PLC2_Step_Bon4_Khuay_Thuan" THEN
       "AI_AGTR3263_Toc_Do_AO" := "AI_HMI_SP_PLC2_Toc_Do_Bon4_Main";
   END_IF;
END_REGION

REGION Network 139: Timer đếm thời gian khuấy thuận Bồn 4
   RUNG wire#powerrail
      Contact( "AI_PLC2_Step_Bon4_Khuay_Thuan" )
      { S7_Templates := "time_type := Time" } "AI_Timers_PLC2".AI_Timer_Khuay_Thuan_Bon4.TON(pt := "AI_HMI_SP_Time_Fwd", et =>)
      Coil( "AI_PLC2_Khuay_Thuan_Bon4_Xong" )
   END_RUNG
   // the same network as SCL:
   "AI_Timers_PLC2".AI_Timer_Khuay_Thuan_Bon4.TON(IN := "AI_PLC2_Step_Bon4_Khuay_Thuan",
                           PT := "AI_HMI_SP_Time_Fwd");
   "AI_PLC2_Khuay_Thuan_Bon4_Xong" := "AI_Timers_PLC2".AI_Timer_Khuay_Thuan_Bon4.Q;
END_REGION

REGION Network 140: Hết khuấy thuận chuyển khuấy ngược Bồn 4
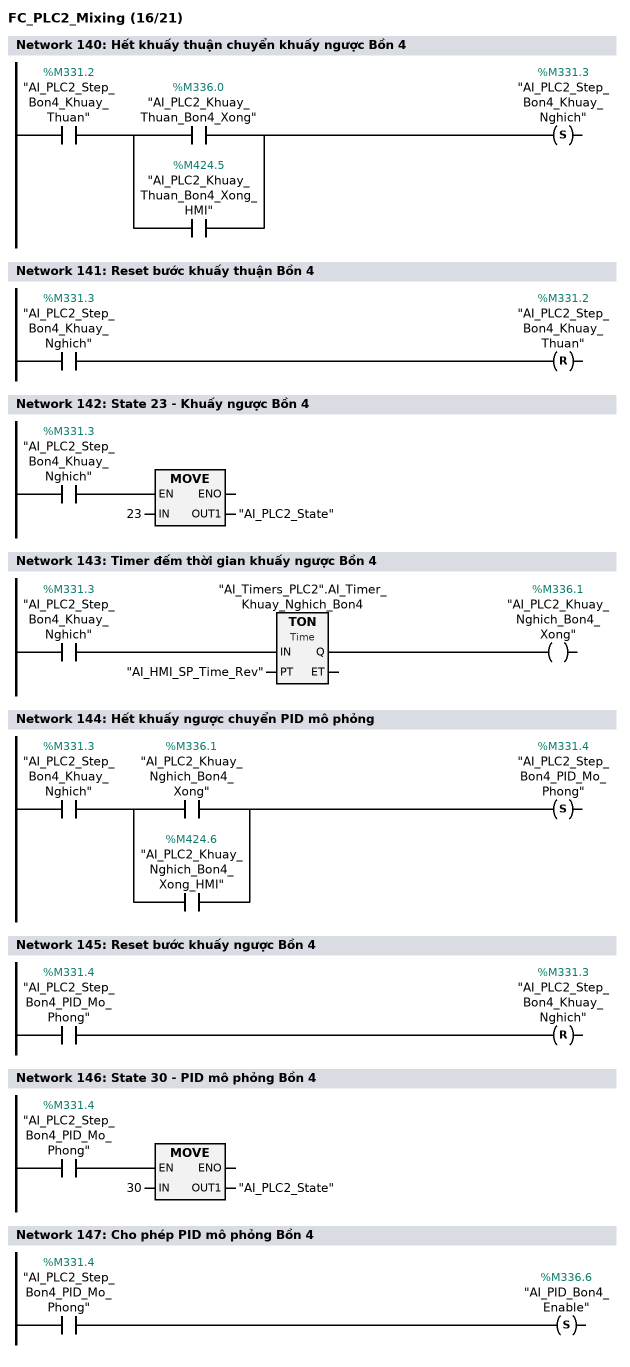
   RUNG wire#powerrail
      Contact( "AI_PLC2_Step_Bon4_Khuay_Thuan" )
      wire#w1
      Contact( "AI_PLC2_Khuay_Thuan_Bon4_Xong" )
      wire#w2
      S_Coil( "AI_PLC2_Step_Bon4_Khuay_Nghich" )
   END_RUNG
   RUNG wire#w1
      Contact( "AI_PLC2_Khuay_Thuan_Bon4_Xong_HMI" )
   END_RUNG wire#w2
   // the same network as SCL:
   IF "AI_PLC2_Step_Bon4_Khuay_Thuan" AND ("AI_PLC2_Khuay_Thuan_Bon4_Xong" OR "AI_PLC2_Khuay_Thuan_Bon4_Xong_HMI") THEN
       "AI_PLC2_Step_Bon4_Khuay_Nghich" := TRUE;
   END_IF;
END_REGION

REGION Network 141: Reset bước khuấy thuận Bồn 4
   RUNG wire#powerrail
      Contact( "AI_PLC2_Step_Bon4_Khuay_Nghich" )
      R_Coil( "AI_PLC2_Step_Bon4_Khuay_Thuan" )
   END_RUNG
   // the same network as SCL:
   IF "AI_PLC2_Step_Bon4_Khuay_Nghich" THEN "AI_PLC2_Step_Bon4_Khuay_Thuan" := FALSE; END_IF;
END_REGION

REGION Network 142: State 23 - Khuấy ngược Bồn 4
   RUNG wire#powerrail
      Contact( "AI_PLC2_Step_Bon4_Khuay_Nghich" )
      { S7_GenerateENO := "TRUE" } Move(in := 23, out1 => "AI_PLC2_State")
   END_RUNG
   // the same network as SCL:
   IF "AI_PLC2_Step_Bon4_Khuay_Nghich" THEN "AI_PLC2_State" := 23; END_IF;
END_REGION

REGION Network 143: Timer đếm thời gian khuấy ngược Bồn 4
   RUNG wire#powerrail
      Contact( "AI_PLC2_Step_Bon4_Khuay_Nghich" )
      { S7_Templates := "time_type := Time" } "AI_Timers_PLC2".AI_Timer_Khuay_Nghich_Bon4.TON(pt := "AI_HMI_SP_Time_Rev", et =>)
      Coil( "AI_PLC2_Khuay_Nghich_Bon4_Xong" )
   END_RUNG
   // the same network as SCL:
   "AI_Timers_PLC2".AI_Timer_Khuay_Nghich_Bon4.TON(IN := "AI_PLC2_Step_Bon4_Khuay_Nghich",
                           PT := "AI_HMI_SP_Time_Rev");
   "AI_PLC2_Khuay_Nghich_Bon4_Xong" := "AI_Timers_PLC2".AI_Timer_Khuay_Nghich_Bon4.Q;
END_REGION

REGION Network 144: Hết khuấy ngược chuyển PID mô phỏng
   RUNG wire#powerrail
      Contact( "AI_PLC2_Step_Bon4_Khuay_Nghich" )
      wire#w1
      Contact( "AI_PLC2_Khuay_Nghich_Bon4_Xong" )
      wire#w2
      S_Coil( "AI_PLC2_Step_Bon4_PID_Mo_Phong" )
   END_RUNG
   RUNG wire#w1
      Contact( "AI_PLC2_Khuay_Nghich_Bon4_Xong_HMI" )
   END_RUNG wire#w2
   // the same network as SCL:
   IF "AI_PLC2_Step_Bon4_Khuay_Nghich" AND ("AI_PLC2_Khuay_Nghich_Bon4_Xong" OR "AI_PLC2_Khuay_Nghich_Bon4_Xong_HMI") THEN
       "AI_PLC2_Step_Bon4_PID_Mo_Phong" := TRUE;
   END_IF;
END_REGION

REGION Network 145: Reset bước khuấy ngược Bồn 4
   RUNG wire#powerrail
      Contact( "AI_PLC2_Step_Bon4_PID_Mo_Phong" )
      R_Coil( "AI_PLC2_Step_Bon4_Khuay_Nghich" )
   END_RUNG
   // the same network as SCL:
   IF "AI_PLC2_Step_Bon4_PID_Mo_Phong" THEN "AI_PLC2_Step_Bon4_Khuay_Nghich" := FALSE; END_IF;
END_REGION

REGION Network 146: State 30 - PID mô phỏng Bồn 4
   RUNG wire#powerrail
      Contact( "AI_PLC2_Step_Bon4_PID_Mo_Phong" )
      { S7_GenerateENO := "TRUE" } Move(in := 30, out1 => "AI_PLC2_State")
   END_RUNG
   // the same network as SCL:
   IF "AI_PLC2_Step_Bon4_PID_Mo_Phong" THEN "AI_PLC2_State" := 30; END_IF;
END_REGION

REGION Network 147: Cho phép PID mô phỏng Bồn 4
   RUNG wire#powerrail
      Contact( "AI_PLC2_Step_Bon4_PID_Mo_Phong" )
      S_Coil( "AI_PID_Bon4_Enable" )
   END_RUNG
   // the same network as SCL:
   IF "AI_PLC2_Step_Bon4_PID_Mo_Phong" THEN "AI_PID_Bon4_Enable" := TRUE; END_IF;
END_REGION

REGION Network 148: Nạp SP PID Bồn 4
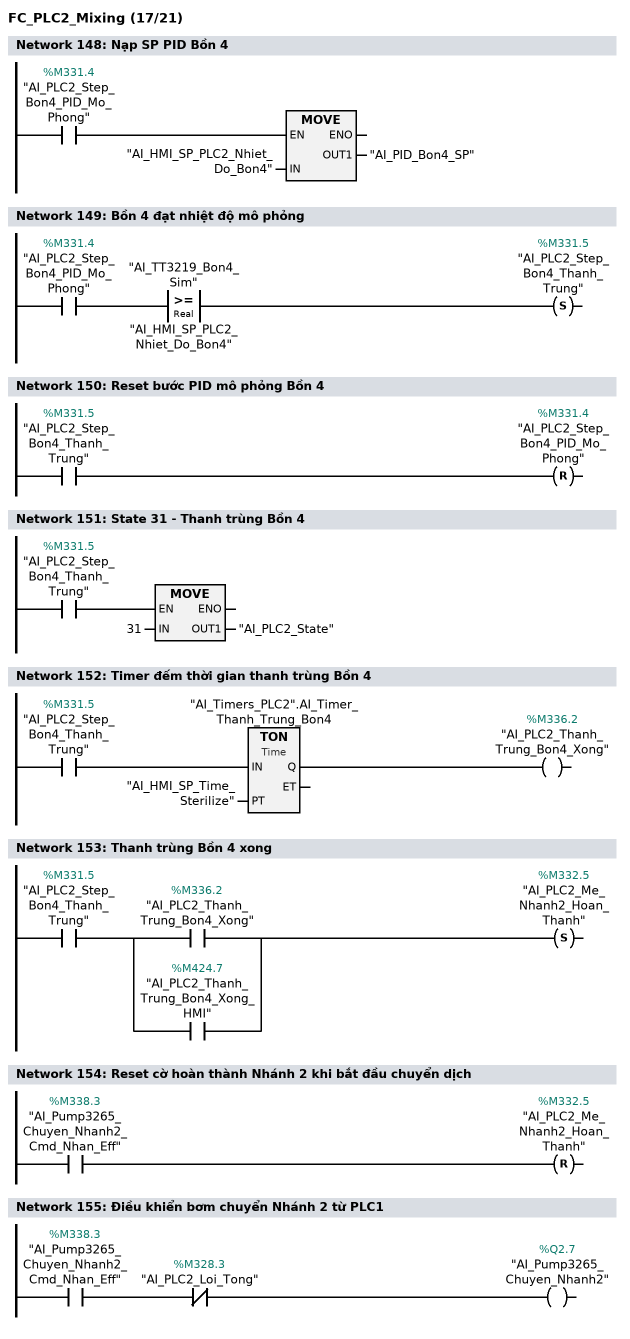
   RUNG wire#powerrail
      Contact( "AI_PLC2_Step_Bon4_PID_Mo_Phong" )
      { S7_GenerateENO := "TRUE" } Move(in := "AI_HMI_SP_PLC2_Nhiet_Do_Bon4", out1 => "AI_PID_Bon4_SP")
   END_RUNG
   // the same network as SCL:
   IF "AI_PLC2_Step_Bon4_PID_Mo_Phong" THEN "AI_PID_Bon4_SP" := "AI_HMI_SP_PLC2_Nhiet_Do_Bon4"; END_IF;
END_REGION

REGION Network 149: Bồn 4 đạt nhiệt độ mô phỏng
   RUNG wire#powerrail
      Contact( "AI_PLC2_Step_Bon4_PID_Mo_Phong" )
      { S7_Templates := "SrcType := Real" } GE_Contact(in1 := "AI_TT3219_Bon4_Sim", in2 := "AI_HMI_SP_PLC2_Nhiet_Do_Bon4")
      S_Coil( "AI_PLC2_Step_Bon4_Thanh_Trung" )
   END_RUNG
   // the same network as SCL:
   IF "AI_PLC2_Step_Bon4_PID_Mo_Phong" AND ("AI_TT3219_Bon4_Sim" >= "AI_HMI_SP_PLC2_Nhiet_Do_Bon4") THEN
       "AI_PLC2_Step_Bon4_Thanh_Trung" := TRUE;
   END_IF;
END_REGION

REGION Network 150: Reset bước PID mô phỏng Bồn 4
   RUNG wire#powerrail
      Contact( "AI_PLC2_Step_Bon4_Thanh_Trung" )
      R_Coil( "AI_PLC2_Step_Bon4_PID_Mo_Phong" )
   END_RUNG
   // the same network as SCL:
   IF "AI_PLC2_Step_Bon4_Thanh_Trung" THEN "AI_PLC2_Step_Bon4_PID_Mo_Phong" := FALSE; END_IF;
END_REGION

REGION Network 151: State 31 - Thanh trùng Bồn 4
   RUNG wire#powerrail
      Contact( "AI_PLC2_Step_Bon4_Thanh_Trung" )
      { S7_GenerateENO := "TRUE" } Move(in := 31, out1 => "AI_PLC2_State")
   END_RUNG
   // the same network as SCL:
   IF "AI_PLC2_Step_Bon4_Thanh_Trung" THEN "AI_PLC2_State" := 31; END_IF;
END_REGION

REGION Network 152: Timer đếm thời gian thanh trùng Bồn 4
   RUNG wire#powerrail
      Contact( "AI_PLC2_Step_Bon4_Thanh_Trung" )
      { S7_Templates := "time_type := Time" } "AI_Timers_PLC2".AI_Timer_Thanh_Trung_Bon4.TON(pt := "AI_HMI_SP_Time_Sterilize", et =>)
      Coil( "AI_PLC2_Thanh_Trung_Bon4_Xong" )
   END_RUNG
   // the same network as SCL:
   "AI_Timers_PLC2".AI_Timer_Thanh_Trung_Bon4.TON(IN := "AI_PLC2_Step_Bon4_Thanh_Trung",
                           PT := "AI_HMI_SP_Time_Sterilize");
   "AI_PLC2_Thanh_Trung_Bon4_Xong" := "AI_Timers_PLC2".AI_Timer_Thanh_Trung_Bon4.Q;
END_REGION

REGION Network 153: Thanh trùng Bồn 4 xong
   RUNG wire#powerrail
      Contact( "AI_PLC2_Step_Bon4_Thanh_Trung" )
      wire#w1
      Contact( "AI_PLC2_Thanh_Trung_Bon4_Xong" )
      wire#w2
      S_Coil( "AI_PLC2_Me_Nhanh2_Hoan_Thanh" )
   END_RUNG
   RUNG wire#w1
      Contact( "AI_PLC2_Thanh_Trung_Bon4_Xong_HMI" )
   END_RUNG wire#w2
   // the same network as SCL:
   IF "AI_PLC2_Step_Bon4_Thanh_Trung" AND ("AI_PLC2_Thanh_Trung_Bon4_Xong" OR "AI_PLC2_Thanh_Trung_Bon4_Xong_HMI") THEN
       "AI_PLC2_Me_Nhanh2_Hoan_Thanh" := TRUE;
   END_IF;
END_REGION

REGION Network 154: Reset cờ hoàn thành Nhánh 2 khi bắt đầu chuyển dịch
   RUNG wire#powerrail
      Contact( "AI_Pump3265_Chuyen_Nhanh2_Cmd_Nhan_Eff" )
      R_Coil( "AI_PLC2_Me_Nhanh2_Hoan_Thanh" )
   END_RUNG
   // the same network as SCL:
   IF "AI_Pump3265_Chuyen_Nhanh2_Cmd_Nhan_Eff" THEN "AI_PLC2_Me_Nhanh2_Hoan_Thanh" := FALSE; END_IF;
END_REGION

REGION Network 155: Điều khiển bơm chuyển Nhánh 2 từ PLC1
   RUNG wire#powerrail
      Contact( "AI_Pump3265_Chuyen_Nhanh2_Cmd_Nhan_Eff" )
      I_Contact( "AI_PLC2_Loi_Tong" )
      Coil( "AI_Pump3265_Chuyen_Nhanh2" )
   END_RUNG
   // the same network as SCL:
   "AI_Pump3265_Chuyen_Nhanh2" := "AI_Pump3265_Chuyen_Nhanh2_Cmd_Nhan_Eff" AND NOT "AI_PLC2_Loi_Tong";
END_REGION

REGION Network 156: Dừng PID khi hoàn thành Nhánh 2
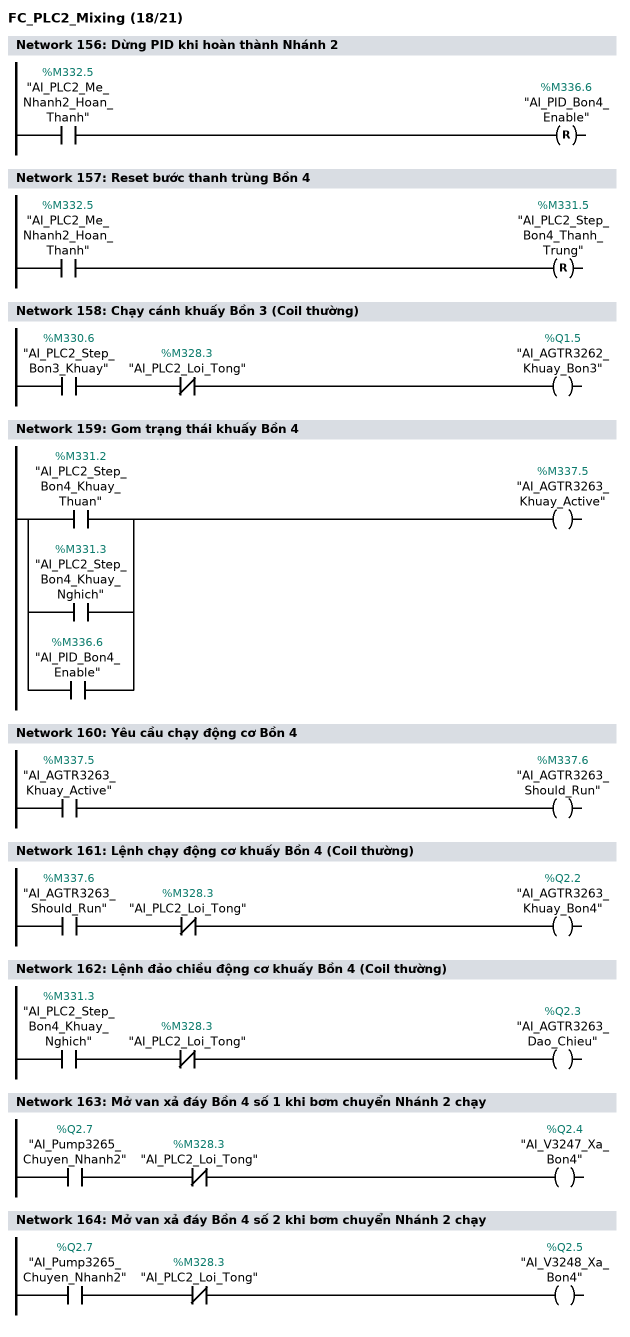
   RUNG wire#powerrail
      Contact( "AI_PLC2_Me_Nhanh2_Hoan_Thanh" )
      R_Coil( "AI_PID_Bon4_Enable" )
   END_RUNG
   // the same network as SCL:
   IF "AI_PLC2_Me_Nhanh2_Hoan_Thanh" THEN "AI_PID_Bon4_Enable" := FALSE; END_IF;
END_REGION

REGION Network 157: Reset bước thanh trùng Bồn 4
   RUNG wire#powerrail
      Contact( "AI_PLC2_Me_Nhanh2_Hoan_Thanh" )
      R_Coil( "AI_PLC2_Step_Bon4_Thanh_Trung" )
   END_RUNG
   // the same network as SCL:
   IF "AI_PLC2_Me_Nhanh2_Hoan_Thanh" THEN "AI_PLC2_Step_Bon4_Thanh_Trung" := FALSE; END_IF;
END_REGION

REGION Network 158: Chạy cánh khuấy Bồn 3 (Coil thường)
   RUNG wire#powerrail
      Contact( "AI_PLC2_Step_Bon3_Khuay" )
      I_Contact( "AI_PLC2_Loi_Tong" )
      Coil( "AI_AGTR3262_Khuay_Bon3" )
   END_RUNG
   // the same network as SCL:
   "AI_AGTR3262_Khuay_Bon3" := "AI_PLC2_Step_Bon3_Khuay" AND NOT "AI_PLC2_Loi_Tong";
END_REGION

REGION Network 159: Gom trạng thái khuấy Bồn 4
   RUNG wire#powerrail
      Contact( "AI_PLC2_Step_Bon4_Khuay_Thuan" )
      wire#w1
      Coil( "AI_AGTR3263_Khuay_Active" )
   END_RUNG
   RUNG wire#powerrail
      Contact( "AI_PLC2_Step_Bon4_Khuay_Nghich" )
   END_RUNG wire#w1
   RUNG wire#powerrail
      Contact( "AI_PID_Bon4_Enable" )
   END_RUNG wire#w1
   // the same network as SCL:
   "AI_AGTR3263_Khuay_Active" := "AI_PLC2_Step_Bon4_Khuay_Thuan" OR "AI_PLC2_Step_Bon4_Khuay_Nghich" OR "AI_PID_Bon4_Enable";
END_REGION

REGION Network 160: Yêu cầu chạy động cơ Bồn 4
   RUNG wire#powerrail
      Contact( "AI_AGTR3263_Khuay_Active" )
      Coil( "AI_AGTR3263_Should_Run" )
   END_RUNG
   // the same network as SCL:
   "AI_AGTR3263_Should_Run" := "AI_AGTR3263_Khuay_Active";
END_REGION

REGION Network 161: Lệnh chạy động cơ khuấy Bồn 4 (Coil thường)
   RUNG wire#powerrail
      Contact( "AI_AGTR3263_Should_Run" )
      I_Contact( "AI_PLC2_Loi_Tong" )
      Coil( "AI_AGTR3263_Khuay_Bon4" )
   END_RUNG
   // the same network as SCL:
   "AI_AGTR3263_Khuay_Bon4" := "AI_AGTR3263_Should_Run" AND NOT "AI_PLC2_Loi_Tong";
END_REGION

REGION Network 162: Lệnh đảo chiều động cơ khuấy Bồn 4 (Coil thường)
   RUNG wire#powerrail
      Contact( "AI_PLC2_Step_Bon4_Khuay_Nghich" )
      I_Contact( "AI_PLC2_Loi_Tong" )
      Coil( "AI_AGTR3263_Dao_Chieu" )
   END_RUNG
   // the same network as SCL:
   "AI_AGTR3263_Dao_Chieu" := "AI_PLC2_Step_Bon4_Khuay_Nghich" AND NOT "AI_PLC2_Loi_Tong";
END_REGION

REGION Network 163: Mở van xả đáy Bồn 4 số 1 khi bơm chuyển Nhánh 2 chạy
   RUNG wire#powerrail
      Contact( "AI_Pump3265_Chuyen_Nhanh2" )
      I_Contact( "AI_PLC2_Loi_Tong" )
      Coil( "AI_V3247_Xa_Bon4" )
   END_RUNG
   // the same network as SCL:
   "AI_V3247_Xa_Bon4" := "AI_Pump3265_Chuyen_Nhanh2" AND NOT "AI_PLC2_Loi_Tong";
END_REGION

REGION Network 164: Mở van xả đáy Bồn 4 số 2 khi bơm chuyển Nhánh 2 chạy
   RUNG wire#powerrail
      Contact( "AI_Pump3265_Chuyen_Nhanh2" )
      I_Contact( "AI_PLC2_Loi_Tong" )
      Coil( "AI_V3248_Xa_Bon4" )
   END_RUNG
   // the same network as SCL:
   "AI_V3248_Xa_Bon4" := "AI_Pump3265_Chuyen_Nhanh2" AND NOT "AI_PLC2_Loi_Tong";
END_REGION

REGION Network 165: Mở van xả đáy Bồn 4 số 3 khi bơm chuyển Nhánh 2 chạy
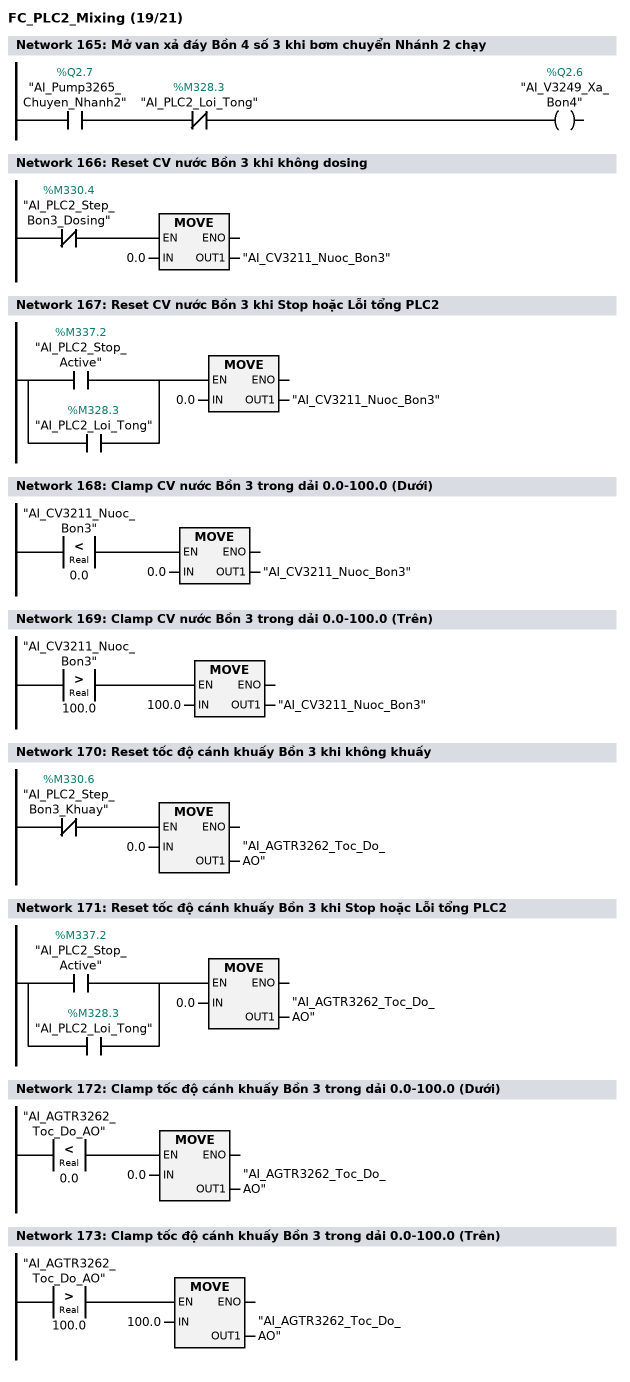
   RUNG wire#powerrail
      Contact( "AI_Pump3265_Chuyen_Nhanh2" )
      I_Contact( "AI_PLC2_Loi_Tong" )
      Coil( "AI_V3249_Xa_Bon4" )
   END_RUNG
   // the same network as SCL:
   "AI_V3249_Xa_Bon4" := "AI_Pump3265_Chuyen_Nhanh2" AND NOT "AI_PLC2_Loi_Tong";
END_REGION

REGION Network 166: Reset CV nước Bồn 3 khi không dosing
   RUNG wire#powerrail
      I_Contact( "AI_PLC2_Step_Bon3_Dosing" )
      { S7_GenerateENO := "TRUE" } Move(in := 0.0, out1 => "AI_CV3211_Nuoc_Bon3")
   END_RUNG
   // the same network as SCL:
   IF NOT "AI_PLC2_Step_Bon3_Dosing" THEN "AI_CV3211_Nuoc_Bon3" := 0.0; END_IF;
END_REGION

REGION Network 167: Reset CV nước Bồn 3 khi Stop hoặc Lỗi tổng PLC2
   RUNG wire#powerrail
      Contact( "AI_PLC2_Stop_Active" )
      wire#w1
      { S7_GenerateENO := "TRUE" } Move(in := 0.0, out1 => "AI_CV3211_Nuoc_Bon3")
   END_RUNG
   RUNG wire#powerrail
      Contact( "AI_PLC2_Loi_Tong" )
   END_RUNG wire#w1
   // the same network as SCL:
   IF "AI_PLC2_Stop_Active" OR "AI_PLC2_Loi_Tong" THEN "AI_CV3211_Nuoc_Bon3" := 0.0; END_IF;
END_REGION

REGION Network 168: Clamp CV nước Bồn 3 trong dải 0.0-100.0 (Dưới)
   RUNG wire#powerrail
      { S7_Templates := "SrcType := Real" } LT_Contact(in1 := "AI_CV3211_Nuoc_Bon3", in2 := 0.0)
      { S7_GenerateENO := "TRUE" } Move(in := 0.0, out1 => "AI_CV3211_Nuoc_Bon3")
   END_RUNG
   // the same network as SCL:
   IF "AI_CV3211_Nuoc_Bon3" < 0.0 THEN "AI_CV3211_Nuoc_Bon3" := 0.0; END_IF;
END_REGION

REGION Network 169: Clamp CV nước Bồn 3 trong dải 0.0-100.0 (Trên)
   RUNG wire#powerrail
      { S7_Templates := "SrcType := Real" } GT_Contact(in1 := "AI_CV3211_Nuoc_Bon3", in2 := 100.0)
      { S7_GenerateENO := "TRUE" } Move(in := 100.0, out1 => "AI_CV3211_Nuoc_Bon3")
   END_RUNG
   // the same network as SCL:
   IF "AI_CV3211_Nuoc_Bon3" > 100.0 THEN "AI_CV3211_Nuoc_Bon3" := 100.0; END_IF;
END_REGION

REGION Network 170: Reset tốc độ cánh khuấy Bồn 3 khi không khuấy
   RUNG wire#powerrail
      I_Contact( "AI_PLC2_Step_Bon3_Khuay" )
      { S7_GenerateENO := "TRUE" } Move(in := 0.0, out1 => "AI_AGTR3262_Toc_Do_AO")
   END_RUNG
   // the same network as SCL:
   IF NOT "AI_PLC2_Step_Bon3_Khuay" THEN "AI_AGTR3262_Toc_Do_AO" := 0.0; END_IF;
END_REGION

REGION Network 171: Reset tốc độ cánh khuấy Bồn 3 khi Stop hoặc Lỗi tổng PLC2
   RUNG wire#powerrail
      Contact( "AI_PLC2_Stop_Active" )
      wire#w1
      { S7_GenerateENO := "TRUE" } Move(in := 0.0, out1 => "AI_AGTR3262_Toc_Do_AO")
   END_RUNG
   RUNG wire#powerrail
      Contact( "AI_PLC2_Loi_Tong" )
   END_RUNG wire#w1
   // the same network as SCL:
   IF "AI_PLC2_Stop_Active" OR "AI_PLC2_Loi_Tong" THEN "AI_AGTR3262_Toc_Do_AO" := 0.0; END_IF;
END_REGION

REGION Network 172: Clamp tốc độ cánh khuấy Bồn 3 trong dải 0.0-100.0 (Dưới)
   RUNG wire#powerrail
      { S7_Templates := "SrcType := Real" } LT_Contact(in1 := "AI_AGTR3262_Toc_Do_AO", in2 := 0.0)
      { S7_GenerateENO := "TRUE" } Move(in := 0.0, out1 => "AI_AGTR3262_Toc_Do_AO")
   END_RUNG
   // the same network as SCL:
   IF "AI_AGTR3262_Toc_Do_AO" < 0.0 THEN "AI_AGTR3262_Toc_Do_AO" := 0.0; END_IF;
END_REGION

REGION Network 173: Clamp tốc độ cánh khuấy Bồn 3 trong dải 0.0-100.0 (Trên)
   RUNG wire#powerrail
      { S7_Templates := "SrcType := Real" } GT_Contact(in1 := "AI_AGTR3262_Toc_Do_AO", in2 := 100.0)
      { S7_GenerateENO := "TRUE" } Move(in := 100.0, out1 => "AI_AGTR3262_Toc_Do_AO")
   END_RUNG
   // the same network as SCL:
   IF "AI_AGTR3262_Toc_Do_AO" > 100.0 THEN "AI_AGTR3262_Toc_Do_AO" := 100.0; END_IF;
END_REGION

